REGION Network 146: Step[2901] :
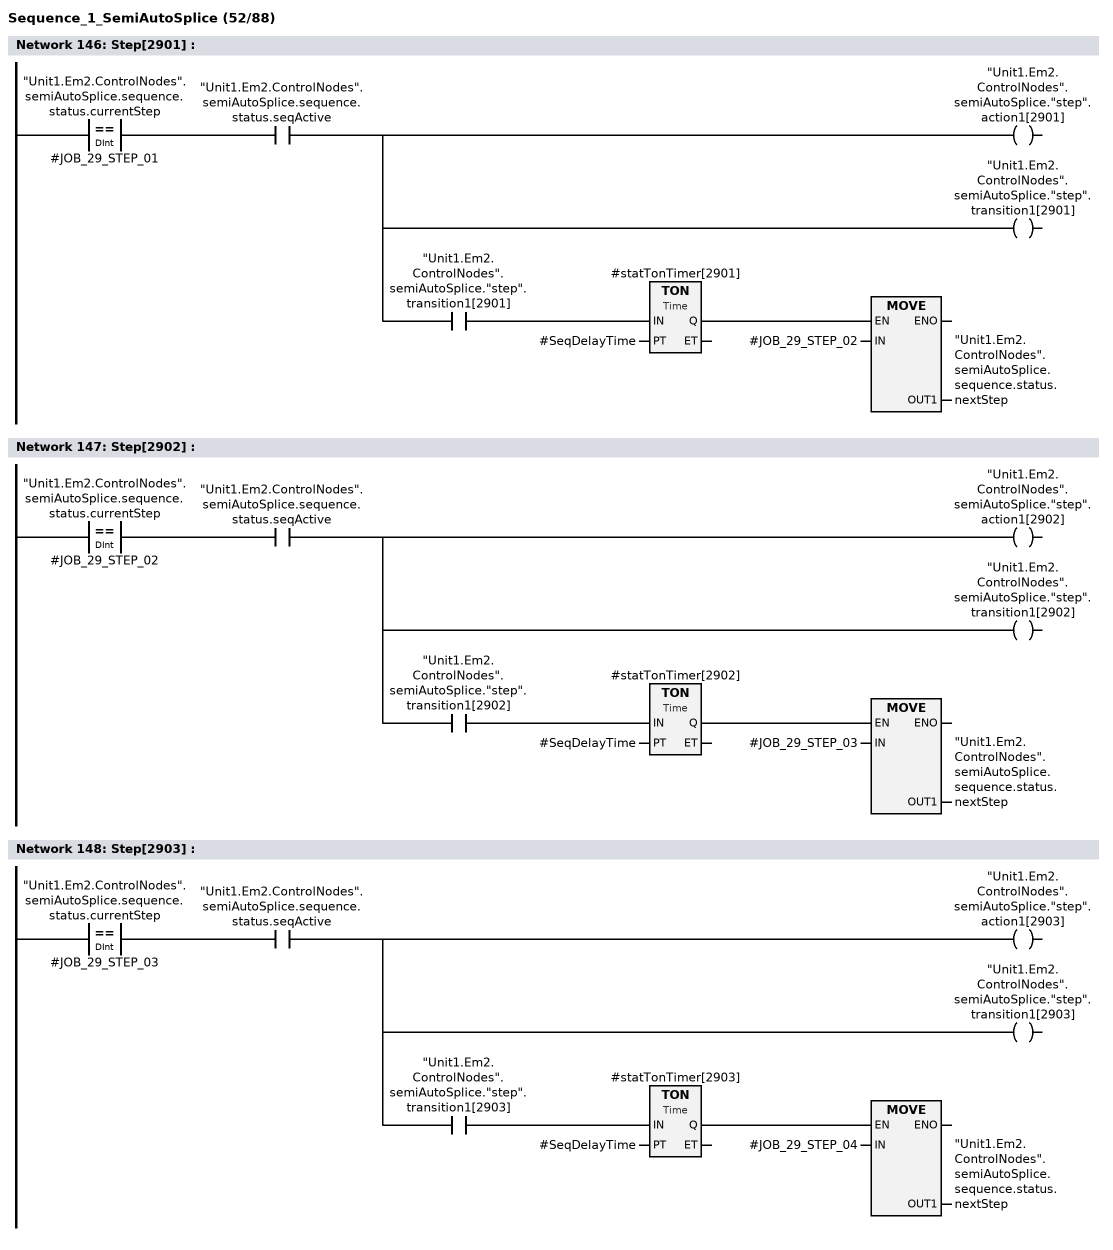
   RUNG wire#powerrail
      { S7_Templates := "SrcType := DInt" } EQ_Contact(in1 := "Unit1.Em2.ControlNodes".semiAutoSplice.sequence.status.currentStep, in2 := #JOB_29_STEP_01)
      Contact( "Unit1.Em2.ControlNodes".semiAutoSplice.sequence.status.seqActive )
      wire#w1
      Coil( "Unit1.Em2.ControlNodes".semiAutoSplice."step".action1[2901] )
   END_RUNG
   RUNG wire#w1
      Coil( "Unit1.Em2.ControlNodes".semiAutoSplice."step".transition1[2901] )
   END_RUNG
   RUNG wire#w1
      Contact( "Unit1.Em2.ControlNodes".semiAutoSplice."step".transition1[2901] )
      { S7_Templates := "time_type := Time" } #statTonTimer[2901].TON(pt := #SeqDelayTime, et =>)
      Move(in := #JOB_29_STEP_02, out1 => "Unit1.Em2.ControlNodes".semiAutoSplice.sequence.status.nextStep)
   END_RUNG
   // the same network as SCL:
   "Unit1.Em2.ControlNodes".semiAutoSplice."step".action1[2901] := ("Unit1.Em2.ControlNodes".semiAutoSplice.sequence.status.currentStep = #JOB_29_STEP_01) AND "Unit1.Em2.ControlNodes".semiAutoSplice.sequence.status.seqActive;
   "Unit1.Em2.ControlNodes".semiAutoSplice."step".transition1[2901] := ("Unit1.Em2.ControlNodes".semiAutoSplice.sequence.status.currentStep = #JOB_29_STEP_01) AND "Unit1.Em2.ControlNodes".semiAutoSplice.sequence.status.seqActive;
   #statTonTimer[2901].TON(IN := ("Unit1.Em2.ControlNodes".semiAutoSplice.sequence.status.currentStep = #JOB_29_STEP_01) AND "Unit1.Em2.ControlNodes".semiAutoSplice.sequence.status.seqActive AND "Unit1.Em2.ControlNodes".semiAutoSplice."step".transition1[2901],
                           PT := #SeqDelayTime);
   IF #statTonTimer[2901].Q THEN
       "Unit1.Em2.ControlNodes".semiAutoSplice.sequence.status.nextStep := #JOB_29_STEP_02;
   END_IF;
END_REGION

REGION Network 147: Step[2902] :
   RUNG wire#powerrail
      { S7_Templates := "SrcType := DInt" } EQ_Contact(in1 := "Unit1.Em2.ControlNodes".semiAutoSplice.sequence.status.currentStep, in2 := #JOB_29_STEP_02)
      Contact( "Unit1.Em2.ControlNodes".semiAutoSplice.sequence.status.seqActive )
      wire#w1
      Coil( "Unit1.Em2.ControlNodes".semiAutoSplice."step".action1[2902] )
   END_RUNG
   RUNG wire#w1
      Coil( "Unit1.Em2.ControlNodes".semiAutoSplice."step".transition1[2902] )
   END_RUNG
   RUNG wire#w1
      Contact( "Unit1.Em2.ControlNodes".semiAutoSplice."step".transition1[2902] )
      { S7_Templates := "time_type := Time" } #statTonTimer[2902].TON(pt := #SeqDelayTime, et =>)
      Move(in := #JOB_29_STEP_03, out1 => "Unit1.Em2.ControlNodes".semiAutoSplice.sequence.status.nextStep)
   END_RUNG
   // the same network as SCL:
   "Unit1.Em2.ControlNodes".semiAutoSplice."step".action1[2902] := ("Unit1.Em2.ControlNodes".semiAutoSplice.sequence.status.currentStep = #JOB_29_STEP_02) AND "Unit1.Em2.ControlNodes".semiAutoSplice.sequence.status.seqActive;
   "Unit1.Em2.ControlNodes".semiAutoSplice."step".transition1[2902] := ("Unit1.Em2.ControlNodes".semiAutoSplice.sequence.status.currentStep = #JOB_29_STEP_02) AND "Unit1.Em2.ControlNodes".semiAutoSplice.sequence.status.seqActive;
   #statTonTimer[2902].TON(IN := ("Unit1.Em2.ControlNodes".semiAutoSplice.sequence.status.currentStep = #JOB_29_STEP_02) AND "Unit1.Em2.ControlNodes".semiAutoSplice.sequence.status.seqActive AND "Unit1.Em2.ControlNodes".semiAutoSplice."step".transition1[2902],
                           PT := #SeqDelayTime);
   IF #statTonTimer[2902].Q THEN
       "Unit1.Em2.ControlNodes".semiAutoSplice.sequence.status.nextStep := #JOB_29_STEP_03;
   END_IF;
END_REGION

REGION Network 148: Step[2903] :
   RUNG wire#powerrail
      { S7_Templates := "SrcType := DInt" } EQ_Contact(in1 := "Unit1.Em2.ControlNodes".semiAutoSplice.sequence.status.currentStep, in2 := #JOB_29_STEP_03)
      Contact( "Unit1.Em2.ControlNodes".semiAutoSplice.sequence.status.seqActive )
      wire#w1
      Coil( "Unit1.Em2.ControlNodes".semiAutoSplice."step".action1[2903] )
   END_RUNG
   RUNG wire#w1
      Coil( "Unit1.Em2.ControlNodes".semiAutoSplice."step".transition1[2903] )
   END_RUNG
   RUNG wire#w1
      Contact( "Unit1.Em2.ControlNodes".semiAutoSplice."step".transition1[2903] )
      { S7_Templates := "time_type := Time" } #statTonTimer[2903].TON(pt := #SeqDelayTime, et =>)
      Move(in := #JOB_29_STEP_04, out1 => "Unit1.Em2.ControlNodes".semiAutoSplice.sequence.status.nextStep)
   END_RUNG
   // the same network as SCL:
   "Unit1.Em2.ControlNodes".semiAutoSplice."step".action1[2903] := ("Unit1.Em2.ControlNodes".semiAutoSplice.sequence.status.currentStep = #JOB_29_STEP_03) AND "Unit1.Em2.ControlNodes".semiAutoSplice.sequence.status.seqActive;
   "Unit1.Em2.ControlNodes".semiAutoSplice."step".transition1[2903] := ("Unit1.Em2.ControlNodes".semiAutoSplice.sequence.status.currentStep = #JOB_29_STEP_03) AND "Unit1.Em2.ControlNodes".semiAutoSplice.sequence.status.seqActive;
   #statTonTimer[2903].TON(IN := ("Unit1.Em2.ControlNodes".semiAutoSplice.sequence.status.currentStep = #JOB_29_STEP_03) AND "Unit1.Em2.ControlNodes".semiAutoSplice.sequence.status.seqActive AND "Unit1.Em2.ControlNodes".semiAutoSplice."step".transition1[2903],
                           PT := #SeqDelayTime);
   IF #statTonTimer[2903].Q THEN
       "Unit1.Em2.ControlNodes".semiAutoSplice.sequence.status.nextStep := #JOB_29_STEP_04;
   END_IF;
END_REGION

REGION Network 149: Step[2904] :
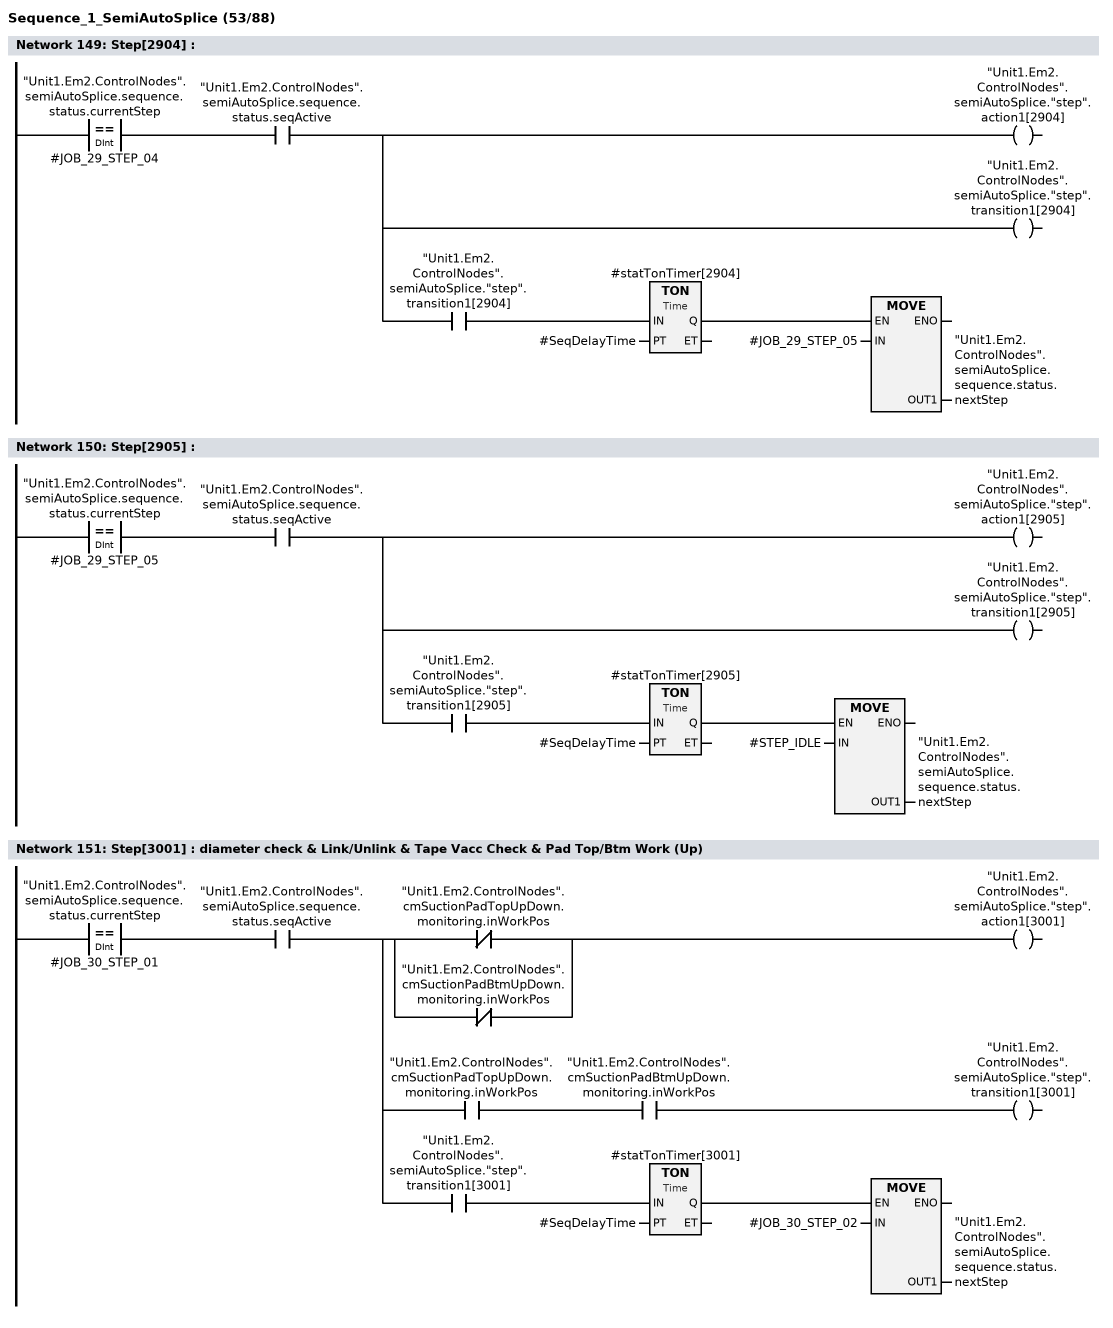
   RUNG wire#powerrail
      { S7_Templates := "SrcType := DInt" } EQ_Contact(in1 := "Unit1.Em2.ControlNodes".semiAutoSplice.sequence.status.currentStep, in2 := #JOB_29_STEP_04)
      Contact( "Unit1.Em2.ControlNodes".semiAutoSplice.sequence.status.seqActive )
      wire#w1
      Coil( "Unit1.Em2.ControlNodes".semiAutoSplice."step".action1[2904] )
   END_RUNG
   RUNG wire#w1
      Coil( "Unit1.Em2.ControlNodes".semiAutoSplice."step".transition1[2904] )
   END_RUNG
   RUNG wire#w1
      Contact( "Unit1.Em2.ControlNodes".semiAutoSplice."step".transition1[2904] )
      { S7_Templates := "time_type := Time" } #statTonTimer[2904].TON(pt := #SeqDelayTime, et =>)
      Move(in := #JOB_29_STEP_05, out1 => "Unit1.Em2.ControlNodes".semiAutoSplice.sequence.status.nextStep)
   END_RUNG
   // the same network as SCL:
   "Unit1.Em2.ControlNodes".semiAutoSplice."step".action1[2904] := ("Unit1.Em2.ControlNodes".semiAutoSplice.sequence.status.currentStep = #JOB_29_STEP_04) AND "Unit1.Em2.ControlNodes".semiAutoSplice.sequence.status.seqActive;
   "Unit1.Em2.ControlNodes".semiAutoSplice."step".transition1[2904] := ("Unit1.Em2.ControlNodes".semiAutoSplice.sequence.status.currentStep = #JOB_29_STEP_04) AND "Unit1.Em2.ControlNodes".semiAutoSplice.sequence.status.seqActive;
   #statTonTimer[2904].TON(IN := ("Unit1.Em2.ControlNodes".semiAutoSplice.sequence.status.currentStep = #JOB_29_STEP_04) AND "Unit1.Em2.ControlNodes".semiAutoSplice.sequence.status.seqActive AND "Unit1.Em2.ControlNodes".semiAutoSplice."step".transition1[2904],
                           PT := #SeqDelayTime);
   IF #statTonTimer[2904].Q THEN
       "Unit1.Em2.ControlNodes".semiAutoSplice.sequence.status.nextStep := #JOB_29_STEP_05;
   END_IF;
END_REGION

REGION Network 150: Step[2905] :
   RUNG wire#powerrail
      { S7_Templates := "SrcType := DInt" } EQ_Contact(in1 := "Unit1.Em2.ControlNodes".semiAutoSplice.sequence.status.currentStep, in2 := #JOB_29_STEP_05)
      Contact( "Unit1.Em2.ControlNodes".semiAutoSplice.sequence.status.seqActive )
      wire#w1
      Coil( "Unit1.Em2.ControlNodes".semiAutoSplice."step".action1[2905] )
   END_RUNG
   RUNG wire#w1
      Coil( "Unit1.Em2.ControlNodes".semiAutoSplice."step".transition1[2905] )
   END_RUNG
   RUNG wire#w1
      Contact( "Unit1.Em2.ControlNodes".semiAutoSplice."step".transition1[2905] )
      { S7_Templates := "time_type := Time" } #statTonTimer[2905].TON(pt := #SeqDelayTime, et =>)
      Move(in := #STEP_IDLE, out1 => "Unit1.Em2.ControlNodes".semiAutoSplice.sequence.status.nextStep)
   END_RUNG
   // the same network as SCL:
   "Unit1.Em2.ControlNodes".semiAutoSplice."step".action1[2905] := ("Unit1.Em2.ControlNodes".semiAutoSplice.sequence.status.currentStep = #JOB_29_STEP_05) AND "Unit1.Em2.ControlNodes".semiAutoSplice.sequence.status.seqActive;
   "Unit1.Em2.ControlNodes".semiAutoSplice."step".transition1[2905] := ("Unit1.Em2.ControlNodes".semiAutoSplice.sequence.status.currentStep = #JOB_29_STEP_05) AND "Unit1.Em2.ControlNodes".semiAutoSplice.sequence.status.seqActive;
   #statTonTimer[2905].TON(IN := ("Unit1.Em2.ControlNodes".semiAutoSplice.sequence.status.currentStep = #JOB_29_STEP_05) AND "Unit1.Em2.ControlNodes".semiAutoSplice.sequence.status.seqActive AND "Unit1.Em2.ControlNodes".semiAutoSplice."step".transition1[2905],
                           PT := #SeqDelayTime);
   IF #statTonTimer[2905].Q THEN
       "Unit1.Em2.ControlNodes".semiAutoSplice.sequence.status.nextStep := #STEP_IDLE;
   END_IF;
END_REGION

REGION Network 151: Step[3001] : diameter check & Link/Unlink & Tape Vacc Check & Pad Top/Btm Work (Up)
   RUNG wire#powerrail
      { S7_Templates := "SrcType := DInt" } EQ_Contact(in1 := "Unit1.Em2.ControlNodes".semiAutoSplice.sequence.status.currentStep, in2 := #JOB_30_STEP_01)
      Contact( "Unit1.Em2.ControlNodes".semiAutoSplice.sequence.status.seqActive )
      wire#w1
      I_Contact( "Unit1.Em2.ControlNodes".cmSuctionPadTopUpDown.monitoring.inWorkPos )
      wire#w2
      Coil( "Unit1.Em2.ControlNodes".semiAutoSplice."step".action1[3001] )
   END_RUNG
   RUNG wire#w1
      I_Contact( "Unit1.Em2.ControlNodes".cmSuctionPadBtmUpDown.monitoring.inWorkPos )
   END_RUNG wire#w2
   RUNG wire#w1
      Contact( "Unit1.Em2.ControlNodes".cmSuctionPadTopUpDown.monitoring.inWorkPos )
      Contact( "Unit1.Em2.ControlNodes".cmSuctionPadBtmUpDown.monitoring.inWorkPos )
      Coil( "Unit1.Em2.ControlNodes".semiAutoSplice."step".transition1[3001] )
   END_RUNG
   RUNG wire#w1
      Contact( "Unit1.Em2.ControlNodes".semiAutoSplice."step".transition1[3001] )
      { S7_Templates := "time_type := Time" } #statTonTimer[3001].TON(pt := #SeqDelayTime, et =>)
      Move(in := #JOB_30_STEP_02, out1 => "Unit1.Em2.ControlNodes".semiAutoSplice.sequence.status.nextStep)
   END_RUNG
   // the same network as SCL:
   #_w1 := ("Unit1.Em2.ControlNodes".semiAutoSplice.sequence.status.currentStep = #JOB_30_STEP_01) AND "Unit1.Em2.ControlNodes".semiAutoSplice.sequence.status.seqActive;
   "Unit1.Em2.ControlNodes".semiAutoSplice."step".action1[3001] := #_w1 AND (NOT "Unit1.Em2.ControlNodes".cmSuctionPadTopUpDown.monitoring.inWorkPos OR NOT "Unit1.Em2.ControlNodes".cmSuctionPadBtmUpDown.monitoring.inWorkPos);
   "Unit1.Em2.ControlNodes".semiAutoSplice."step".transition1[3001] := #_w1 AND "Unit1.Em2.ControlNodes".cmSuctionPadTopUpDown.monitoring.inWorkPos AND "Unit1.Em2.ControlNodes".cmSuctionPadBtmUpDown.monitoring.inWorkPos;
   #statTonTimer[3001].TON(IN := #_w1 AND "Unit1.Em2.ControlNodes".semiAutoSplice."step".transition1[3001],
                           PT := #SeqDelayTime);
   IF #statTonTimer[3001].Q THEN
       "Unit1.Em2.ControlNodes".semiAutoSplice.sequence.status.nextStep := #JOB_30_STEP_02;
   END_IF;
END_REGION

REGION Network 152: Step[3002] :
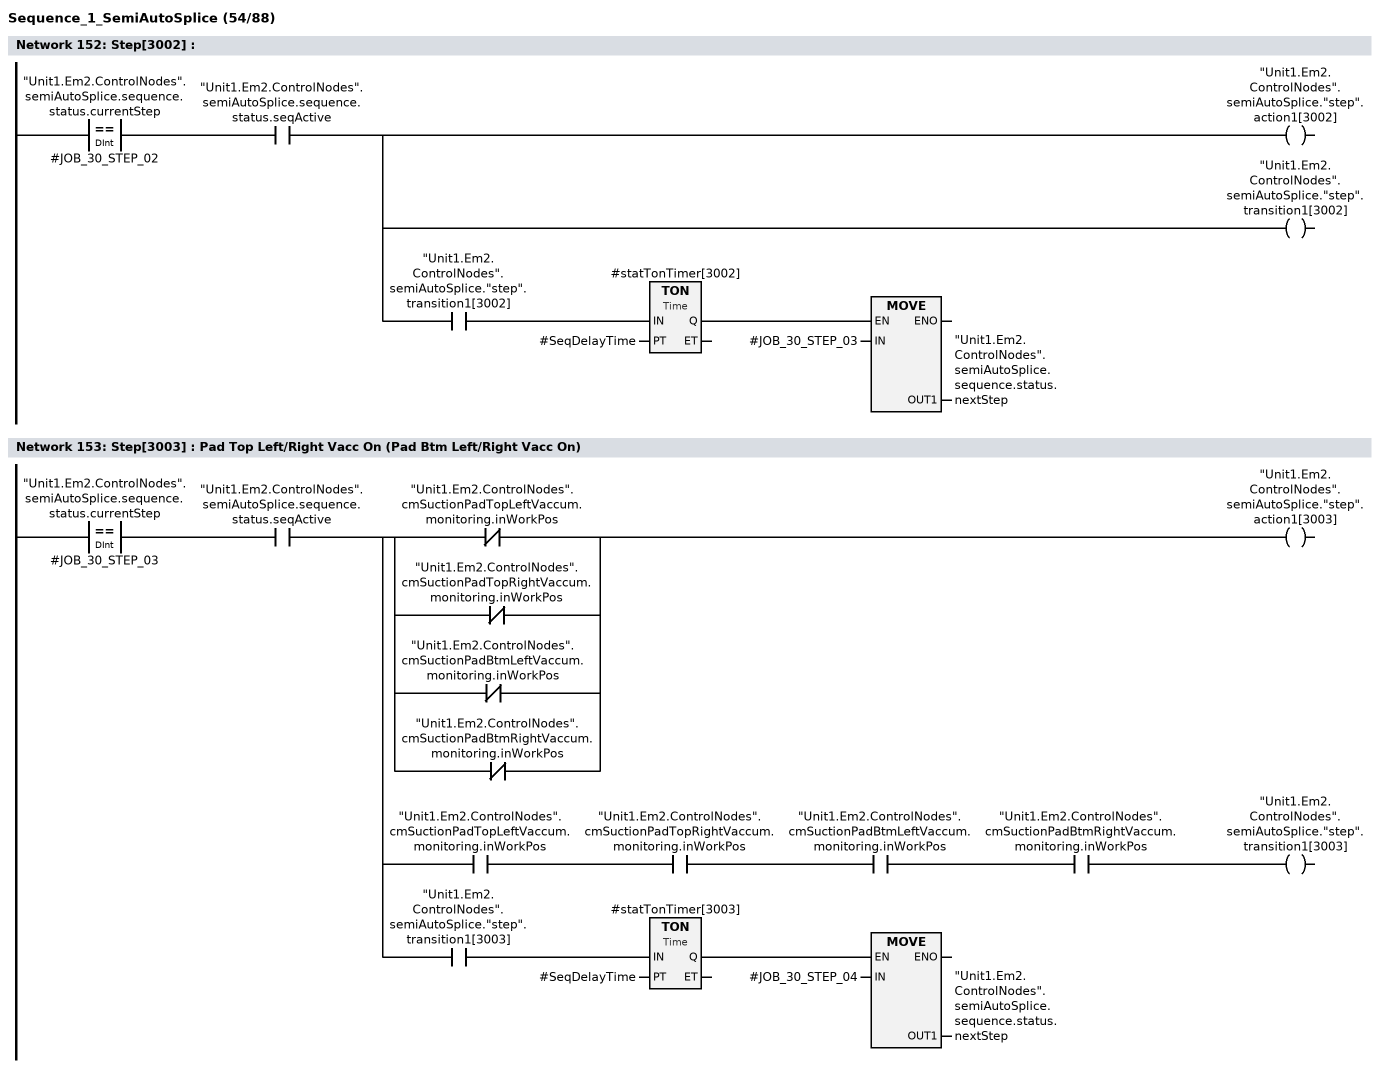
   RUNG wire#powerrail
      { S7_Templates := "SrcType := DInt" } EQ_Contact(in1 := "Unit1.Em2.ControlNodes".semiAutoSplice.sequence.status.currentStep, in2 := #JOB_30_STEP_02)
      Contact( "Unit1.Em2.ControlNodes".semiAutoSplice.sequence.status.seqActive )
      wire#w1
      Coil( "Unit1.Em2.ControlNodes".semiAutoSplice."step".action1[3002] )
   END_RUNG
   RUNG wire#w1
      Coil( "Unit1.Em2.ControlNodes".semiAutoSplice."step".transition1[3002] )
   END_RUNG
   RUNG wire#w1
      Contact( "Unit1.Em2.ControlNodes".semiAutoSplice."step".transition1[3002] )
      { S7_Templates := "time_type := Time" } #statTonTimer[3002].TON(pt := #SeqDelayTime, et =>)
      Move(in := #JOB_30_STEP_03, out1 => "Unit1.Em2.ControlNodes".semiAutoSplice.sequence.status.nextStep)
   END_RUNG
   // the same network as SCL:
   "Unit1.Em2.ControlNodes".semiAutoSplice."step".action1[3002] := ("Unit1.Em2.ControlNodes".semiAutoSplice.sequence.status.currentStep = #JOB_30_STEP_02) AND "Unit1.Em2.ControlNodes".semiAutoSplice.sequence.status.seqActive;
   "Unit1.Em2.ControlNodes".semiAutoSplice."step".transition1[3002] := ("Unit1.Em2.ControlNodes".semiAutoSplice.sequence.status.currentStep = #JOB_30_STEP_02) AND "Unit1.Em2.ControlNodes".semiAutoSplice.sequence.status.seqActive;
   #statTonTimer[3002].TON(IN := ("Unit1.Em2.ControlNodes".semiAutoSplice.sequence.status.currentStep = #JOB_30_STEP_02) AND "Unit1.Em2.ControlNodes".semiAutoSplice.sequence.status.seqActive AND "Unit1.Em2.ControlNodes".semiAutoSplice."step".transition1[3002],
                           PT := #SeqDelayTime);
   IF #statTonTimer[3002].Q THEN
       "Unit1.Em2.ControlNodes".semiAutoSplice.sequence.status.nextStep := #JOB_30_STEP_03;
   END_IF;
END_REGION

REGION Network 153: Step[3003] : Pad Top Left/Right Vacc On (Pad Btm Left/Right Vacc On)
   RUNG wire#powerrail
      { S7_Templates := "SrcType := DInt" } EQ_Contact(in1 := "Unit1.Em2.ControlNodes".semiAutoSplice.sequence.status.currentStep, in2 := #JOB_30_STEP_03)
      Contact( "Unit1.Em2.ControlNodes".semiAutoSplice.sequence.status.seqActive )
      wire#w1
      I_Contact( "Unit1.Em2.ControlNodes".cmSuctionPadTopLeftVaccum.monitoring.inWorkPos )
      wire#w2
      Coil( "Unit1.Em2.ControlNodes".semiAutoSplice."step".action1[3003] )
   END_RUNG
   RUNG wire#w1
      I_Contact( "Unit1.Em2.ControlNodes".cmSuctionPadTopRightVaccum.monitoring.inWorkPos )
   END_RUNG wire#w2
   RUNG wire#w1
      I_Contact( "Unit1.Em2.ControlNodes".cmSuctionPadBtmLeftVaccum.monitoring.inWorkPos )
   END_RUNG wire#w2
   RUNG wire#w1
      I_Contact( "Unit1.Em2.ControlNodes".cmSuctionPadBtmRightVaccum.monitoring.inWorkPos )
   END_RUNG wire#w2
   RUNG wire#w1
      Contact( "Unit1.Em2.ControlNodes".cmSuctionPadTopLeftVaccum.monitoring.inWorkPos )
      Contact( "Unit1.Em2.ControlNodes".cmSuctionPadTopRightVaccum.monitoring.inWorkPos )
      Contact( "Unit1.Em2.ControlNodes".cmSuctionPadBtmLeftVaccum.monitoring.inWorkPos )
      Contact( "Unit1.Em2.ControlNodes".cmSuctionPadBtmRightVaccum.monitoring.inWorkPos )
      Coil( "Unit1.Em2.ControlNodes".semiAutoSplice."step".transition1[3003] )
   END_RUNG
   RUNG wire#w1
      Contact( "Unit1.Em2.ControlNodes".semiAutoSplice."step".transition1[3003] )
      { S7_Templates := "time_type := Time" } #statTonTimer[3003].TON(pt := #SeqDelayTime, et =>)
      Move(in := #JOB_30_STEP_04, out1 => "Unit1.Em2.ControlNodes".semiAutoSplice.sequence.status.nextStep)
   END_RUNG
   // the same network as SCL:
   #_w1 := ("Unit1.Em2.ControlNodes".semiAutoSplice.sequence.status.currentStep = #JOB_30_STEP_03) AND "Unit1.Em2.ControlNodes".semiAutoSplice.sequence.status.seqActive;
   "Unit1.Em2.ControlNodes".semiAutoSplice."step".action1[3003] := #_w1 AND (NOT "Unit1.Em2.ControlNodes".cmSuctionPadTopLeftVaccum.monitoring.inWorkPos OR NOT "Unit1.Em2.ControlNodes".cmSuctionPadTopRightVaccum.monitoring.inWorkPos OR NOT "Unit1.Em2.ControlNodes".cmSuctionPadBtmLeftVaccum.monitoring.inWorkPos OR NOT "Unit1.Em2.ControlNodes".cmSuctionPadBtmRightVaccum.monitoring.inWorkPos);
   "Unit1.Em2.ControlNodes".semiAutoSplice."step".transition1[3003] := #_w1 AND "Unit1.Em2.ControlNodes".cmSuctionPadTopLeftVaccum.monitoring.inWorkPos AND "Unit1.Em2.ControlNodes".cmSuctionPadTopRightVaccum.monitoring.inWorkPos AND "Unit1.Em2.ControlNodes".cmSuctionPadBtmLeftVaccum.monitoring.inWorkPos AND "Unit1.Em2.ControlNodes".cmSuctionPadBtmRightVaccum.monitoring.inWorkPos;
   #statTonTimer[3003].TON(IN := #_w1 AND "Unit1.Em2.ControlNodes".semiAutoSplice."step".transition1[3003],
                           PT := #SeqDelayTime);
   IF #statTonTimer[3003].Q THEN
       "Unit1.Em2.ControlNodes".semiAutoSplice.sequence.status.nextStep := #JOB_30_STEP_04;
   END_IF;
END_REGION

REGION Network 154: Step[3004] :
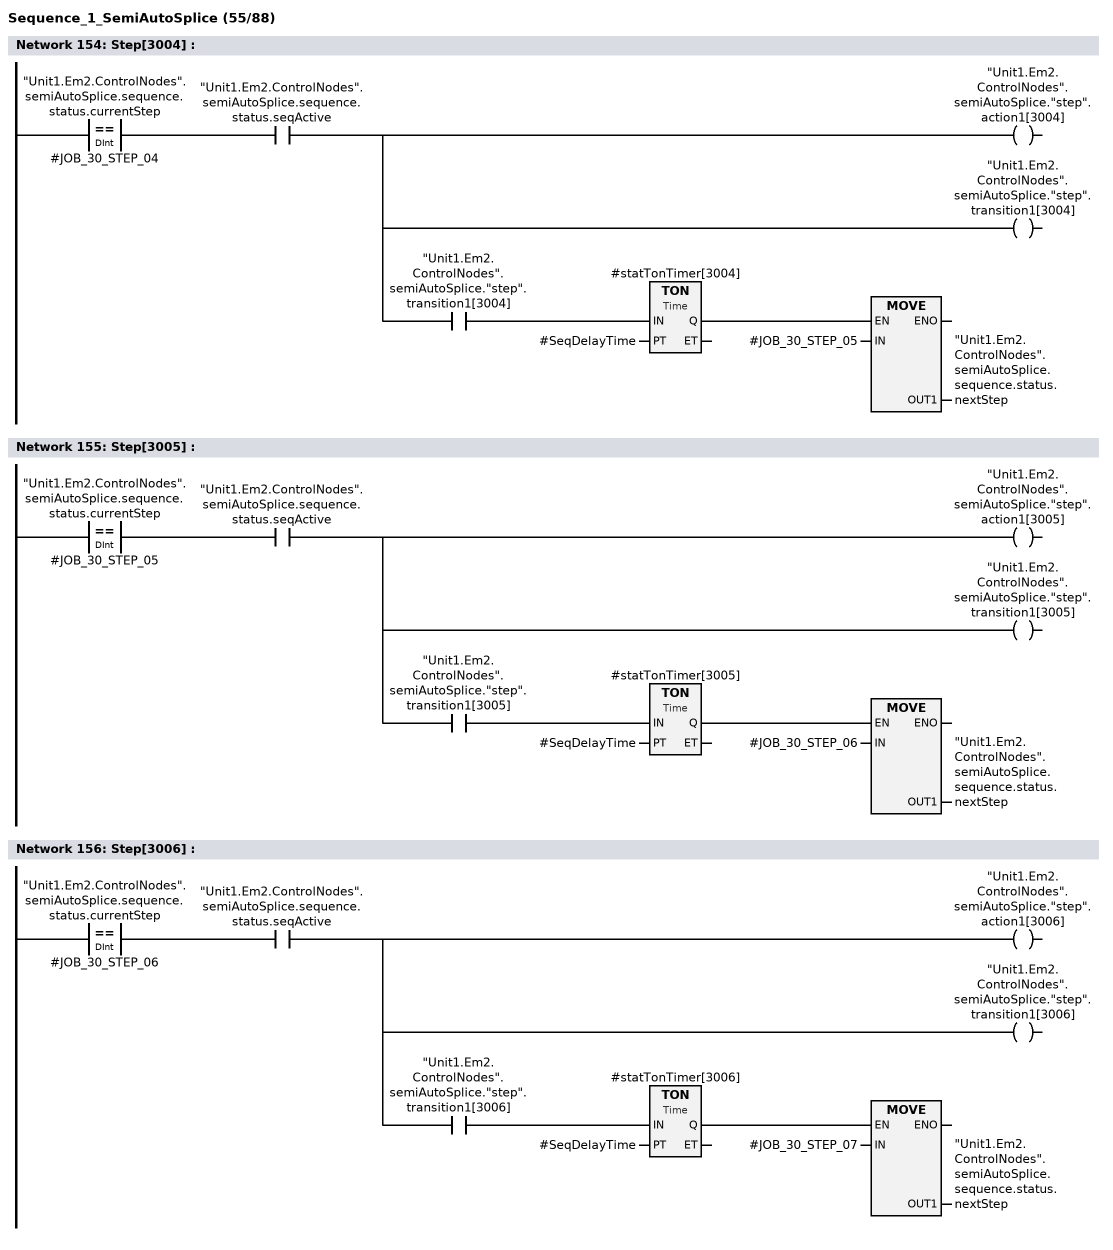
   RUNG wire#powerrail
      { S7_Templates := "SrcType := DInt" } EQ_Contact(in1 := "Unit1.Em2.ControlNodes".semiAutoSplice.sequence.status.currentStep, in2 := #JOB_30_STEP_04)
      Contact( "Unit1.Em2.ControlNodes".semiAutoSplice.sequence.status.seqActive )
      wire#w1
      Coil( "Unit1.Em2.ControlNodes".semiAutoSplice."step".action1[3004] )
   END_RUNG
   RUNG wire#w1
      Coil( "Unit1.Em2.ControlNodes".semiAutoSplice."step".transition1[3004] )
   END_RUNG
   RUNG wire#w1
      Contact( "Unit1.Em2.ControlNodes".semiAutoSplice."step".transition1[3004] )
      { S7_Templates := "time_type := Time" } #statTonTimer[3004].TON(pt := #SeqDelayTime, et =>)
      Move(in := #JOB_30_STEP_05, out1 => "Unit1.Em2.ControlNodes".semiAutoSplice.sequence.status.nextStep)
   END_RUNG
   // the same network as SCL:
   "Unit1.Em2.ControlNodes".semiAutoSplice."step".action1[3004] := ("Unit1.Em2.ControlNodes".semiAutoSplice.sequence.status.currentStep = #JOB_30_STEP_04) AND "Unit1.Em2.ControlNodes".semiAutoSplice.sequence.status.seqActive;
   "Unit1.Em2.ControlNodes".semiAutoSplice."step".transition1[3004] := ("Unit1.Em2.ControlNodes".semiAutoSplice.sequence.status.currentStep = #JOB_30_STEP_04) AND "Unit1.Em2.ControlNodes".semiAutoSplice.sequence.status.seqActive;
   #statTonTimer[3004].TON(IN := ("Unit1.Em2.ControlNodes".semiAutoSplice.sequence.status.currentStep = #JOB_30_STEP_04) AND "Unit1.Em2.ControlNodes".semiAutoSplice.sequence.status.seqActive AND "Unit1.Em2.ControlNodes".semiAutoSplice."step".transition1[3004],
                           PT := #SeqDelayTime);
   IF #statTonTimer[3004].Q THEN
       "Unit1.Em2.ControlNodes".semiAutoSplice.sequence.status.nextStep := #JOB_30_STEP_05;
   END_IF;
END_REGION

REGION Network 155: Step[3005] :
   RUNG wire#powerrail
      { S7_Templates := "SrcType := DInt" } EQ_Contact(in1 := "Unit1.Em2.ControlNodes".semiAutoSplice.sequence.status.currentStep, in2 := #JOB_30_STEP_05)
      Contact( "Unit1.Em2.ControlNodes".semiAutoSplice.sequence.status.seqActive )
      wire#w1
      Coil( "Unit1.Em2.ControlNodes".semiAutoSplice."step".action1[3005] )
   END_RUNG
   RUNG wire#w1
      Coil( "Unit1.Em2.ControlNodes".semiAutoSplice."step".transition1[3005] )
   END_RUNG
   RUNG wire#w1
      Contact( "Unit1.Em2.ControlNodes".semiAutoSplice."step".transition1[3005] )
      { S7_Templates := "time_type := Time" } #statTonTimer[3005].TON(pt := #SeqDelayTime, et =>)
      Move(in := #JOB_30_STEP_06, out1 => "Unit1.Em2.ControlNodes".semiAutoSplice.sequence.status.nextStep)
   END_RUNG
   // the same network as SCL:
   "Unit1.Em2.ControlNodes".semiAutoSplice."step".action1[3005] := ("Unit1.Em2.ControlNodes".semiAutoSplice.sequence.status.currentStep = #JOB_30_STEP_05) AND "Unit1.Em2.ControlNodes".semiAutoSplice.sequence.status.seqActive;
   "Unit1.Em2.ControlNodes".semiAutoSplice."step".transition1[3005] := ("Unit1.Em2.ControlNodes".semiAutoSplice.sequence.status.currentStep = #JOB_30_STEP_05) AND "Unit1.Em2.ControlNodes".semiAutoSplice.sequence.status.seqActive;
   #statTonTimer[3005].TON(IN := ("Unit1.Em2.ControlNodes".semiAutoSplice.sequence.status.currentStep = #JOB_30_STEP_05) AND "Unit1.Em2.ControlNodes".semiAutoSplice.sequence.status.seqActive AND "Unit1.Em2.ControlNodes".semiAutoSplice."step".transition1[3005],
                           PT := #SeqDelayTime);
   IF #statTonTimer[3005].Q THEN
       "Unit1.Em2.ControlNodes".semiAutoSplice.sequence.status.nextStep := #JOB_30_STEP_06;
   END_IF;
END_REGION

REGION Network 156: Step[3006] :
   RUNG wire#powerrail
      { S7_Templates := "SrcType := DInt" } EQ_Contact(in1 := "Unit1.Em2.ControlNodes".semiAutoSplice.sequence.status.currentStep, in2 := #JOB_30_STEP_06)
      Contact( "Unit1.Em2.ControlNodes".semiAutoSplice.sequence.status.seqActive )
      wire#w1
      Coil( "Unit1.Em2.ControlNodes".semiAutoSplice."step".action1[3006] )
   END_RUNG
   RUNG wire#w1
      Coil( "Unit1.Em2.ControlNodes".semiAutoSplice."step".transition1[3006] )
   END_RUNG
   RUNG wire#w1
      Contact( "Unit1.Em2.ControlNodes".semiAutoSplice."step".transition1[3006] )
      { S7_Templates := "time_type := Time" } #statTonTimer[3006].TON(pt := #SeqDelayTime, et =>)
      Move(in := #JOB_30_STEP_07, out1 => "Unit1.Em2.ControlNodes".semiAutoSplice.sequence.status.nextStep)
   END_RUNG
   // the same network as SCL:
   "Unit1.Em2.ControlNodes".semiAutoSplice."step".action1[3006] := ("Unit1.Em2.ControlNodes".semiAutoSplice.sequence.status.currentStep = #JOB_30_STEP_06) AND "Unit1.Em2.ControlNodes".semiAutoSplice.sequence.status.seqActive;
   "Unit1.Em2.ControlNodes".semiAutoSplice."step".transition1[3006] := ("Unit1.Em2.ControlNodes".semiAutoSplice.sequence.status.currentStep = #JOB_30_STEP_06) AND "Unit1.Em2.ControlNodes".semiAutoSplice.sequence.status.seqActive;
   #statTonTimer[3006].TON(IN := ("Unit1.Em2.ControlNodes".semiAutoSplice.sequence.status.currentStep = #JOB_30_STEP_06) AND "Unit1.Em2.ControlNodes".semiAutoSplice.sequence.status.seqActive AND "Unit1.Em2.ControlNodes".semiAutoSplice."step".transition1[3006],
                           PT := #SeqDelayTime);
   IF #statTonTimer[3006].Q THEN
       "Unit1.Em2.ControlNodes".semiAutoSplice.sequence.status.nextStep := #JOB_30_STEP_07;
   END_IF;
END_REGION

REGION Network 157: Step[3007] :
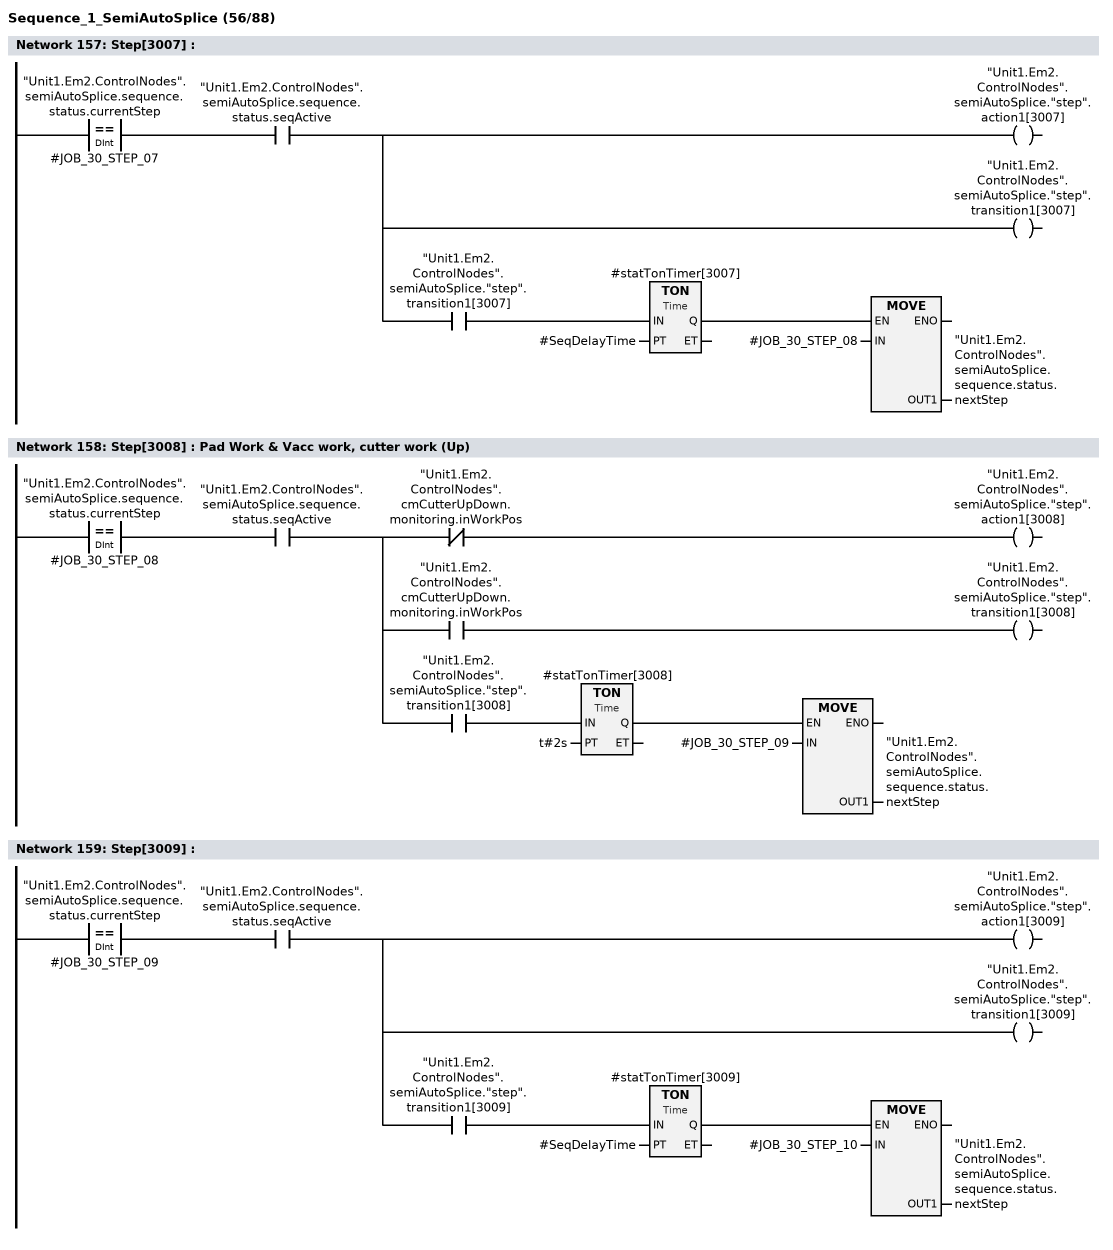
   RUNG wire#powerrail
      { S7_Templates := "SrcType := DInt" } EQ_Contact(in1 := "Unit1.Em2.ControlNodes".semiAutoSplice.sequence.status.currentStep, in2 := #JOB_30_STEP_07)
      Contact( "Unit1.Em2.ControlNodes".semiAutoSplice.sequence.status.seqActive )
      wire#w1
      Coil( "Unit1.Em2.ControlNodes".semiAutoSplice."step".action1[3007] )
   END_RUNG
   RUNG wire#w1
      Coil( "Unit1.Em2.ControlNodes".semiAutoSplice."step".transition1[3007] )
   END_RUNG
   RUNG wire#w1
      Contact( "Unit1.Em2.ControlNodes".semiAutoSplice."step".transition1[3007] )
      { S7_Templates := "time_type := Time" } #statTonTimer[3007].TON(pt := #SeqDelayTime, et =>)
      Move(in := #JOB_30_STEP_08, out1 => "Unit1.Em2.ControlNodes".semiAutoSplice.sequence.status.nextStep)
   END_RUNG
   // the same network as SCL:
   "Unit1.Em2.ControlNodes".semiAutoSplice."step".action1[3007] := ("Unit1.Em2.ControlNodes".semiAutoSplice.sequence.status.currentStep = #JOB_30_STEP_07) AND "Unit1.Em2.ControlNodes".semiAutoSplice.sequence.status.seqActive;
   "Unit1.Em2.ControlNodes".semiAutoSplice."step".transition1[3007] := ("Unit1.Em2.ControlNodes".semiAutoSplice.sequence.status.currentStep = #JOB_30_STEP_07) AND "Unit1.Em2.ControlNodes".semiAutoSplice.sequence.status.seqActive;
   #statTonTimer[3007].TON(IN := ("Unit1.Em2.ControlNodes".semiAutoSplice.sequence.status.currentStep = #JOB_30_STEP_07) AND "Unit1.Em2.ControlNodes".semiAutoSplice.sequence.status.seqActive AND "Unit1.Em2.ControlNodes".semiAutoSplice."step".transition1[3007],
                           PT := #SeqDelayTime);
   IF #statTonTimer[3007].Q THEN
       "Unit1.Em2.ControlNodes".semiAutoSplice.sequence.status.nextStep := #JOB_30_STEP_08;
   END_IF;
END_REGION

REGION Network 158: Step[3008] : Pad Work & Vacc work, cutter work (Up)
   RUNG wire#powerrail
      { S7_Templates := "SrcType := DInt" } EQ_Contact(in1 := "Unit1.Em2.ControlNodes".semiAutoSplice.sequence.status.currentStep, in2 := #JOB_30_STEP_08)
      Contact( "Unit1.Em2.ControlNodes".semiAutoSplice.sequence.status.seqActive )
      wire#w1
      I_Contact( "Unit1.Em2.ControlNodes".cmCutterUpDown.monitoring.inWorkPos )
      Coil( "Unit1.Em2.ControlNodes".semiAutoSplice."step".action1[3008] )
   END_RUNG
   RUNG wire#w1
      Contact( "Unit1.Em2.ControlNodes".cmCutterUpDown.monitoring.inWorkPos )
      Coil( "Unit1.Em2.ControlNodes".semiAutoSplice."step".transition1[3008] )
   END_RUNG
   RUNG wire#w1
      Contact( "Unit1.Em2.ControlNodes".semiAutoSplice."step".transition1[3008] )
      { S7_Templates := "time_type := Time" } #statTonTimer[3008].TON(pt := t#2s, et =>)
      Move(in := #JOB_30_STEP_09, out1 => "Unit1.Em2.ControlNodes".semiAutoSplice.sequence.status.nextStep)
   END_RUNG
   // the same network as SCL:
   #_w1 := ("Unit1.Em2.ControlNodes".semiAutoSplice.sequence.status.currentStep = #JOB_30_STEP_08) AND "Unit1.Em2.ControlNodes".semiAutoSplice.sequence.status.seqActive;
   "Unit1.Em2.ControlNodes".semiAutoSplice."step".action1[3008] := #_w1 AND NOT "Unit1.Em2.ControlNodes".cmCutterUpDown.monitoring.inWorkPos;
   "Unit1.Em2.ControlNodes".semiAutoSplice."step".transition1[3008] := #_w1 AND "Unit1.Em2.ControlNodes".cmCutterUpDown.monitoring.inWorkPos;
   #statTonTimer[3008].TON(IN := #_w1 AND "Unit1.Em2.ControlNodes".semiAutoSplice."step".transition1[3008],
                           PT := t#2s);
   IF #statTonTimer[3008].Q THEN
       "Unit1.Em2.ControlNodes".semiAutoSplice.sequence.status.nextStep := #JOB_30_STEP_09;
   END_IF;
END_REGION

REGION Network 159: Step[3009] :
   RUNG wire#powerrail
      { S7_Templates := "SrcType := DInt" } EQ_Contact(in1 := "Unit1.Em2.ControlNodes".semiAutoSplice.sequence.status.currentStep, in2 := #JOB_30_STEP_09)
      Contact( "Unit1.Em2.ControlNodes".semiAutoSplice.sequence.status.seqActive )
      wire#w1
      Coil( "Unit1.Em2.ControlNodes".semiAutoSplice."step".action1[3009] )
   END_RUNG
   RUNG wire#w1
      Coil( "Unit1.Em2.ControlNodes".semiAutoSplice."step".transition1[3009] )
   END_RUNG
   RUNG wire#w1
      Contact( "Unit1.Em2.ControlNodes".semiAutoSplice."step".transition1[3009] )
      { S7_Templates := "time_type := Time" } #statTonTimer[3009].TON(pt := #SeqDelayTime, et =>)
      Move(in := #JOB_30_STEP_10, out1 => "Unit1.Em2.ControlNodes".semiAutoSplice.sequence.status.nextStep)
   END_RUNG
   // the same network as SCL:
   "Unit1.Em2.ControlNodes".semiAutoSplice."step".action1[3009] := ("Unit1.Em2.ControlNodes".semiAutoSplice.sequence.status.currentStep = #JOB_30_STEP_09) AND "Unit1.Em2.ControlNodes".semiAutoSplice.sequence.status.seqActive;
   "Unit1.Em2.ControlNodes".semiAutoSplice."step".transition1[3009] := ("Unit1.Em2.ControlNodes".semiAutoSplice.sequence.status.currentStep = #JOB_30_STEP_09) AND "Unit1.Em2.ControlNodes".semiAutoSplice.sequence.status.seqActive;
   #statTonTimer[3009].TON(IN := ("Unit1.Em2.ControlNodes".semiAutoSplice.sequence.status.currentStep = #JOB_30_STEP_09) AND "Unit1.Em2.ControlNodes".semiAutoSplice.sequence.status.seqActive AND "Unit1.Em2.ControlNodes".semiAutoSplice."step".transition1[3009],
                           PT := #SeqDelayTime);
   IF #statTonTimer[3009].Q THEN
       "Unit1.Em2.ControlNodes".semiAutoSplice.sequence.status.nextStep := #JOB_30_STEP_10;
   END_IF;
END_REGION

REGION Network 160: Step[3010] : Pad Work & Vacc work, cutter Home (Down)
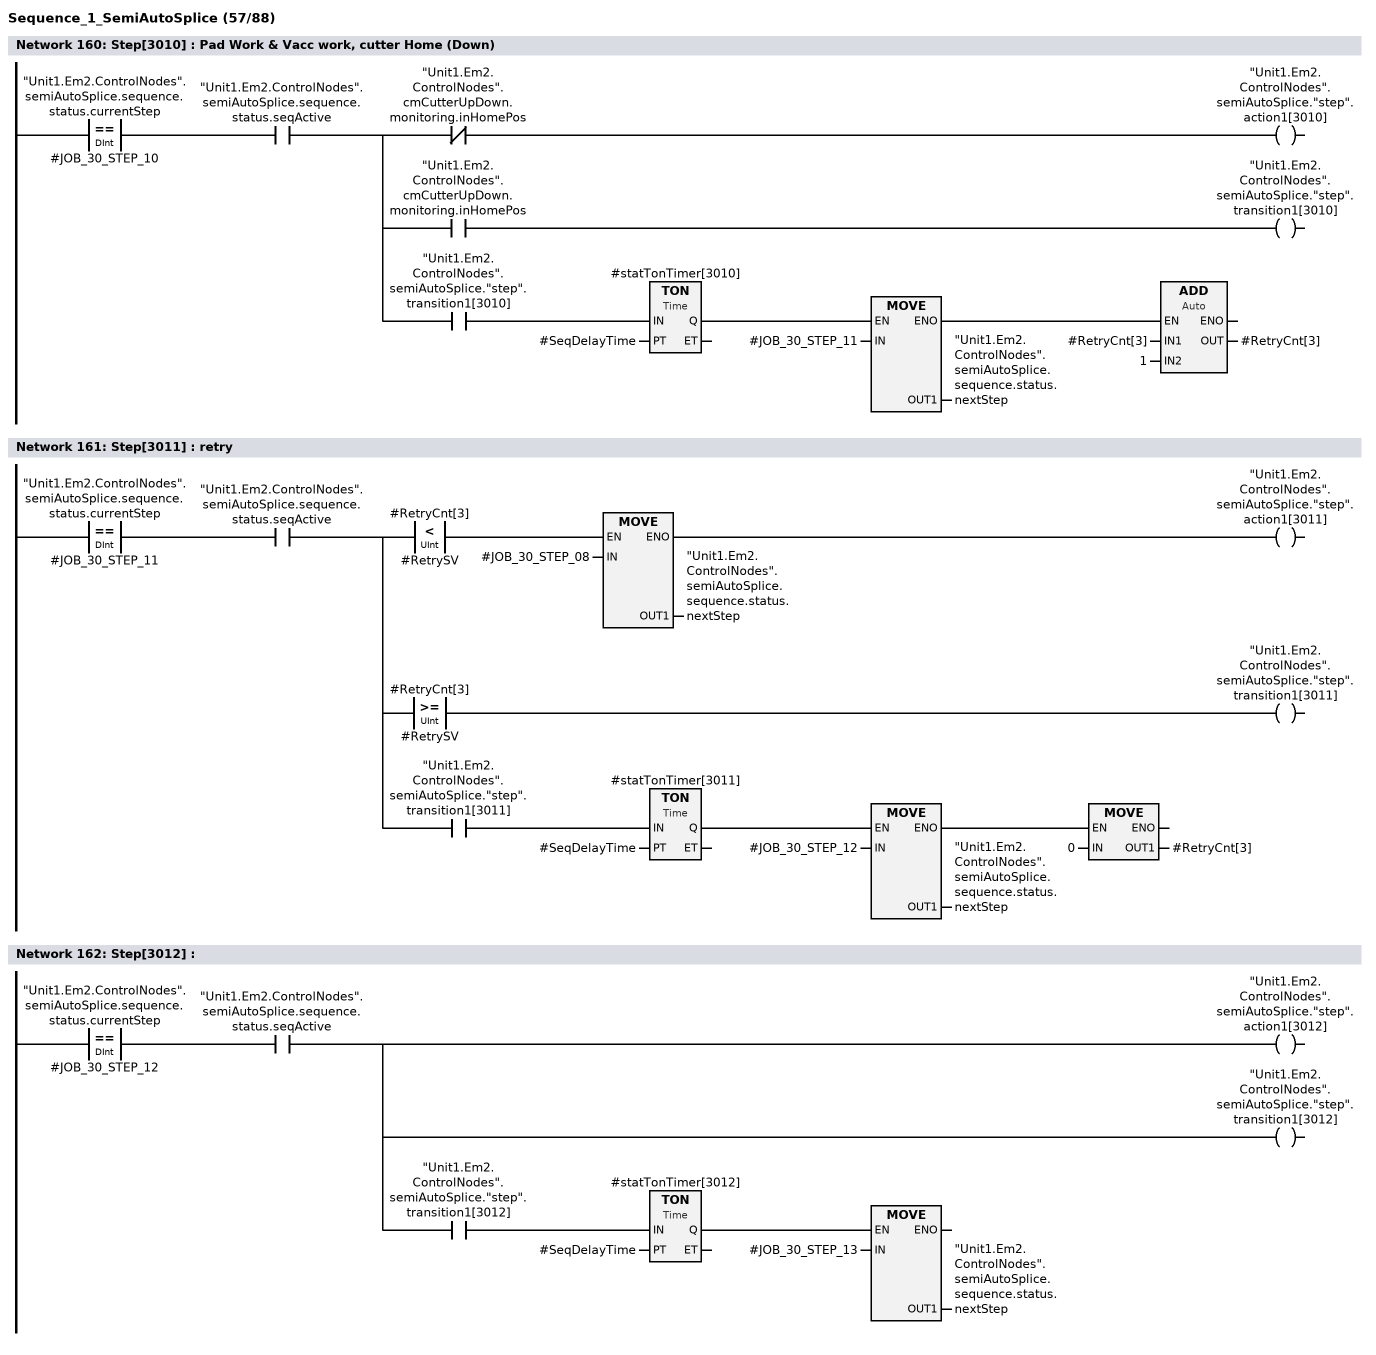
   RUNG wire#powerrail
      { S7_Templates := "SrcType := DInt" } EQ_Contact(in1 := "Unit1.Em2.ControlNodes".semiAutoSplice.sequence.status.currentStep, in2 := #JOB_30_STEP_10)
      Contact( "Unit1.Em2.ControlNodes".semiAutoSplice.sequence.status.seqActive )
      wire#w1
      I_Contact( "Unit1.Em2.ControlNodes".cmCutterUpDown.monitoring.inHomePos )
      Coil( "Unit1.Em2.ControlNodes".semiAutoSplice."step".action1[3010] )
   END_RUNG
   RUNG wire#w1
      Contact( "Unit1.Em2.ControlNodes".cmCutterUpDown.monitoring.inHomePos )
      Coil( "Unit1.Em2.ControlNodes".semiAutoSplice."step".transition1[3010] )
   END_RUNG
   RUNG wire#w1
      Contact( "Unit1.Em2.ControlNodes".semiAutoSplice."step".transition1[3010] )
      { S7_Templates := "time_type := Time" } #statTonTimer[3010].TON(pt := #SeqDelayTime, et =>)
      Move(in := #JOB_30_STEP_11, out1 => "Unit1.Em2.ControlNodes".semiAutoSplice.sequence.status.nextStep)
      Add(in1 := #RetryCnt[3], in2 := 1, out => #RetryCnt[3])
   END_RUNG
   // the same network as SCL:
   #_w1 := ("Unit1.Em2.ControlNodes".semiAutoSplice.sequence.status.currentStep = #JOB_30_STEP_10) AND "Unit1.Em2.ControlNodes".semiAutoSplice.sequence.status.seqActive;
   "Unit1.Em2.ControlNodes".semiAutoSplice."step".action1[3010] := #_w1 AND NOT "Unit1.Em2.ControlNodes".cmCutterUpDown.monitoring.inHomePos;
   "Unit1.Em2.ControlNodes".semiAutoSplice."step".transition1[3010] := #_w1 AND "Unit1.Em2.ControlNodes".cmCutterUpDown.monitoring.inHomePos;
   #statTonTimer[3010].TON(IN := #_w1 AND "Unit1.Em2.ControlNodes".semiAutoSplice."step".transition1[3010],
                           PT := #SeqDelayTime);
   IF #statTonTimer[3010].Q THEN
       "Unit1.Em2.ControlNodes".semiAutoSplice.sequence.status.nextStep := #JOB_30_STEP_11;
       #RetryCnt[3] := #RetryCnt[3] + 1;
   END_IF;
END_REGION

REGION Network 161: Step[3011] : retry
   RUNG wire#powerrail
      { S7_Templates := "SrcType := DInt" } EQ_Contact(in1 := "Unit1.Em2.ControlNodes".semiAutoSplice.sequence.status.currentStep, in2 := #JOB_30_STEP_11)
      Contact( "Unit1.Em2.ControlNodes".semiAutoSplice.sequence.status.seqActive )
      wire#w1
      { S7_Templates := "SrcType := UInt" } LT_Contact(in1 := #RetryCnt[3], in2 := #RetrySV)
      Move(in := #JOB_30_STEP_08, out1 => "Unit1.Em2.ControlNodes".semiAutoSplice.sequence.status.nextStep)
      Coil( "Unit1.Em2.ControlNodes".semiAutoSplice."step".action1[3011] )
   END_RUNG
   RUNG wire#w1
      { S7_Templates := "SrcType := UInt" } GE_Contact(in1 := #RetryCnt[3], in2 := #RetrySV)
      Coil( "Unit1.Em2.ControlNodes".semiAutoSplice."step".transition1[3011] )
   END_RUNG
   RUNG wire#w1
      Contact( "Unit1.Em2.ControlNodes".semiAutoSplice."step".transition1[3011] )
      { S7_Templates := "time_type := Time" } #statTonTimer[3011].TON(pt := #SeqDelayTime, et =>)
      Move(in := #JOB_30_STEP_12, out1 => "Unit1.Em2.ControlNodes".semiAutoSplice.sequence.status.nextStep)
      Move(in := 0, out1 => #RetryCnt[3])
   END_RUNG
   // the same network as SCL:
   #_w1 := ("Unit1.Em2.ControlNodes".semiAutoSplice.sequence.status.currentStep = #JOB_30_STEP_11) AND "Unit1.Em2.ControlNodes".semiAutoSplice.sequence.status.seqActive;
   #_w2 := #_w1 AND (#RetryCnt[3] < #RetrySV);
   IF #_w2 THEN "Unit1.Em2.ControlNodes".semiAutoSplice.sequence.status.nextStep := #JOB_30_STEP_08; END_IF;
   "Unit1.Em2.ControlNodes".semiAutoSplice."step".action1[3011] := #_w2;
   "Unit1.Em2.ControlNodes".semiAutoSplice."step".transition1[3011] := #_w1 AND (#RetryCnt[3] >= #RetrySV);
   #statTonTimer[3011].TON(IN := #_w1 AND "Unit1.Em2.ControlNodes".semiAutoSplice."step".transition1[3011],
                           PT := #SeqDelayTime);
   IF #statTonTimer[3011].Q THEN
       "Unit1.Em2.ControlNodes".semiAutoSplice.sequence.status.nextStep := #JOB_30_STEP_12;
       #RetryCnt[3] := 0;
   END_IF;
END_REGION

REGION Network 162: Step[3012] :
   RUNG wire#powerrail
      { S7_Templates := "SrcType := DInt" } EQ_Contact(in1 := "Unit1.Em2.ControlNodes".semiAutoSplice.sequence.status.currentStep, in2 := #JOB_30_STEP_12)
      Contact( "Unit1.Em2.ControlNodes".semiAutoSplice.sequence.status.seqActive )
      wire#w1
      Coil( "Unit1.Em2.ControlNodes".semiAutoSplice."step".action1[3012] )
   END_RUNG
   RUNG wire#w1
      Coil( "Unit1.Em2.ControlNodes".semiAutoSplice."step".transition1[3012] )
   END_RUNG
   RUNG wire#w1
      Contact( "Unit1.Em2.ControlNodes".semiAutoSplice."step".transition1[3012] )
      { S7_Templates := "time_type := Time" } #statTonTimer[3012].TON(pt := #SeqDelayTime, et =>)
      Move(in := #JOB_30_STEP_13, out1 => "Unit1.Em2.ControlNodes".semiAutoSplice.sequence.status.nextStep)
   END_RUNG
   // the same network as SCL:
   "Unit1.Em2.ControlNodes".semiAutoSplice."step".action1[3012] := ("Unit1.Em2.ControlNodes".semiAutoSplice.sequence.status.currentStep = #JOB_30_STEP_12) AND "Unit1.Em2.ControlNodes".semiAutoSplice.sequence.status.seqActive;
   "Unit1.Em2.ControlNodes".semiAutoSplice."step".transition1[3012] := ("Unit1.Em2.ControlNodes".semiAutoSplice.sequence.status.currentStep = #JOB_30_STEP_12) AND "Unit1.Em2.ControlNodes".semiAutoSplice.sequence.status.seqActive;
   #statTonTimer[3012].TON(IN := ("Unit1.Em2.ControlNodes".semiAutoSplice.sequence.status.currentStep = #JOB_30_STEP_12) AND "Unit1.Em2.ControlNodes".semiAutoSplice.sequence.status.seqActive AND "Unit1.Em2.ControlNodes".semiAutoSplice."step".transition1[3012],
                           PT := #SeqDelayTime);
   IF #statTonTimer[3012].Q THEN
       "Unit1.Em2.ControlNodes".semiAutoSplice.sequence.status.nextStep := #JOB_30_STEP_13;
   END_IF;
END_REGION

REGION Network 163: Step[3013] :
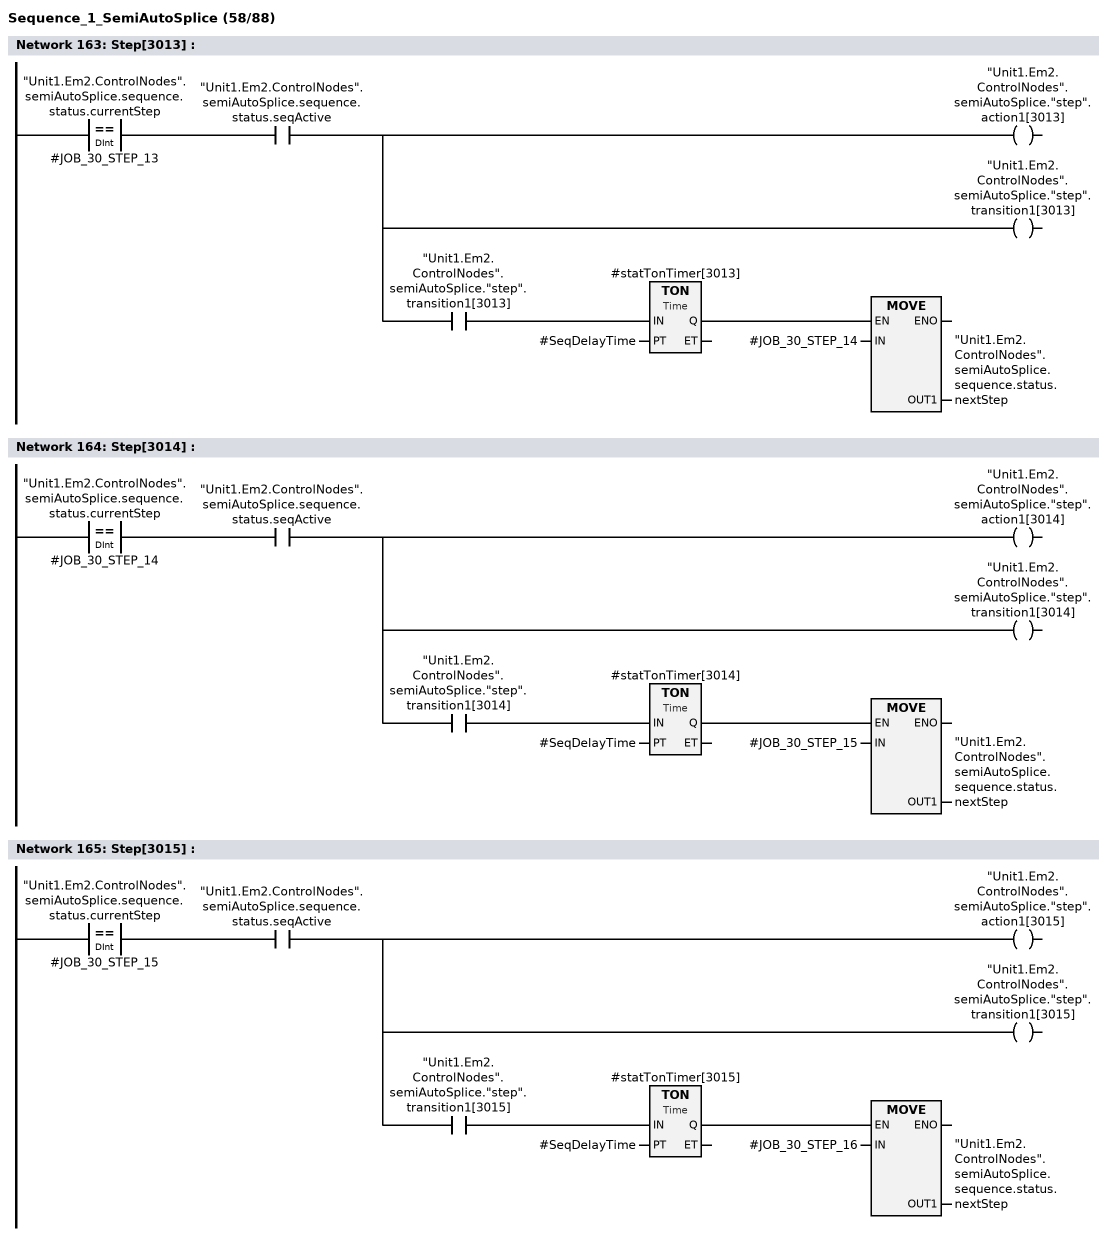
   RUNG wire#powerrail
      { S7_Templates := "SrcType := DInt" } EQ_Contact(in1 := "Unit1.Em2.ControlNodes".semiAutoSplice.sequence.status.currentStep, in2 := #JOB_30_STEP_13)
      Contact( "Unit1.Em2.ControlNodes".semiAutoSplice.sequence.status.seqActive )
      wire#w1
      Coil( "Unit1.Em2.ControlNodes".semiAutoSplice."step".action1[3013] )
   END_RUNG
   RUNG wire#w1
      Coil( "Unit1.Em2.ControlNodes".semiAutoSplice."step".transition1[3013] )
   END_RUNG
   RUNG wire#w1
      Contact( "Unit1.Em2.ControlNodes".semiAutoSplice."step".transition1[3013] )
      { S7_Templates := "time_type := Time" } #statTonTimer[3013].TON(pt := #SeqDelayTime, et =>)
      Move(in := #JOB_30_STEP_14, out1 => "Unit1.Em2.ControlNodes".semiAutoSplice.sequence.status.nextStep)
   END_RUNG
   // the same network as SCL:
   "Unit1.Em2.ControlNodes".semiAutoSplice."step".action1[3013] := ("Unit1.Em2.ControlNodes".semiAutoSplice.sequence.status.currentStep = #JOB_30_STEP_13) AND "Unit1.Em2.ControlNodes".semiAutoSplice.sequence.status.seqActive;
   "Unit1.Em2.ControlNodes".semiAutoSplice."step".transition1[3013] := ("Unit1.Em2.ControlNodes".semiAutoSplice.sequence.status.currentStep = #JOB_30_STEP_13) AND "Unit1.Em2.ControlNodes".semiAutoSplice.sequence.status.seqActive;
   #statTonTimer[3013].TON(IN := ("Unit1.Em2.ControlNodes".semiAutoSplice.sequence.status.currentStep = #JOB_30_STEP_13) AND "Unit1.Em2.ControlNodes".semiAutoSplice.sequence.status.seqActive AND "Unit1.Em2.ControlNodes".semiAutoSplice."step".transition1[3013],
                           PT := #SeqDelayTime);
   IF #statTonTimer[3013].Q THEN
       "Unit1.Em2.ControlNodes".semiAutoSplice.sequence.status.nextStep := #JOB_30_STEP_14;
   END_IF;
END_REGION

REGION Network 164: Step[3014] :
   RUNG wire#powerrail
      { S7_Templates := "SrcType := DInt" } EQ_Contact(in1 := "Unit1.Em2.ControlNodes".semiAutoSplice.sequence.status.currentStep, in2 := #JOB_30_STEP_14)
      Contact( "Unit1.Em2.ControlNodes".semiAutoSplice.sequence.status.seqActive )
      wire#w1
      Coil( "Unit1.Em2.ControlNodes".semiAutoSplice."step".action1[3014] )
   END_RUNG
   RUNG wire#w1
      Coil( "Unit1.Em2.ControlNodes".semiAutoSplice."step".transition1[3014] )
   END_RUNG
   RUNG wire#w1
      Contact( "Unit1.Em2.ControlNodes".semiAutoSplice."step".transition1[3014] )
      { S7_Templates := "time_type := Time" } #statTonTimer[3014].TON(pt := #SeqDelayTime, et =>)
      Move(in := #JOB_30_STEP_15, out1 => "Unit1.Em2.ControlNodes".semiAutoSplice.sequence.status.nextStep)
   END_RUNG
   // the same network as SCL:
   "Unit1.Em2.ControlNodes".semiAutoSplice."step".action1[3014] := ("Unit1.Em2.ControlNodes".semiAutoSplice.sequence.status.currentStep = #JOB_30_STEP_14) AND "Unit1.Em2.ControlNodes".semiAutoSplice.sequence.status.seqActive;
   "Unit1.Em2.ControlNodes".semiAutoSplice."step".transition1[3014] := ("Unit1.Em2.ControlNodes".semiAutoSplice.sequence.status.currentStep = #JOB_30_STEP_14) AND "Unit1.Em2.ControlNodes".semiAutoSplice.sequence.status.seqActive;
   #statTonTimer[3014].TON(IN := ("Unit1.Em2.ControlNodes".semiAutoSplice.sequence.status.currentStep = #JOB_30_STEP_14) AND "Unit1.Em2.ControlNodes".semiAutoSplice.sequence.status.seqActive AND "Unit1.Em2.ControlNodes".semiAutoSplice."step".transition1[3014],
                           PT := #SeqDelayTime);
   IF #statTonTimer[3014].Q THEN
       "Unit1.Em2.ControlNodes".semiAutoSplice.sequence.status.nextStep := #JOB_30_STEP_15;
   END_IF;
END_REGION

REGION Network 165: Step[3015] :
   RUNG wire#powerrail
      { S7_Templates := "SrcType := DInt" } EQ_Contact(in1 := "Unit1.Em2.ControlNodes".semiAutoSplice.sequence.status.currentStep, in2 := #JOB_30_STEP_15)
      Contact( "Unit1.Em2.ControlNodes".semiAutoSplice.sequence.status.seqActive )
      wire#w1
      Coil( "Unit1.Em2.ControlNodes".semiAutoSplice."step".action1[3015] )
   END_RUNG
   RUNG wire#w1
      Coil( "Unit1.Em2.ControlNodes".semiAutoSplice."step".transition1[3015] )
   END_RUNG
   RUNG wire#w1
      Contact( "Unit1.Em2.ControlNodes".semiAutoSplice."step".transition1[3015] )
      { S7_Templates := "time_type := Time" } #statTonTimer[3015].TON(pt := #SeqDelayTime, et =>)
      Move(in := #JOB_30_STEP_16, out1 => "Unit1.Em2.ControlNodes".semiAutoSplice.sequence.status.nextStep)
   END_RUNG
   // the same network as SCL:
   "Unit1.Em2.ControlNodes".semiAutoSplice."step".action1[3015] := ("Unit1.Em2.ControlNodes".semiAutoSplice.sequence.status.currentStep = #JOB_30_STEP_15) AND "Unit1.Em2.ControlNodes".semiAutoSplice.sequence.status.seqActive;
   "Unit1.Em2.ControlNodes".semiAutoSplice."step".transition1[3015] := ("Unit1.Em2.ControlNodes".semiAutoSplice.sequence.status.currentStep = #JOB_30_STEP_15) AND "Unit1.Em2.ControlNodes".semiAutoSplice.sequence.status.seqActive;
   #statTonTimer[3015].TON(IN := ("Unit1.Em2.ControlNodes".semiAutoSplice.sequence.status.currentStep = #JOB_30_STEP_15) AND "Unit1.Em2.ControlNodes".semiAutoSplice.sequence.status.seqActive AND "Unit1.Em2.ControlNodes".semiAutoSplice."step".transition1[3015],
                           PT := #SeqDelayTime);
   IF #statTonTimer[3015].Q THEN
       "Unit1.Em2.ControlNodes".semiAutoSplice.sequence.status.nextStep := #JOB_30_STEP_16;
   END_IF;
END_REGION

REGION Network 166: Step[3016] :
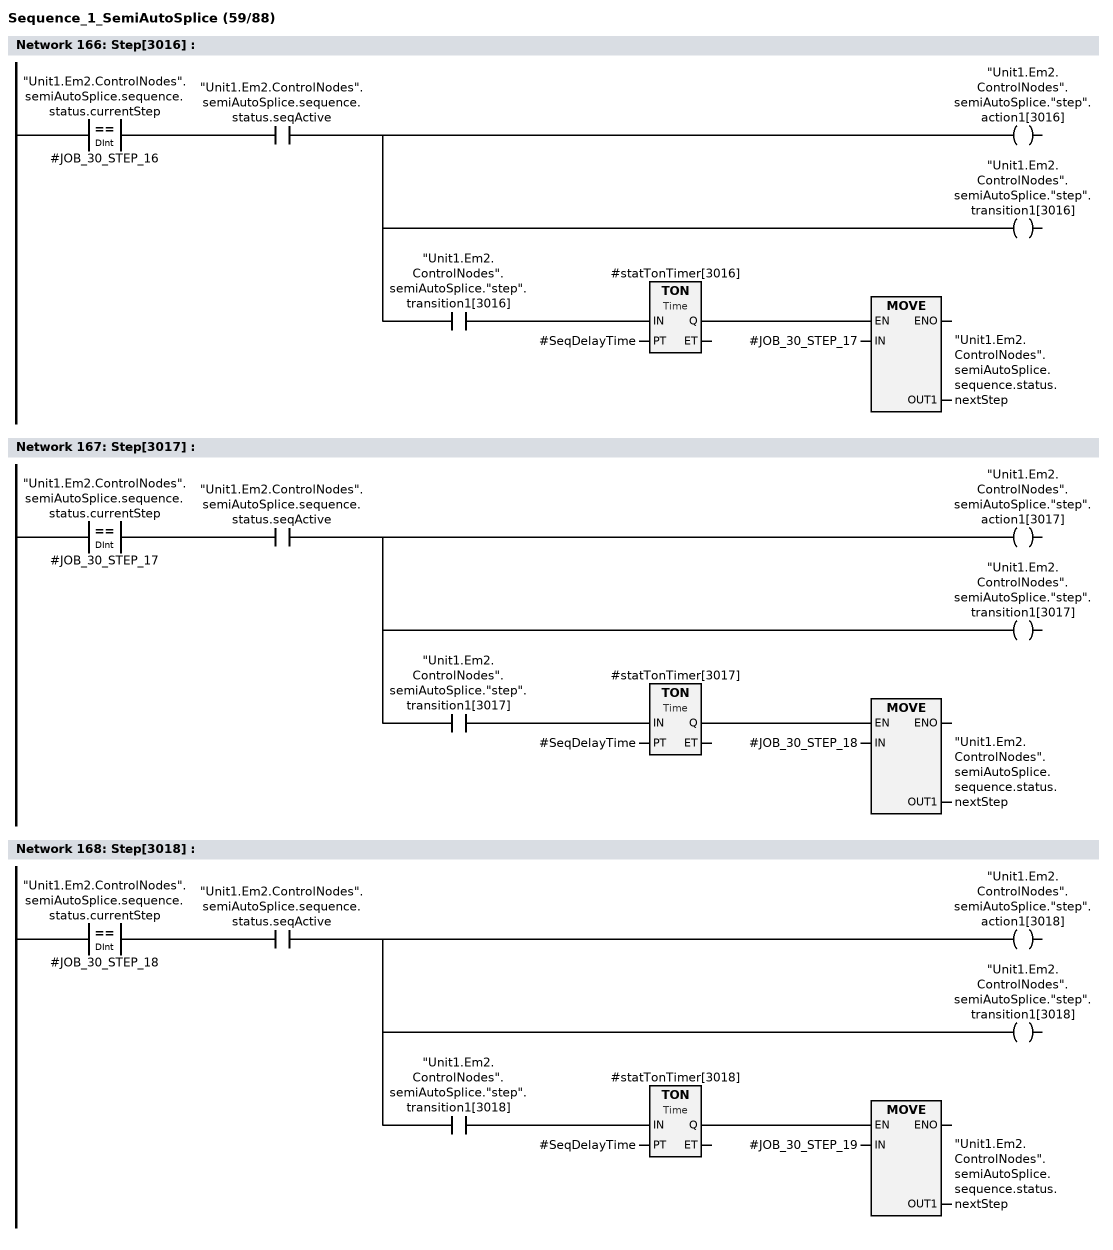
   RUNG wire#powerrail
      { S7_Templates := "SrcType := DInt" } EQ_Contact(in1 := "Unit1.Em2.ControlNodes".semiAutoSplice.sequence.status.currentStep, in2 := #JOB_30_STEP_16)
      Contact( "Unit1.Em2.ControlNodes".semiAutoSplice.sequence.status.seqActive )
      wire#w1
      Coil( "Unit1.Em2.ControlNodes".semiAutoSplice."step".action1[3016] )
   END_RUNG
   RUNG wire#w1
      Coil( "Unit1.Em2.ControlNodes".semiAutoSplice."step".transition1[3016] )
   END_RUNG
   RUNG wire#w1
      Contact( "Unit1.Em2.ControlNodes".semiAutoSplice."step".transition1[3016] )
      { S7_Templates := "time_type := Time" } #statTonTimer[3016].TON(pt := #SeqDelayTime, et =>)
      Move(in := #JOB_30_STEP_17, out1 => "Unit1.Em2.ControlNodes".semiAutoSplice.sequence.status.nextStep)
   END_RUNG
   // the same network as SCL:
   "Unit1.Em2.ControlNodes".semiAutoSplice."step".action1[3016] := ("Unit1.Em2.ControlNodes".semiAutoSplice.sequence.status.currentStep = #JOB_30_STEP_16) AND "Unit1.Em2.ControlNodes".semiAutoSplice.sequence.status.seqActive;
   "Unit1.Em2.ControlNodes".semiAutoSplice."step".transition1[3016] := ("Unit1.Em2.ControlNodes".semiAutoSplice.sequence.status.currentStep = #JOB_30_STEP_16) AND "Unit1.Em2.ControlNodes".semiAutoSplice.sequence.status.seqActive;
   #statTonTimer[3016].TON(IN := ("Unit1.Em2.ControlNodes".semiAutoSplice.sequence.status.currentStep = #JOB_30_STEP_16) AND "Unit1.Em2.ControlNodes".semiAutoSplice.sequence.status.seqActive AND "Unit1.Em2.ControlNodes".semiAutoSplice."step".transition1[3016],
                           PT := #SeqDelayTime);
   IF #statTonTimer[3016].Q THEN
       "Unit1.Em2.ControlNodes".semiAutoSplice.sequence.status.nextStep := #JOB_30_STEP_17;
   END_IF;
END_REGION

REGION Network 167: Step[3017] :
   RUNG wire#powerrail
      { S7_Templates := "SrcType := DInt" } EQ_Contact(in1 := "Unit1.Em2.ControlNodes".semiAutoSplice.sequence.status.currentStep, in2 := #JOB_30_STEP_17)
      Contact( "Unit1.Em2.ControlNodes".semiAutoSplice.sequence.status.seqActive )
      wire#w1
      Coil( "Unit1.Em2.ControlNodes".semiAutoSplice."step".action1[3017] )
   END_RUNG
   RUNG wire#w1
      Coil( "Unit1.Em2.ControlNodes".semiAutoSplice."step".transition1[3017] )
   END_RUNG
   RUNG wire#w1
      Contact( "Unit1.Em2.ControlNodes".semiAutoSplice."step".transition1[3017] )
      { S7_Templates := "time_type := Time" } #statTonTimer[3017].TON(pt := #SeqDelayTime, et =>)
      Move(in := #JOB_30_STEP_18, out1 => "Unit1.Em2.ControlNodes".semiAutoSplice.sequence.status.nextStep)
   END_RUNG
   // the same network as SCL:
   "Unit1.Em2.ControlNodes".semiAutoSplice."step".action1[3017] := ("Unit1.Em2.ControlNodes".semiAutoSplice.sequence.status.currentStep = #JOB_30_STEP_17) AND "Unit1.Em2.ControlNodes".semiAutoSplice.sequence.status.seqActive;
   "Unit1.Em2.ControlNodes".semiAutoSplice."step".transition1[3017] := ("Unit1.Em2.ControlNodes".semiAutoSplice.sequence.status.currentStep = #JOB_30_STEP_17) AND "Unit1.Em2.ControlNodes".semiAutoSplice.sequence.status.seqActive;
   #statTonTimer[3017].TON(IN := ("Unit1.Em2.ControlNodes".semiAutoSplice.sequence.status.currentStep = #JOB_30_STEP_17) AND "Unit1.Em2.ControlNodes".semiAutoSplice.sequence.status.seqActive AND "Unit1.Em2.ControlNodes".semiAutoSplice."step".transition1[3017],
                           PT := #SeqDelayTime);
   IF #statTonTimer[3017].Q THEN
       "Unit1.Em2.ControlNodes".semiAutoSplice.sequence.status.nextStep := #JOB_30_STEP_18;
   END_IF;
END_REGION

REGION Network 168: Step[3018] :
   RUNG wire#powerrail
      { S7_Templates := "SrcType := DInt" } EQ_Contact(in1 := "Unit1.Em2.ControlNodes".semiAutoSplice.sequence.status.currentStep, in2 := #JOB_30_STEP_18)
      Contact( "Unit1.Em2.ControlNodes".semiAutoSplice.sequence.status.seqActive )
      wire#w1
      Coil( "Unit1.Em2.ControlNodes".semiAutoSplice."step".action1[3018] )
   END_RUNG
   RUNG wire#w1
      Coil( "Unit1.Em2.ControlNodes".semiAutoSplice."step".transition1[3018] )
   END_RUNG
   RUNG wire#w1
      Contact( "Unit1.Em2.ControlNodes".semiAutoSplice."step".transition1[3018] )
      { S7_Templates := "time_type := Time" } #statTonTimer[3018].TON(pt := #SeqDelayTime, et =>)
      Move(in := #JOB_30_STEP_19, out1 => "Unit1.Em2.ControlNodes".semiAutoSplice.sequence.status.nextStep)
   END_RUNG
   // the same network as SCL:
   "Unit1.Em2.ControlNodes".semiAutoSplice."step".action1[3018] := ("Unit1.Em2.ControlNodes".semiAutoSplice.sequence.status.currentStep = #JOB_30_STEP_18) AND "Unit1.Em2.ControlNodes".semiAutoSplice.sequence.status.seqActive;
   "Unit1.Em2.ControlNodes".semiAutoSplice."step".transition1[3018] := ("Unit1.Em2.ControlNodes".semiAutoSplice.sequence.status.currentStep = #JOB_30_STEP_18) AND "Unit1.Em2.ControlNodes".semiAutoSplice.sequence.status.seqActive;
   #statTonTimer[3018].TON(IN := ("Unit1.Em2.ControlNodes".semiAutoSplice.sequence.status.currentStep = #JOB_30_STEP_18) AND "Unit1.Em2.ControlNodes".semiAutoSplice.sequence.status.seqActive AND "Unit1.Em2.ControlNodes".semiAutoSplice."step".transition1[3018],
                           PT := #SeqDelayTime);
   IF #statTonTimer[3018].Q THEN
       "Unit1.Em2.ControlNodes".semiAutoSplice.sequence.status.nextStep := #JOB_30_STEP_19;
   END_IF;
END_REGION

REGION Network 169: Step[3019] :
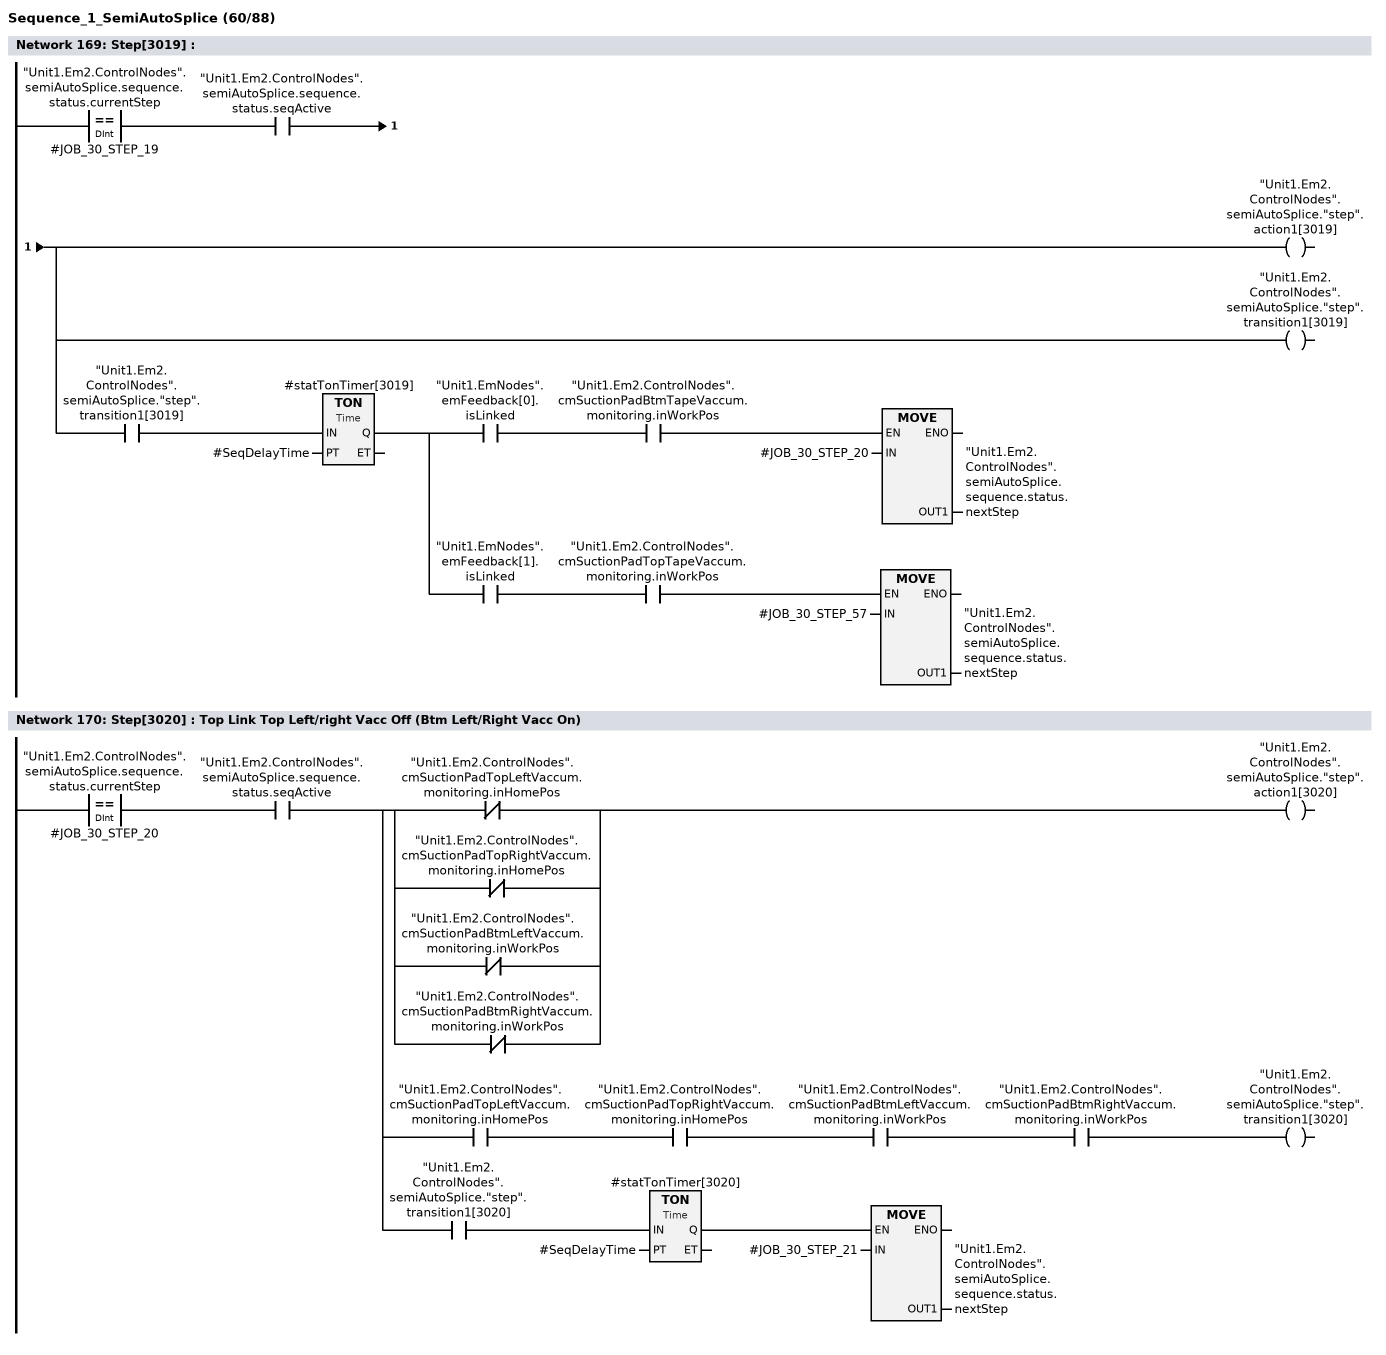
   RUNG wire#powerrail
      { S7_Templates := "SrcType := DInt" } EQ_Contact(in1 := "Unit1.Em2.ControlNodes".semiAutoSplice.sequence.status.currentStep, in2 := #JOB_30_STEP_19)
      Contact( "Unit1.Em2.ControlNodes".semiAutoSplice.sequence.status.seqActive )
      wire#w1
      Coil( "Unit1.Em2.ControlNodes".semiAutoSplice."step".action1[3019] )
   END_RUNG
   RUNG wire#w1
      Coil( "Unit1.Em2.ControlNodes".semiAutoSplice."step".transition1[3019] )
   END_RUNG
   RUNG wire#w1
      Contact( "Unit1.Em2.ControlNodes".semiAutoSplice."step".transition1[3019] )
      { S7_Templates := "time_type := Time" } #statTonTimer[3019].TON(pt := #SeqDelayTime, et =>)
      wire#w2
      Contact( "Unit1.EmNodes".emFeedback[0].isLinked )
      Contact( "Unit1.Em2.ControlNodes".cmSuctionPadBtmTapeVaccum.monitoring.inWorkPos )
      Move(in := #JOB_30_STEP_20, out1 => "Unit1.Em2.ControlNodes".semiAutoSplice.sequence.status.nextStep)
   END_RUNG
   RUNG wire#w2
      Contact( "Unit1.EmNodes".emFeedback[1].isLinked )
      Contact( "Unit1.Em2.ControlNodes".cmSuctionPadTopTapeVaccum.monitoring.inWorkPos )
      Move(in := #JOB_30_STEP_57, out1 => "Unit1.Em2.ControlNodes".semiAutoSplice.sequence.status.nextStep)
   END_RUNG
   // the same network as SCL:
   "Unit1.Em2.ControlNodes".semiAutoSplice."step".action1[3019] := ("Unit1.Em2.ControlNodes".semiAutoSplice.sequence.status.currentStep = #JOB_30_STEP_19) AND "Unit1.Em2.ControlNodes".semiAutoSplice.sequence.status.seqActive;
   "Unit1.Em2.ControlNodes".semiAutoSplice."step".transition1[3019] := ("Unit1.Em2.ControlNodes".semiAutoSplice.sequence.status.currentStep = #JOB_30_STEP_19) AND "Unit1.Em2.ControlNodes".semiAutoSplice.sequence.status.seqActive;
   #statTonTimer[3019].TON(IN := ("Unit1.Em2.ControlNodes".semiAutoSplice.sequence.status.currentStep = #JOB_30_STEP_19) AND "Unit1.Em2.ControlNodes".semiAutoSplice.sequence.status.seqActive AND "Unit1.Em2.ControlNodes".semiAutoSplice."step".transition1[3019],
                           PT := #SeqDelayTime);
   IF #statTonTimer[3019].Q AND "Unit1.EmNodes".emFeedback[0].isLinked AND "Unit1.Em2.ControlNodes".cmSuctionPadBtmTapeVaccum.monitoring.inWorkPos THEN
       "Unit1.Em2.ControlNodes".semiAutoSplice.sequence.status.nextStep := #JOB_30_STEP_20;
   END_IF;
   IF #statTonTimer[3019].Q AND "Unit1.EmNodes".emFeedback[1].isLinked AND "Unit1.Em2.ControlNodes".cmSuctionPadTopTapeVaccum.monitoring.inWorkPos THEN
       "Unit1.Em2.ControlNodes".semiAutoSplice.sequence.status.nextStep := #JOB_30_STEP_57;
   END_IF;
END_REGION

REGION Network 170: Step[3020] : Top Link Top Left/right Vacc Off (Btm Left/Right Vacc On)
   RUNG wire#powerrail
      { S7_Templates := "SrcType := DInt" } EQ_Contact(in1 := "Unit1.Em2.ControlNodes".semiAutoSplice.sequence.status.currentStep, in2 := #JOB_30_STEP_20)
      Contact( "Unit1.Em2.ControlNodes".semiAutoSplice.sequence.status.seqActive )
      wire#w1
      I_Contact( "Unit1.Em2.ControlNodes".cmSuctionPadTopLeftVaccum.monitoring.inHomePos )
      wire#w2
      Coil( "Unit1.Em2.ControlNodes".semiAutoSplice."step".action1[3020] )
   END_RUNG
   RUNG wire#w1
      I_Contact( "Unit1.Em2.ControlNodes".cmSuctionPadTopRightVaccum.monitoring.inHomePos )
   END_RUNG wire#w2
   RUNG wire#w1
      I_Contact( "Unit1.Em2.ControlNodes".cmSuctionPadBtmLeftVaccum.monitoring.inWorkPos )
   END_RUNG wire#w2
   RUNG wire#w1
      I_Contact( "Unit1.Em2.ControlNodes".cmSuctionPadBtmRightVaccum.monitoring.inWorkPos )
   END_RUNG wire#w2
   RUNG wire#w1
      Contact( "Unit1.Em2.ControlNodes".cmSuctionPadTopLeftVaccum.monitoring.inHomePos )
      Contact( "Unit1.Em2.ControlNodes".cmSuctionPadTopRightVaccum.monitoring.inHomePos )
      Contact( "Unit1.Em2.ControlNodes".cmSuctionPadBtmLeftVaccum.monitoring.inWorkPos )
      Contact( "Unit1.Em2.ControlNodes".cmSuctionPadBtmRightVaccum.monitoring.inWorkPos )
      Coil( "Unit1.Em2.ControlNodes".semiAutoSplice."step".transition1[3020] )
   END_RUNG
   RUNG wire#w1
      Contact( "Unit1.Em2.ControlNodes".semiAutoSplice."step".transition1[3020] )
      { S7_Templates := "time_type := Time" } #statTonTimer[3020].TON(pt := #SeqDelayTime, et =>)
      Move(in := #JOB_30_STEP_21, out1 => "Unit1.Em2.ControlNodes".semiAutoSplice.sequence.status.nextStep)
   END_RUNG
   // the same network as SCL:
   #_w1 := ("Unit1.Em2.ControlNodes".semiAutoSplice.sequence.status.currentStep = #JOB_30_STEP_20) AND "Unit1.Em2.ControlNodes".semiAutoSplice.sequence.status.seqActive;
   "Unit1.Em2.ControlNodes".semiAutoSplice."step".action1[3020] := #_w1 AND (NOT "Unit1.Em2.ControlNodes".cmSuctionPadTopLeftVaccum.monitoring.inHomePos OR NOT "Unit1.Em2.ControlNodes".cmSuctionPadTopRightVaccum.monitoring.inHomePos OR NOT "Unit1.Em2.ControlNodes".cmSuctionPadBtmLeftVaccum.monitoring.inWorkPos OR NOT "Unit1.Em2.ControlNodes".cmSuctionPadBtmRightVaccum.monitoring.inWorkPos);
   "Unit1.Em2.ControlNodes".semiAutoSplice."step".transition1[3020] := #_w1 AND "Unit1.Em2.ControlNodes".cmSuctionPadTopLeftVaccum.monitoring.inHomePos AND "Unit1.Em2.ControlNodes".cmSuctionPadTopRightVaccum.monitoring.inHomePos AND "Unit1.Em2.ControlNodes".cmSuctionPadBtmLeftVaccum.monitoring.inWorkPos AND "Unit1.Em2.ControlNodes".cmSuctionPadBtmRightVaccum.monitoring.inWorkPos;
   #statTonTimer[3020].TON(IN := #_w1 AND "Unit1.Em2.ControlNodes".semiAutoSplice."step".transition1[3020],
                           PT := #SeqDelayTime);
   IF #statTonTimer[3020].Q THEN
       "Unit1.Em2.ControlNodes".semiAutoSplice.sequence.status.nextStep := #JOB_30_STEP_21;
   END_IF;
END_REGION

REGION Network 171: Step[3021] : Pad Top Home (Down)
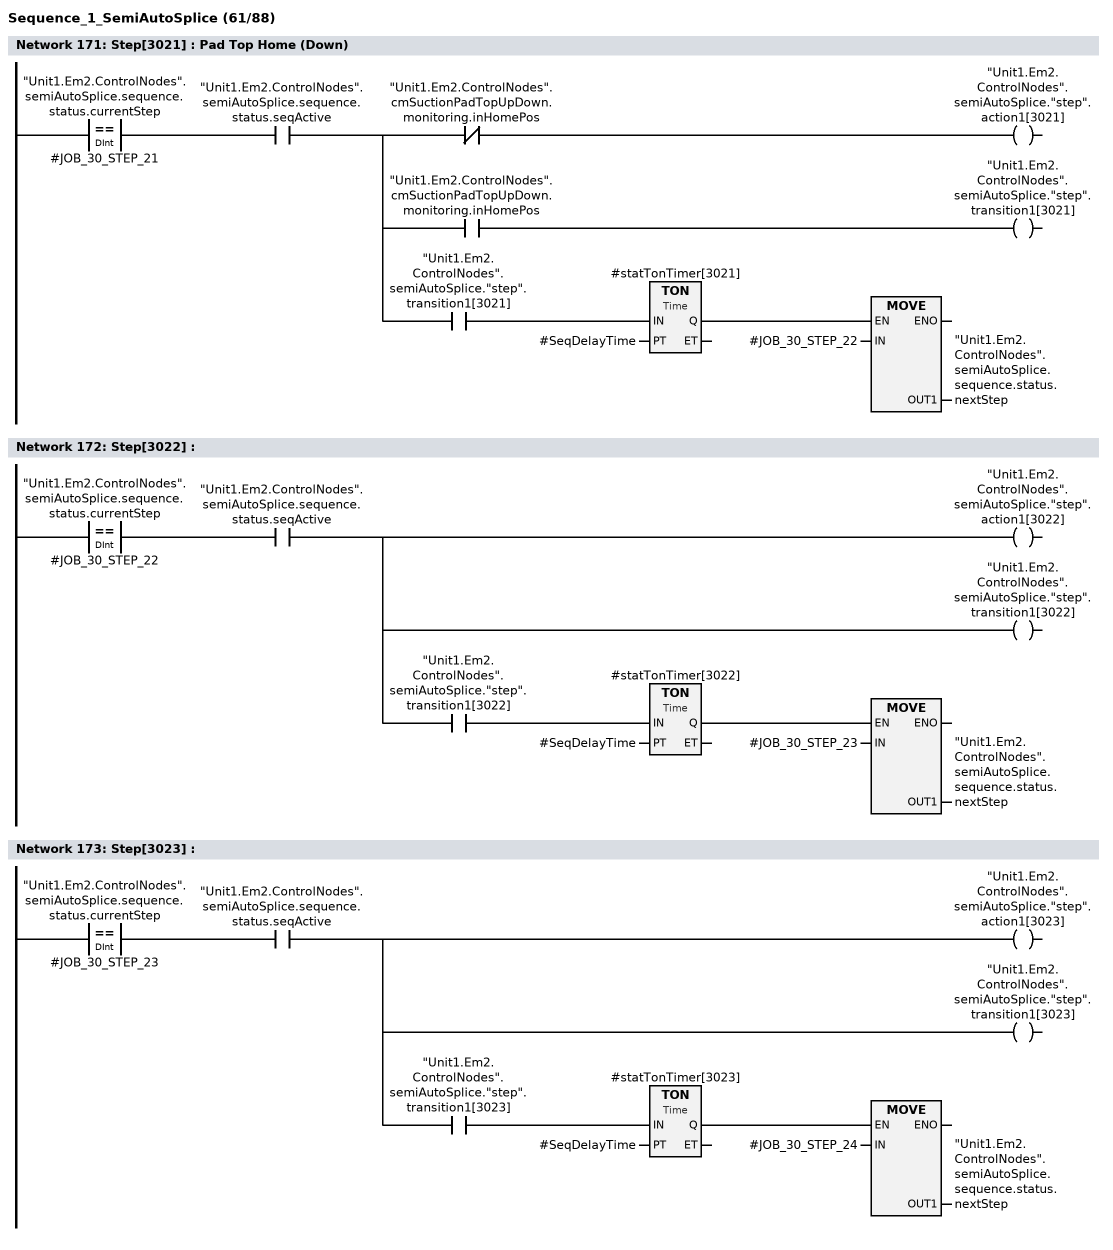
   RUNG wire#powerrail
      { S7_Templates := "SrcType := DInt" } EQ_Contact(in1 := "Unit1.Em2.ControlNodes".semiAutoSplice.sequence.status.currentStep, in2 := #JOB_30_STEP_21)
      Contact( "Unit1.Em2.ControlNodes".semiAutoSplice.sequence.status.seqActive )
      wire#w1
      I_Contact( "Unit1.Em2.ControlNodes".cmSuctionPadTopUpDown.monitoring.inHomePos )
      Coil( "Unit1.Em2.ControlNodes".semiAutoSplice."step".action1[3021] )
   END_RUNG
   RUNG wire#w1
      Contact( "Unit1.Em2.ControlNodes".cmSuctionPadTopUpDown.monitoring.inHomePos )
      Coil( "Unit1.Em2.ControlNodes".semiAutoSplice."step".transition1[3021] )
   END_RUNG
   RUNG wire#w1
      Contact( "Unit1.Em2.ControlNodes".semiAutoSplice."step".transition1[3021] )
      { S7_Templates := "time_type := Time" } #statTonTimer[3021].TON(pt := #SeqDelayTime, et =>)
      Move(in := #JOB_30_STEP_22, out1 => "Unit1.Em2.ControlNodes".semiAutoSplice.sequence.status.nextStep)
   END_RUNG
   // the same network as SCL:
   #_w1 := ("Unit1.Em2.ControlNodes".semiAutoSplice.sequence.status.currentStep = #JOB_30_STEP_21) AND "Unit1.Em2.ControlNodes".semiAutoSplice.sequence.status.seqActive;
   "Unit1.Em2.ControlNodes".semiAutoSplice."step".action1[3021] := #_w1 AND NOT "Unit1.Em2.ControlNodes".cmSuctionPadTopUpDown.monitoring.inHomePos;
   "Unit1.Em2.ControlNodes".semiAutoSplice."step".transition1[3021] := #_w1 AND "Unit1.Em2.ControlNodes".cmSuctionPadTopUpDown.monitoring.inHomePos;
   #statTonTimer[3021].TON(IN := #_w1 AND "Unit1.Em2.ControlNodes".semiAutoSplice."step".transition1[3021],
                           PT := #SeqDelayTime);
   IF #statTonTimer[3021].Q THEN
       "Unit1.Em2.ControlNodes".semiAutoSplice.sequence.status.nextStep := #JOB_30_STEP_22;
   END_IF;
END_REGION

REGION Network 172: Step[3022] :
   RUNG wire#powerrail
      { S7_Templates := "SrcType := DInt" } EQ_Contact(in1 := "Unit1.Em2.ControlNodes".semiAutoSplice.sequence.status.currentStep, in2 := #JOB_30_STEP_22)
      Contact( "Unit1.Em2.ControlNodes".semiAutoSplice.sequence.status.seqActive )
      wire#w1
      Coil( "Unit1.Em2.ControlNodes".semiAutoSplice."step".action1[3022] )
   END_RUNG
   RUNG wire#w1
      Coil( "Unit1.Em2.ControlNodes".semiAutoSplice."step".transition1[3022] )
   END_RUNG
   RUNG wire#w1
      Contact( "Unit1.Em2.ControlNodes".semiAutoSplice."step".transition1[3022] )
      { S7_Templates := "time_type := Time" } #statTonTimer[3022].TON(pt := #SeqDelayTime, et =>)
      Move(in := #JOB_30_STEP_23, out1 => "Unit1.Em2.ControlNodes".semiAutoSplice.sequence.status.nextStep)
   END_RUNG
   // the same network as SCL:
   "Unit1.Em2.ControlNodes".semiAutoSplice."step".action1[3022] := ("Unit1.Em2.ControlNodes".semiAutoSplice.sequence.status.currentStep = #JOB_30_STEP_22) AND "Unit1.Em2.ControlNodes".semiAutoSplice.sequence.status.seqActive;
   "Unit1.Em2.ControlNodes".semiAutoSplice."step".transition1[3022] := ("Unit1.Em2.ControlNodes".semiAutoSplice.sequence.status.currentStep = #JOB_30_STEP_22) AND "Unit1.Em2.ControlNodes".semiAutoSplice.sequence.status.seqActive;
   #statTonTimer[3022].TON(IN := ("Unit1.Em2.ControlNodes".semiAutoSplice.sequence.status.currentStep = #JOB_30_STEP_22) AND "Unit1.Em2.ControlNodes".semiAutoSplice.sequence.status.seqActive AND "Unit1.Em2.ControlNodes".semiAutoSplice."step".transition1[3022],
                           PT := #SeqDelayTime);
   IF #statTonTimer[3022].Q THEN
       "Unit1.Em2.ControlNodes".semiAutoSplice.sequence.status.nextStep := #JOB_30_STEP_23;
   END_IF;
END_REGION

REGION Network 173: Step[3023] :
   RUNG wire#powerrail
      { S7_Templates := "SrcType := DInt" } EQ_Contact(in1 := "Unit1.Em2.ControlNodes".semiAutoSplice.sequence.status.currentStep, in2 := #JOB_30_STEP_23)
      Contact( "Unit1.Em2.ControlNodes".semiAutoSplice.sequence.status.seqActive )
      wire#w1
      Coil( "Unit1.Em2.ControlNodes".semiAutoSplice."step".action1[3023] )
   END_RUNG
   RUNG wire#w1
      Coil( "Unit1.Em2.ControlNodes".semiAutoSplice."step".transition1[3023] )
   END_RUNG
   RUNG wire#w1
      Contact( "Unit1.Em2.ControlNodes".semiAutoSplice."step".transition1[3023] )
      { S7_Templates := "time_type := Time" } #statTonTimer[3023].TON(pt := #SeqDelayTime, et =>)
      Move(in := #JOB_30_STEP_24, out1 => "Unit1.Em2.ControlNodes".semiAutoSplice.sequence.status.nextStep)
   END_RUNG
   // the same network as SCL:
   "Unit1.Em2.ControlNodes".semiAutoSplice."step".action1[3023] := ("Unit1.Em2.ControlNodes".semiAutoSplice.sequence.status.currentStep = #JOB_30_STEP_23) AND "Unit1.Em2.ControlNodes".semiAutoSplice.sequence.status.seqActive;
   "Unit1.Em2.ControlNodes".semiAutoSplice."step".transition1[3023] := ("Unit1.Em2.ControlNodes".semiAutoSplice.sequence.status.currentStep = #JOB_30_STEP_23) AND "Unit1.Em2.ControlNodes".semiAutoSplice.sequence.status.seqActive;
   #statTonTimer[3023].TON(IN := ("Unit1.Em2.ControlNodes".semiAutoSplice.sequence.status.currentStep = #JOB_30_STEP_23) AND "Unit1.Em2.ControlNodes".semiAutoSplice.sequence.status.seqActive AND "Unit1.Em2.ControlNodes".semiAutoSplice."step".transition1[3023],
                           PT := #SeqDelayTime);
   IF #statTonTimer[3023].Q THEN
       "Unit1.Em2.ControlNodes".semiAutoSplice.sequence.status.nextStep := #JOB_30_STEP_24;
   END_IF;
END_REGION

REGION Network 174: Step[3024] : rewinder Top
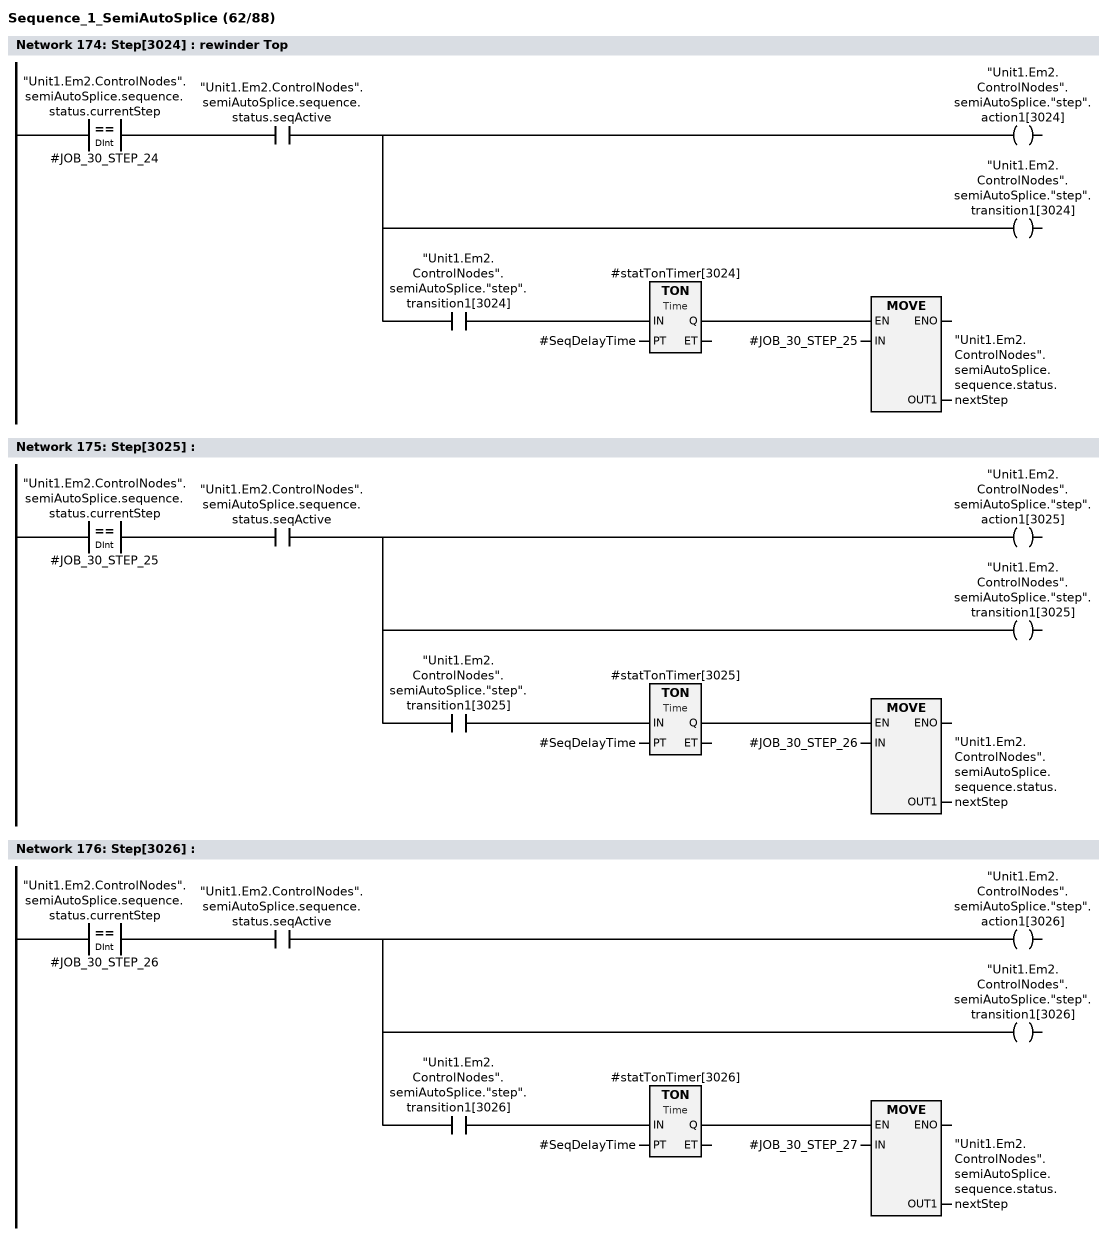
   RUNG wire#powerrail
      { S7_Templates := "SrcType := DInt" } EQ_Contact(in1 := "Unit1.Em2.ControlNodes".semiAutoSplice.sequence.status.currentStep, in2 := #JOB_30_STEP_24)
      Contact( "Unit1.Em2.ControlNodes".semiAutoSplice.sequence.status.seqActive )
      wire#w1
      Coil( "Unit1.Em2.ControlNodes".semiAutoSplice."step".action1[3024] )
   END_RUNG
   RUNG wire#w1
      Coil( "Unit1.Em2.ControlNodes".semiAutoSplice."step".transition1[3024] )
   END_RUNG
   RUNG wire#w1
      Contact( "Unit1.Em2.ControlNodes".semiAutoSplice."step".transition1[3024] )
      { S7_Templates := "time_type := Time" } #statTonTimer[3024].TON(pt := #SeqDelayTime, et =>)
      Move(in := #JOB_30_STEP_25, out1 => "Unit1.Em2.ControlNodes".semiAutoSplice.sequence.status.nextStep)
   END_RUNG
   // the same network as SCL:
   "Unit1.Em2.ControlNodes".semiAutoSplice."step".action1[3024] := ("Unit1.Em2.ControlNodes".semiAutoSplice.sequence.status.currentStep = #JOB_30_STEP_24) AND "Unit1.Em2.ControlNodes".semiAutoSplice.sequence.status.seqActive;
   "Unit1.Em2.ControlNodes".semiAutoSplice."step".transition1[3024] := ("Unit1.Em2.ControlNodes".semiAutoSplice.sequence.status.currentStep = #JOB_30_STEP_24) AND "Unit1.Em2.ControlNodes".semiAutoSplice.sequence.status.seqActive;
   #statTonTimer[3024].TON(IN := ("Unit1.Em2.ControlNodes".semiAutoSplice.sequence.status.currentStep = #JOB_30_STEP_24) AND "Unit1.Em2.ControlNodes".semiAutoSplice.sequence.status.seqActive AND "Unit1.Em2.ControlNodes".semiAutoSplice."step".transition1[3024],
                           PT := #SeqDelayTime);
   IF #statTonTimer[3024].Q THEN
       "Unit1.Em2.ControlNodes".semiAutoSplice.sequence.status.nextStep := #JOB_30_STEP_25;
   END_IF;
END_REGION

REGION Network 175: Step[3025] :
   RUNG wire#powerrail
      { S7_Templates := "SrcType := DInt" } EQ_Contact(in1 := "Unit1.Em2.ControlNodes".semiAutoSplice.sequence.status.currentStep, in2 := #JOB_30_STEP_25)
      Contact( "Unit1.Em2.ControlNodes".semiAutoSplice.sequence.status.seqActive )
      wire#w1
      Coil( "Unit1.Em2.ControlNodes".semiAutoSplice."step".action1[3025] )
   END_RUNG
   RUNG wire#w1
      Coil( "Unit1.Em2.ControlNodes".semiAutoSplice."step".transition1[3025] )
   END_RUNG
   RUNG wire#w1
      Contact( "Unit1.Em2.ControlNodes".semiAutoSplice."step".transition1[3025] )
      { S7_Templates := "time_type := Time" } #statTonTimer[3025].TON(pt := #SeqDelayTime, et =>)
      Move(in := #JOB_30_STEP_26, out1 => "Unit1.Em2.ControlNodes".semiAutoSplice.sequence.status.nextStep)
   END_RUNG
   // the same network as SCL:
   "Unit1.Em2.ControlNodes".semiAutoSplice."step".action1[3025] := ("Unit1.Em2.ControlNodes".semiAutoSplice.sequence.status.currentStep = #JOB_30_STEP_25) AND "Unit1.Em2.ControlNodes".semiAutoSplice.sequence.status.seqActive;
   "Unit1.Em2.ControlNodes".semiAutoSplice."step".transition1[3025] := ("Unit1.Em2.ControlNodes".semiAutoSplice.sequence.status.currentStep = #JOB_30_STEP_25) AND "Unit1.Em2.ControlNodes".semiAutoSplice.sequence.status.seqActive;
   #statTonTimer[3025].TON(IN := ("Unit1.Em2.ControlNodes".semiAutoSplice.sequence.status.currentStep = #JOB_30_STEP_25) AND "Unit1.Em2.ControlNodes".semiAutoSplice.sequence.status.seqActive AND "Unit1.Em2.ControlNodes".semiAutoSplice."step".transition1[3025],
                           PT := #SeqDelayTime);
   IF #statTonTimer[3025].Q THEN
       "Unit1.Em2.ControlNodes".semiAutoSplice.sequence.status.nextStep := #JOB_30_STEP_26;
   END_IF;
END_REGION

REGION Network 176: Step[3026] :
   RUNG wire#powerrail
      { S7_Templates := "SrcType := DInt" } EQ_Contact(in1 := "Unit1.Em2.ControlNodes".semiAutoSplice.sequence.status.currentStep, in2 := #JOB_30_STEP_26)
      Contact( "Unit1.Em2.ControlNodes".semiAutoSplice.sequence.status.seqActive )
      wire#w1
      Coil( "Unit1.Em2.ControlNodes".semiAutoSplice."step".action1[3026] )
   END_RUNG
   RUNG wire#w1
      Coil( "Unit1.Em2.ControlNodes".semiAutoSplice."step".transition1[3026] )
   END_RUNG
   RUNG wire#w1
      Contact( "Unit1.Em2.ControlNodes".semiAutoSplice."step".transition1[3026] )
      { S7_Templates := "time_type := Time" } #statTonTimer[3026].TON(pt := #SeqDelayTime, et =>)
      Move(in := #JOB_30_STEP_27, out1 => "Unit1.Em2.ControlNodes".semiAutoSplice.sequence.status.nextStep)
   END_RUNG
   // the same network as SCL:
   "Unit1.Em2.ControlNodes".semiAutoSplice."step".action1[3026] := ("Unit1.Em2.ControlNodes".semiAutoSplice.sequence.status.currentStep = #JOB_30_STEP_26) AND "Unit1.Em2.ControlNodes".semiAutoSplice.sequence.status.seqActive;
   "Unit1.Em2.ControlNodes".semiAutoSplice."step".transition1[3026] := ("Unit1.Em2.ControlNodes".semiAutoSplice.sequence.status.currentStep = #JOB_30_STEP_26) AND "Unit1.Em2.ControlNodes".semiAutoSplice.sequence.status.seqActive;
   #statTonTimer[3026].TON(IN := ("Unit1.Em2.ControlNodes".semiAutoSplice.sequence.status.currentStep = #JOB_30_STEP_26) AND "Unit1.Em2.ControlNodes".semiAutoSplice.sequence.status.seqActive AND "Unit1.Em2.ControlNodes".semiAutoSplice."step".transition1[3026],
                           PT := #SeqDelayTime);
   IF #statTonTimer[3026].Q THEN
       "Unit1.Em2.ControlNodes".semiAutoSplice.sequence.status.nextStep := #JOB_30_STEP_27;
   END_IF;
END_REGION

REGION Network 177: Step[3027] : Pad Top Work (Up)
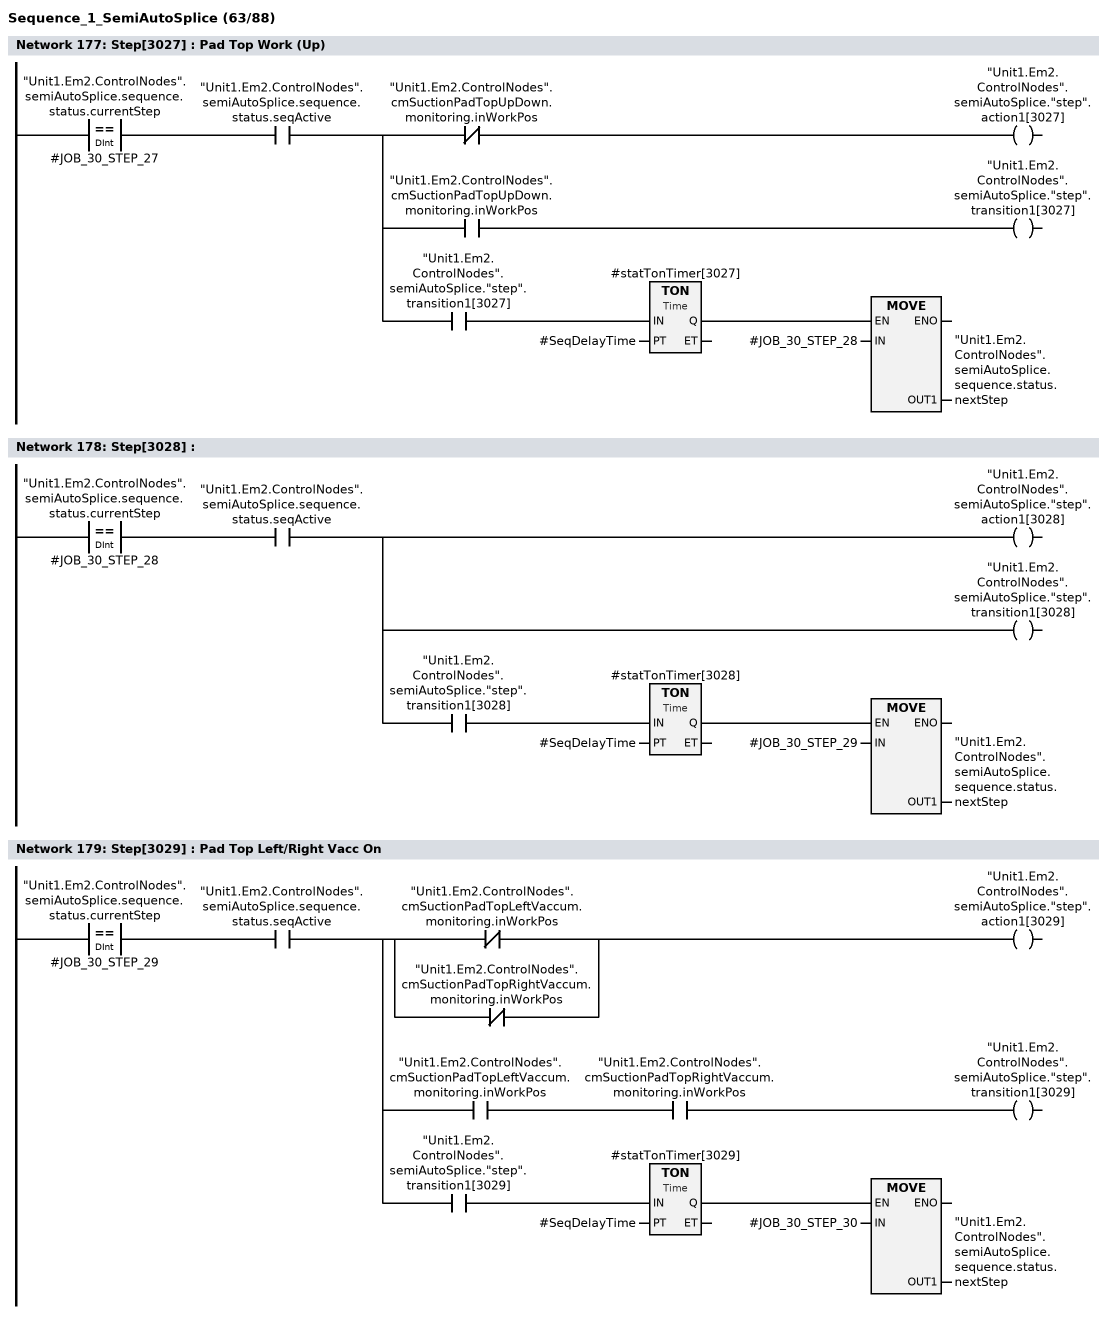
   RUNG wire#powerrail
      { S7_Templates := "SrcType := DInt" } EQ_Contact(in1 := "Unit1.Em2.ControlNodes".semiAutoSplice.sequence.status.currentStep, in2 := #JOB_30_STEP_27)
      Contact( "Unit1.Em2.ControlNodes".semiAutoSplice.sequence.status.seqActive )
      wire#w1
      I_Contact( "Unit1.Em2.ControlNodes".cmSuctionPadTopUpDown.monitoring.inWorkPos )
      Coil( "Unit1.Em2.ControlNodes".semiAutoSplice."step".action1[3027] )
   END_RUNG
   RUNG wire#w1
      Contact( "Unit1.Em2.ControlNodes".cmSuctionPadTopUpDown.monitoring.inWorkPos )
      Coil( "Unit1.Em2.ControlNodes".semiAutoSplice."step".transition1[3027] )
   END_RUNG
   RUNG wire#w1
      Contact( "Unit1.Em2.ControlNodes".semiAutoSplice."step".transition1[3027] )
      { S7_Templates := "time_type := Time" } #statTonTimer[3027].TON(pt := #SeqDelayTime, et =>)
      Move(in := #JOB_30_STEP_28, out1 => "Unit1.Em2.ControlNodes".semiAutoSplice.sequence.status.nextStep)
   END_RUNG
   // the same network as SCL:
   #_w1 := ("Unit1.Em2.ControlNodes".semiAutoSplice.sequence.status.currentStep = #JOB_30_STEP_27) AND "Unit1.Em2.ControlNodes".semiAutoSplice.sequence.status.seqActive;
   "Unit1.Em2.ControlNodes".semiAutoSplice."step".action1[3027] := #_w1 AND NOT "Unit1.Em2.ControlNodes".cmSuctionPadTopUpDown.monitoring.inWorkPos;
   "Unit1.Em2.ControlNodes".semiAutoSplice."step".transition1[3027] := #_w1 AND "Unit1.Em2.ControlNodes".cmSuctionPadTopUpDown.monitoring.inWorkPos;
   #statTonTimer[3027].TON(IN := #_w1 AND "Unit1.Em2.ControlNodes".semiAutoSplice."step".transition1[3027],
                           PT := #SeqDelayTime);
   IF #statTonTimer[3027].Q THEN
       "Unit1.Em2.ControlNodes".semiAutoSplice.sequence.status.nextStep := #JOB_30_STEP_28;
   END_IF;
END_REGION

REGION Network 178: Step[3028] :
   RUNG wire#powerrail
      { S7_Templates := "SrcType := DInt" } EQ_Contact(in1 := "Unit1.Em2.ControlNodes".semiAutoSplice.sequence.status.currentStep, in2 := #JOB_30_STEP_28)
      Contact( "Unit1.Em2.ControlNodes".semiAutoSplice.sequence.status.seqActive )
      wire#w1
      Coil( "Unit1.Em2.ControlNodes".semiAutoSplice."step".action1[3028] )
   END_RUNG
   RUNG wire#w1
      Coil( "Unit1.Em2.ControlNodes".semiAutoSplice."step".transition1[3028] )
   END_RUNG
   RUNG wire#w1
      Contact( "Unit1.Em2.ControlNodes".semiAutoSplice."step".transition1[3028] )
      { S7_Templates := "time_type := Time" } #statTonTimer[3028].TON(pt := #SeqDelayTime, et =>)
      Move(in := #JOB_30_STEP_29, out1 => "Unit1.Em2.ControlNodes".semiAutoSplice.sequence.status.nextStep)
   END_RUNG
   // the same network as SCL:
   "Unit1.Em2.ControlNodes".semiAutoSplice."step".action1[3028] := ("Unit1.Em2.ControlNodes".semiAutoSplice.sequence.status.currentStep = #JOB_30_STEP_28) AND "Unit1.Em2.ControlNodes".semiAutoSplice.sequence.status.seqActive;
   "Unit1.Em2.ControlNodes".semiAutoSplice."step".transition1[3028] := ("Unit1.Em2.ControlNodes".semiAutoSplice.sequence.status.currentStep = #JOB_30_STEP_28) AND "Unit1.Em2.ControlNodes".semiAutoSplice.sequence.status.seqActive;
   #statTonTimer[3028].TON(IN := ("Unit1.Em2.ControlNodes".semiAutoSplice.sequence.status.currentStep = #JOB_30_STEP_28) AND "Unit1.Em2.ControlNodes".semiAutoSplice.sequence.status.seqActive AND "Unit1.Em2.ControlNodes".semiAutoSplice."step".transition1[3028],
                           PT := #SeqDelayTime);
   IF #statTonTimer[3028].Q THEN
       "Unit1.Em2.ControlNodes".semiAutoSplice.sequence.status.nextStep := #JOB_30_STEP_29;
   END_IF;
END_REGION

REGION Network 179: Step[3029] : Pad Top Left/Right Vacc On
   RUNG wire#powerrail
      { S7_Templates := "SrcType := DInt" } EQ_Contact(in1 := "Unit1.Em2.ControlNodes".semiAutoSplice.sequence.status.currentStep, in2 := #JOB_30_STEP_29)
      Contact( "Unit1.Em2.ControlNodes".semiAutoSplice.sequence.status.seqActive )
      wire#w1
      I_Contact( "Unit1.Em2.ControlNodes".cmSuctionPadTopLeftVaccum.monitoring.inWorkPos )
      wire#w2
      Coil( "Unit1.Em2.ControlNodes".semiAutoSplice."step".action1[3029] )
   END_RUNG
   RUNG wire#w1
      I_Contact( "Unit1.Em2.ControlNodes".cmSuctionPadTopRightVaccum.monitoring.inWorkPos )
   END_RUNG wire#w2
   RUNG wire#w1
      Contact( "Unit1.Em2.ControlNodes".cmSuctionPadTopLeftVaccum.monitoring.inWorkPos )
      Contact( "Unit1.Em2.ControlNodes".cmSuctionPadTopRightVaccum.monitoring.inWorkPos )
      Coil( "Unit1.Em2.ControlNodes".semiAutoSplice."step".transition1[3029] )
   END_RUNG
   RUNG wire#w1
      Contact( "Unit1.Em2.ControlNodes".semiAutoSplice."step".transition1[3029] )
      { S7_Templates := "time_type := Time" } #statTonTimer[3029].TON(pt := #SeqDelayTime, et =>)
      Move(in := #JOB_30_STEP_30, out1 => "Unit1.Em2.ControlNodes".semiAutoSplice.sequence.status.nextStep)
   END_RUNG
   // the same network as SCL:
   #_w1 := ("Unit1.Em2.ControlNodes".semiAutoSplice.sequence.status.currentStep = #JOB_30_STEP_29) AND "Unit1.Em2.ControlNodes".semiAutoSplice.sequence.status.seqActive;
   "Unit1.Em2.ControlNodes".semiAutoSplice."step".action1[3029] := #_w1 AND (NOT "Unit1.Em2.ControlNodes".cmSuctionPadTopLeftVaccum.monitoring.inWorkPos OR NOT "Unit1.Em2.ControlNodes".cmSuctionPadTopRightVaccum.monitoring.inWorkPos);
   "Unit1.Em2.ControlNodes".semiAutoSplice."step".transition1[3029] := #_w1 AND "Unit1.Em2.ControlNodes".cmSuctionPadTopLeftVaccum.monitoring.inWorkPos AND "Unit1.Em2.ControlNodes".cmSuctionPadTopRightVaccum.monitoring.inWorkPos;
   #statTonTimer[3029].TON(IN := #_w1 AND "Unit1.Em2.ControlNodes".semiAutoSplice."step".transition1[3029],
                           PT := #SeqDelayTime);
   IF #statTonTimer[3029].Q THEN
       "Unit1.Em2.ControlNodes".semiAutoSplice.sequence.status.nextStep := #JOB_30_STEP_30;
   END_IF;
END_REGION

REGION Network 180: Step[3030] :
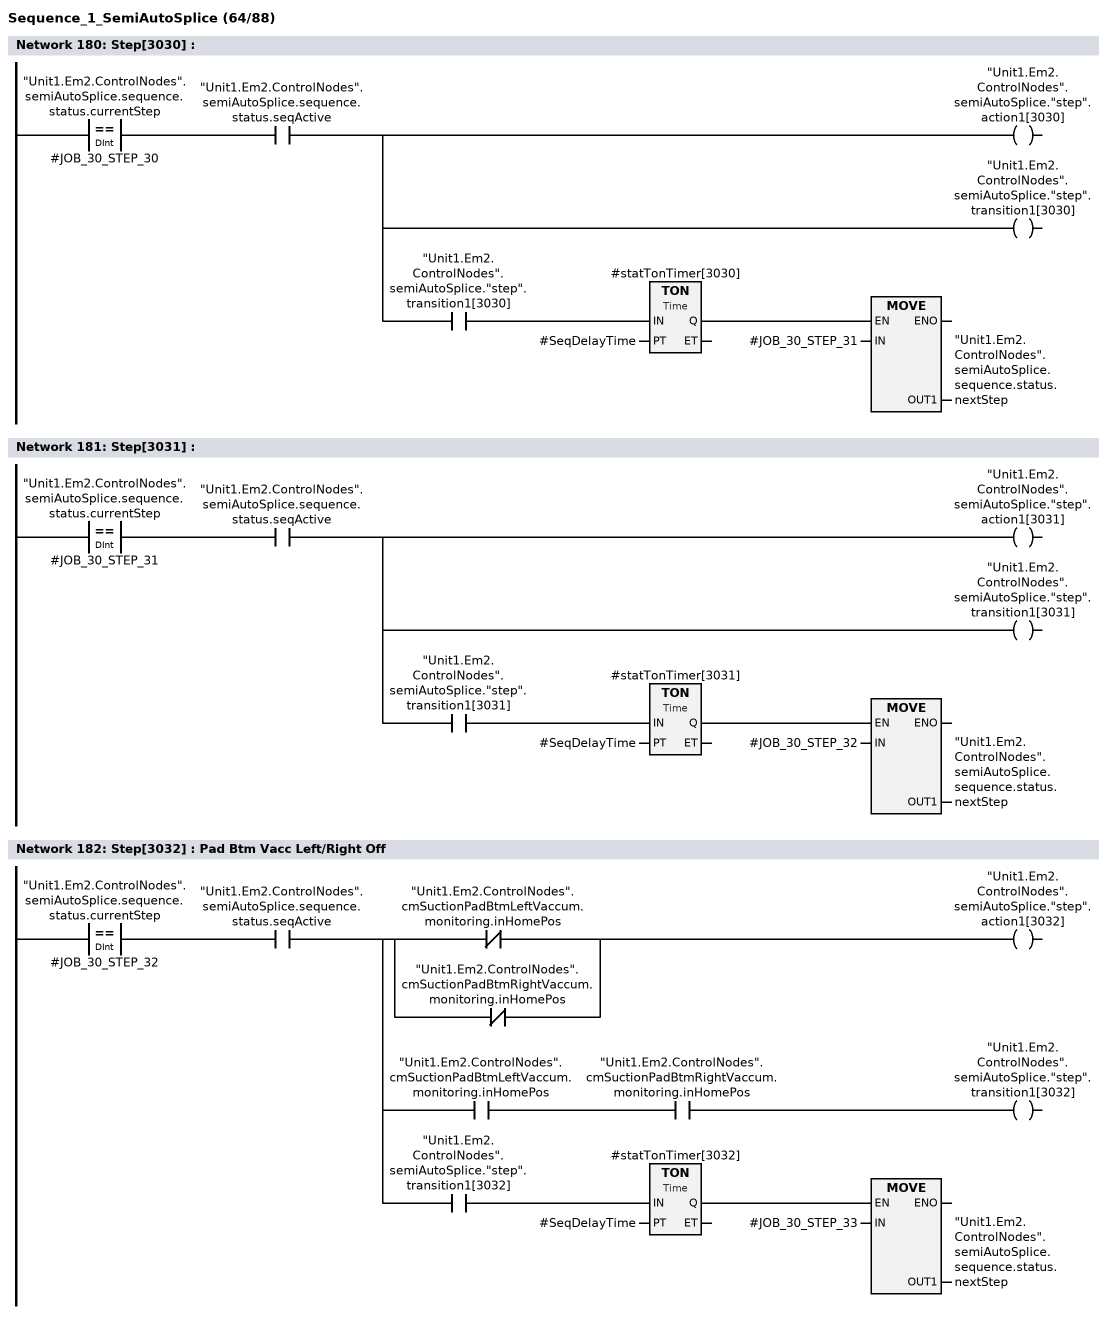
   RUNG wire#powerrail
      { S7_Templates := "SrcType := DInt" } EQ_Contact(in1 := "Unit1.Em2.ControlNodes".semiAutoSplice.sequence.status.currentStep, in2 := #JOB_30_STEP_30)
      Contact( "Unit1.Em2.ControlNodes".semiAutoSplice.sequence.status.seqActive )
      wire#w1
      Coil( "Unit1.Em2.ControlNodes".semiAutoSplice."step".action1[3030] )
   END_RUNG
   RUNG wire#w1
      Coil( "Unit1.Em2.ControlNodes".semiAutoSplice."step".transition1[3030] )
   END_RUNG
   RUNG wire#w1
      Contact( "Unit1.Em2.ControlNodes".semiAutoSplice."step".transition1[3030] )
      { S7_Templates := "time_type := Time" } #statTonTimer[3030].TON(pt := #SeqDelayTime, et =>)
      Move(in := #JOB_30_STEP_31, out1 => "Unit1.Em2.ControlNodes".semiAutoSplice.sequence.status.nextStep)
   END_RUNG
   // the same network as SCL:
   "Unit1.Em2.ControlNodes".semiAutoSplice."step".action1[3030] := ("Unit1.Em2.ControlNodes".semiAutoSplice.sequence.status.currentStep = #JOB_30_STEP_30) AND "Unit1.Em2.ControlNodes".semiAutoSplice.sequence.status.seqActive;
   "Unit1.Em2.ControlNodes".semiAutoSplice."step".transition1[3030] := ("Unit1.Em2.ControlNodes".semiAutoSplice.sequence.status.currentStep = #JOB_30_STEP_30) AND "Unit1.Em2.ControlNodes".semiAutoSplice.sequence.status.seqActive;
   #statTonTimer[3030].TON(IN := ("Unit1.Em2.ControlNodes".semiAutoSplice.sequence.status.currentStep = #JOB_30_STEP_30) AND "Unit1.Em2.ControlNodes".semiAutoSplice.sequence.status.seqActive AND "Unit1.Em2.ControlNodes".semiAutoSplice."step".transition1[3030],
                           PT := #SeqDelayTime);
   IF #statTonTimer[3030].Q THEN
       "Unit1.Em2.ControlNodes".semiAutoSplice.sequence.status.nextStep := #JOB_30_STEP_31;
   END_IF;
END_REGION

REGION Network 181: Step[3031] :
   RUNG wire#powerrail
      { S7_Templates := "SrcType := DInt" } EQ_Contact(in1 := "Unit1.Em2.ControlNodes".semiAutoSplice.sequence.status.currentStep, in2 := #JOB_30_STEP_31)
      Contact( "Unit1.Em2.ControlNodes".semiAutoSplice.sequence.status.seqActive )
      wire#w1
      Coil( "Unit1.Em2.ControlNodes".semiAutoSplice."step".action1[3031] )
   END_RUNG
   RUNG wire#w1
      Coil( "Unit1.Em2.ControlNodes".semiAutoSplice."step".transition1[3031] )
   END_RUNG
   RUNG wire#w1
      Contact( "Unit1.Em2.ControlNodes".semiAutoSplice."step".transition1[3031] )
      { S7_Templates := "time_type := Time" } #statTonTimer[3031].TON(pt := #SeqDelayTime, et =>)
      Move(in := #JOB_30_STEP_32, out1 => "Unit1.Em2.ControlNodes".semiAutoSplice.sequence.status.nextStep)
   END_RUNG
   // the same network as SCL:
   "Unit1.Em2.ControlNodes".semiAutoSplice."step".action1[3031] := ("Unit1.Em2.ControlNodes".semiAutoSplice.sequence.status.currentStep = #JOB_30_STEP_31) AND "Unit1.Em2.ControlNodes".semiAutoSplice.sequence.status.seqActive;
   "Unit1.Em2.ControlNodes".semiAutoSplice."step".transition1[3031] := ("Unit1.Em2.ControlNodes".semiAutoSplice.sequence.status.currentStep = #JOB_30_STEP_31) AND "Unit1.Em2.ControlNodes".semiAutoSplice.sequence.status.seqActive;
   #statTonTimer[3031].TON(IN := ("Unit1.Em2.ControlNodes".semiAutoSplice.sequence.status.currentStep = #JOB_30_STEP_31) AND "Unit1.Em2.ControlNodes".semiAutoSplice.sequence.status.seqActive AND "Unit1.Em2.ControlNodes".semiAutoSplice."step".transition1[3031],
                           PT := #SeqDelayTime);
   IF #statTonTimer[3031].Q THEN
       "Unit1.Em2.ControlNodes".semiAutoSplice.sequence.status.nextStep := #JOB_30_STEP_32;
   END_IF;
END_REGION

REGION Network 182: Step[3032] : Pad Btm Vacc Left/Right Off
   RUNG wire#powerrail
      { S7_Templates := "SrcType := DInt" } EQ_Contact(in1 := "Unit1.Em2.ControlNodes".semiAutoSplice.sequence.status.currentStep, in2 := #JOB_30_STEP_32)
      Contact( "Unit1.Em2.ControlNodes".semiAutoSplice.sequence.status.seqActive )
      wire#w1
      I_Contact( "Unit1.Em2.ControlNodes".cmSuctionPadBtmLeftVaccum.monitoring.inHomePos )
      wire#w2
      Coil( "Unit1.Em2.ControlNodes".semiAutoSplice."step".action1[3032] )
   END_RUNG
   RUNG wire#w1
      I_Contact( "Unit1.Em2.ControlNodes".cmSuctionPadBtmRightVaccum.monitoring.inHomePos )
   END_RUNG wire#w2
   RUNG wire#w1
      Contact( "Unit1.Em2.ControlNodes".cmSuctionPadBtmLeftVaccum.monitoring.inHomePos )
      Contact( "Unit1.Em2.ControlNodes".cmSuctionPadBtmRightVaccum.monitoring.inHomePos )
      Coil( "Unit1.Em2.ControlNodes".semiAutoSplice."step".transition1[3032] )
   END_RUNG
   RUNG wire#w1
      Contact( "Unit1.Em2.ControlNodes".semiAutoSplice."step".transition1[3032] )
      { S7_Templates := "time_type := Time" } #statTonTimer[3032].TON(pt := #SeqDelayTime, et =>)
      Move(in := #JOB_30_STEP_33, out1 => "Unit1.Em2.ControlNodes".semiAutoSplice.sequence.status.nextStep)
   END_RUNG
   // the same network as SCL:
   #_w1 := ("Unit1.Em2.ControlNodes".semiAutoSplice.sequence.status.currentStep = #JOB_30_STEP_32) AND "Unit1.Em2.ControlNodes".semiAutoSplice.sequence.status.seqActive;
   "Unit1.Em2.ControlNodes".semiAutoSplice."step".action1[3032] := #_w1 AND (NOT "Unit1.Em2.ControlNodes".cmSuctionPadBtmLeftVaccum.monitoring.inHomePos OR NOT "Unit1.Em2.ControlNodes".cmSuctionPadBtmRightVaccum.monitoring.inHomePos);
   "Unit1.Em2.ControlNodes".semiAutoSplice."step".transition1[3032] := #_w1 AND "Unit1.Em2.ControlNodes".cmSuctionPadBtmLeftVaccum.monitoring.inHomePos AND "Unit1.Em2.ControlNodes".cmSuctionPadBtmRightVaccum.monitoring.inHomePos;
   #statTonTimer[3032].TON(IN := #_w1 AND "Unit1.Em2.ControlNodes".semiAutoSplice."step".transition1[3032],
                           PT := #SeqDelayTime);
   IF #statTonTimer[3032].Q THEN
       "Unit1.Em2.ControlNodes".semiAutoSplice.sequence.status.nextStep := #JOB_30_STEP_33;
   END_IF;
END_REGION

REGION Network 183: Step[3033] :
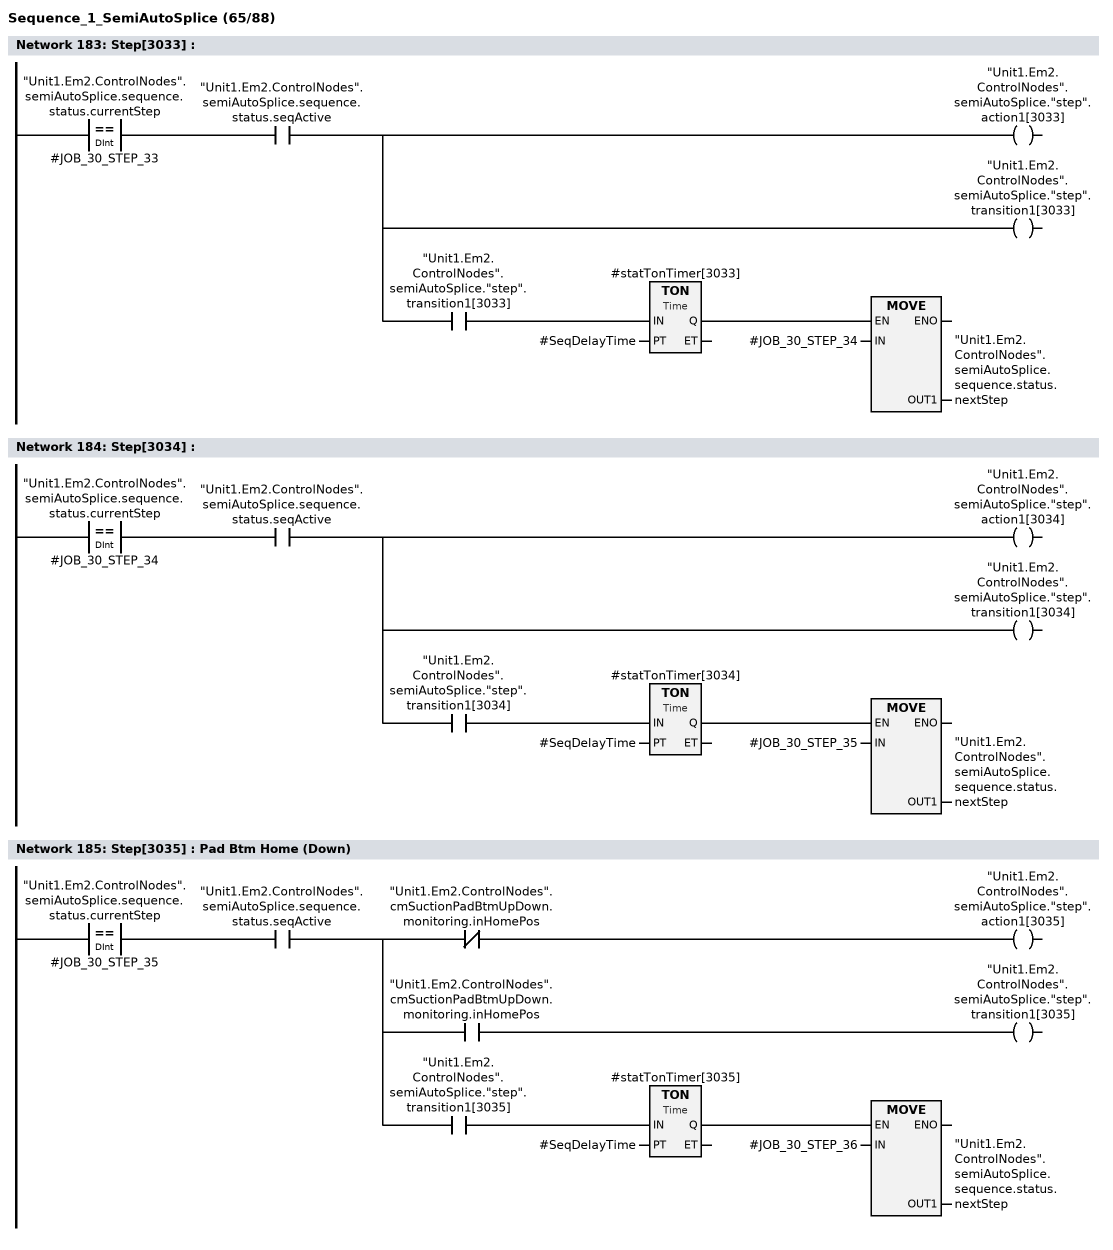
   RUNG wire#powerrail
      { S7_Templates := "SrcType := DInt" } EQ_Contact(in1 := "Unit1.Em2.ControlNodes".semiAutoSplice.sequence.status.currentStep, in2 := #JOB_30_STEP_33)
      Contact( "Unit1.Em2.ControlNodes".semiAutoSplice.sequence.status.seqActive )
      wire#w1
      Coil( "Unit1.Em2.ControlNodes".semiAutoSplice."step".action1[3033] )
   END_RUNG
   RUNG wire#w1
      Coil( "Unit1.Em2.ControlNodes".semiAutoSplice."step".transition1[3033] )
   END_RUNG
   RUNG wire#w1
      Contact( "Unit1.Em2.ControlNodes".semiAutoSplice."step".transition1[3033] )
      { S7_Templates := "time_type := Time" } #statTonTimer[3033].TON(pt := #SeqDelayTime, et =>)
      Move(in := #JOB_30_STEP_34, out1 => "Unit1.Em2.ControlNodes".semiAutoSplice.sequence.status.nextStep)
   END_RUNG
   // the same network as SCL:
   "Unit1.Em2.ControlNodes".semiAutoSplice."step".action1[3033] := ("Unit1.Em2.ControlNodes".semiAutoSplice.sequence.status.currentStep = #JOB_30_STEP_33) AND "Unit1.Em2.ControlNodes".semiAutoSplice.sequence.status.seqActive;
   "Unit1.Em2.ControlNodes".semiAutoSplice."step".transition1[3033] := ("Unit1.Em2.ControlNodes".semiAutoSplice.sequence.status.currentStep = #JOB_30_STEP_33) AND "Unit1.Em2.ControlNodes".semiAutoSplice.sequence.status.seqActive;
   #statTonTimer[3033].TON(IN := ("Unit1.Em2.ControlNodes".semiAutoSplice.sequence.status.currentStep = #JOB_30_STEP_33) AND "Unit1.Em2.ControlNodes".semiAutoSplice.sequence.status.seqActive AND "Unit1.Em2.ControlNodes".semiAutoSplice."step".transition1[3033],
                           PT := #SeqDelayTime);
   IF #statTonTimer[3033].Q THEN
       "Unit1.Em2.ControlNodes".semiAutoSplice.sequence.status.nextStep := #JOB_30_STEP_34;
   END_IF;
END_REGION

REGION Network 184: Step[3034] :
   RUNG wire#powerrail
      { S7_Templates := "SrcType := DInt" } EQ_Contact(in1 := "Unit1.Em2.ControlNodes".semiAutoSplice.sequence.status.currentStep, in2 := #JOB_30_STEP_34)
      Contact( "Unit1.Em2.ControlNodes".semiAutoSplice.sequence.status.seqActive )
      wire#w1
      Coil( "Unit1.Em2.ControlNodes".semiAutoSplice."step".action1[3034] )
   END_RUNG
   RUNG wire#w1
      Coil( "Unit1.Em2.ControlNodes".semiAutoSplice."step".transition1[3034] )
   END_RUNG
   RUNG wire#w1
      Contact( "Unit1.Em2.ControlNodes".semiAutoSplice."step".transition1[3034] )
      { S7_Templates := "time_type := Time" } #statTonTimer[3034].TON(pt := #SeqDelayTime, et =>)
      Move(in := #JOB_30_STEP_35, out1 => "Unit1.Em2.ControlNodes".semiAutoSplice.sequence.status.nextStep)
   END_RUNG
   // the same network as SCL:
   "Unit1.Em2.ControlNodes".semiAutoSplice."step".action1[3034] := ("Unit1.Em2.ControlNodes".semiAutoSplice.sequence.status.currentStep = #JOB_30_STEP_34) AND "Unit1.Em2.ControlNodes".semiAutoSplice.sequence.status.seqActive;
   "Unit1.Em2.ControlNodes".semiAutoSplice."step".transition1[3034] := ("Unit1.Em2.ControlNodes".semiAutoSplice.sequence.status.currentStep = #JOB_30_STEP_34) AND "Unit1.Em2.ControlNodes".semiAutoSplice.sequence.status.seqActive;
   #statTonTimer[3034].TON(IN := ("Unit1.Em2.ControlNodes".semiAutoSplice.sequence.status.currentStep = #JOB_30_STEP_34) AND "Unit1.Em2.ControlNodes".semiAutoSplice.sequence.status.seqActive AND "Unit1.Em2.ControlNodes".semiAutoSplice."step".transition1[3034],
                           PT := #SeqDelayTime);
   IF #statTonTimer[3034].Q THEN
       "Unit1.Em2.ControlNodes".semiAutoSplice.sequence.status.nextStep := #JOB_30_STEP_35;
   END_IF;
END_REGION

REGION Network 185: Step[3035] : Pad Btm Home (Down)
   RUNG wire#powerrail
      { S7_Templates := "SrcType := DInt" } EQ_Contact(in1 := "Unit1.Em2.ControlNodes".semiAutoSplice.sequence.status.currentStep, in2 := #JOB_30_STEP_35)
      Contact( "Unit1.Em2.ControlNodes".semiAutoSplice.sequence.status.seqActive )
      wire#w1
      I_Contact( "Unit1.Em2.ControlNodes".cmSuctionPadBtmUpDown.monitoring.inHomePos )
      Coil( "Unit1.Em2.ControlNodes".semiAutoSplice."step".action1[3035] )
   END_RUNG
   RUNG wire#w1
      Contact( "Unit1.Em2.ControlNodes".cmSuctionPadBtmUpDown.monitoring.inHomePos )
      Coil( "Unit1.Em2.ControlNodes".semiAutoSplice."step".transition1[3035] )
   END_RUNG
   RUNG wire#w1
      Contact( "Unit1.Em2.ControlNodes".semiAutoSplice."step".transition1[3035] )
      { S7_Templates := "time_type := Time" } #statTonTimer[3035].TON(pt := #SeqDelayTime, et =>)
      Move(in := #JOB_30_STEP_36, out1 => "Unit1.Em2.ControlNodes".semiAutoSplice.sequence.status.nextStep)
   END_RUNG
   // the same network as SCL:
   #_w1 := ("Unit1.Em2.ControlNodes".semiAutoSplice.sequence.status.currentStep = #JOB_30_STEP_35) AND "Unit1.Em2.ControlNodes".semiAutoSplice.sequence.status.seqActive;
   "Unit1.Em2.ControlNodes".semiAutoSplice."step".action1[3035] := #_w1 AND NOT "Unit1.Em2.ControlNodes".cmSuctionPadBtmUpDown.monitoring.inHomePos;
   "Unit1.Em2.ControlNodes".semiAutoSplice."step".transition1[3035] := #_w1 AND "Unit1.Em2.ControlNodes".cmSuctionPadBtmUpDown.monitoring.inHomePos;
   #statTonTimer[3035].TON(IN := #_w1 AND "Unit1.Em2.ControlNodes".semiAutoSplice."step".transition1[3035],
                           PT := #SeqDelayTime);
   IF #statTonTimer[3035].Q THEN
       "Unit1.Em2.ControlNodes".semiAutoSplice.sequence.status.nextStep := #JOB_30_STEP_36;
   END_IF;
END_REGION

REGION Network 186: Step[3036] :
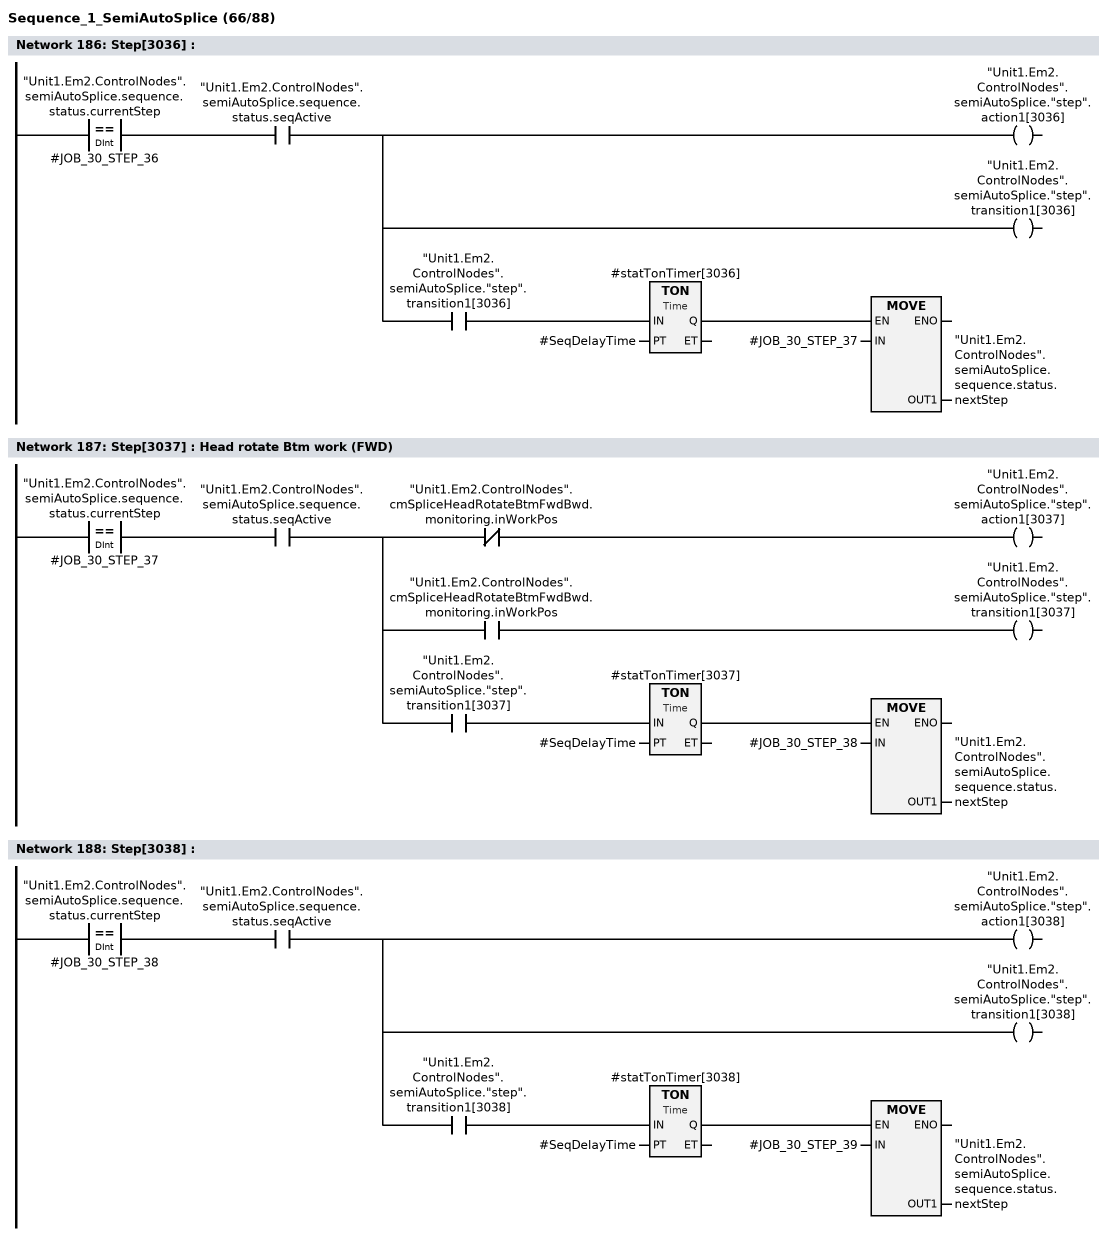
   RUNG wire#powerrail
      { S7_Templates := "SrcType := DInt" } EQ_Contact(in1 := "Unit1.Em2.ControlNodes".semiAutoSplice.sequence.status.currentStep, in2 := #JOB_30_STEP_36)
      Contact( "Unit1.Em2.ControlNodes".semiAutoSplice.sequence.status.seqActive )
      wire#w1
      Coil( "Unit1.Em2.ControlNodes".semiAutoSplice."step".action1[3036] )
   END_RUNG
   RUNG wire#w1
      Coil( "Unit1.Em2.ControlNodes".semiAutoSplice."step".transition1[3036] )
   END_RUNG
   RUNG wire#w1
      Contact( "Unit1.Em2.ControlNodes".semiAutoSplice."step".transition1[3036] )
      { S7_Templates := "time_type := Time" } #statTonTimer[3036].TON(pt := #SeqDelayTime, et =>)
      Move(in := #JOB_30_STEP_37, out1 => "Unit1.Em2.ControlNodes".semiAutoSplice.sequence.status.nextStep)
   END_RUNG
   // the same network as SCL:
   "Unit1.Em2.ControlNodes".semiAutoSplice."step".action1[3036] := ("Unit1.Em2.ControlNodes".semiAutoSplice.sequence.status.currentStep = #JOB_30_STEP_36) AND "Unit1.Em2.ControlNodes".semiAutoSplice.sequence.status.seqActive;
   "Unit1.Em2.ControlNodes".semiAutoSplice."step".transition1[3036] := ("Unit1.Em2.ControlNodes".semiAutoSplice.sequence.status.currentStep = #JOB_30_STEP_36) AND "Unit1.Em2.ControlNodes".semiAutoSplice.sequence.status.seqActive;
   #statTonTimer[3036].TON(IN := ("Unit1.Em2.ControlNodes".semiAutoSplice.sequence.status.currentStep = #JOB_30_STEP_36) AND "Unit1.Em2.ControlNodes".semiAutoSplice.sequence.status.seqActive AND "Unit1.Em2.ControlNodes".semiAutoSplice."step".transition1[3036],
                           PT := #SeqDelayTime);
   IF #statTonTimer[3036].Q THEN
       "Unit1.Em2.ControlNodes".semiAutoSplice.sequence.status.nextStep := #JOB_30_STEP_37;
   END_IF;
END_REGION

REGION Network 187: Step[3037] : Head rotate Btm work (FWD)
   RUNG wire#powerrail
      { S7_Templates := "SrcType := DInt" } EQ_Contact(in1 := "Unit1.Em2.ControlNodes".semiAutoSplice.sequence.status.currentStep, in2 := #JOB_30_STEP_37)
      Contact( "Unit1.Em2.ControlNodes".semiAutoSplice.sequence.status.seqActive )
      wire#w1
      I_Contact( "Unit1.Em2.ControlNodes".cmSpliceHeadRotateBtmFwdBwd.monitoring.inWorkPos )
      Coil( "Unit1.Em2.ControlNodes".semiAutoSplice."step".action1[3037] )
   END_RUNG
   RUNG wire#w1
      Contact( "Unit1.Em2.ControlNodes".cmSpliceHeadRotateBtmFwdBwd.monitoring.inWorkPos )
      Coil( "Unit1.Em2.ControlNodes".semiAutoSplice."step".transition1[3037] )
   END_RUNG
   RUNG wire#w1
      Contact( "Unit1.Em2.ControlNodes".semiAutoSplice."step".transition1[3037] )
      { S7_Templates := "time_type := Time" } #statTonTimer[3037].TON(pt := #SeqDelayTime, et =>)
      Move(in := #JOB_30_STEP_38, out1 => "Unit1.Em2.ControlNodes".semiAutoSplice.sequence.status.nextStep)
   END_RUNG
   // the same network as SCL:
   #_w1 := ("Unit1.Em2.ControlNodes".semiAutoSplice.sequence.status.currentStep = #JOB_30_STEP_37) AND "Unit1.Em2.ControlNodes".semiAutoSplice.sequence.status.seqActive;
   "Unit1.Em2.ControlNodes".semiAutoSplice."step".action1[3037] := #_w1 AND NOT "Unit1.Em2.ControlNodes".cmSpliceHeadRotateBtmFwdBwd.monitoring.inWorkPos;
   "Unit1.Em2.ControlNodes".semiAutoSplice."step".transition1[3037] := #_w1 AND "Unit1.Em2.ControlNodes".cmSpliceHeadRotateBtmFwdBwd.monitoring.inWorkPos;
   #statTonTimer[3037].TON(IN := #_w1 AND "Unit1.Em2.ControlNodes".semiAutoSplice."step".transition1[3037],
                           PT := #SeqDelayTime);
   IF #statTonTimer[3037].Q THEN
       "Unit1.Em2.ControlNodes".semiAutoSplice.sequence.status.nextStep := #JOB_30_STEP_38;
   END_IF;
END_REGION

REGION Network 188: Step[3038] :
   RUNG wire#powerrail
      { S7_Templates := "SrcType := DInt" } EQ_Contact(in1 := "Unit1.Em2.ControlNodes".semiAutoSplice.sequence.status.currentStep, in2 := #JOB_30_STEP_38)
      Contact( "Unit1.Em2.ControlNodes".semiAutoSplice.sequence.status.seqActive )
      wire#w1
      Coil( "Unit1.Em2.ControlNodes".semiAutoSplice."step".action1[3038] )
   END_RUNG
   RUNG wire#w1
      Coil( "Unit1.Em2.ControlNodes".semiAutoSplice."step".transition1[3038] )
   END_RUNG
   RUNG wire#w1
      Contact( "Unit1.Em2.ControlNodes".semiAutoSplice."step".transition1[3038] )
      { S7_Templates := "time_type := Time" } #statTonTimer[3038].TON(pt := #SeqDelayTime, et =>)
      Move(in := #JOB_30_STEP_39, out1 => "Unit1.Em2.ControlNodes".semiAutoSplice.sequence.status.nextStep)
   END_RUNG
   // the same network as SCL:
   "Unit1.Em2.ControlNodes".semiAutoSplice."step".action1[3038] := ("Unit1.Em2.ControlNodes".semiAutoSplice.sequence.status.currentStep = #JOB_30_STEP_38) AND "Unit1.Em2.ControlNodes".semiAutoSplice.sequence.status.seqActive;
   "Unit1.Em2.ControlNodes".semiAutoSplice."step".transition1[3038] := ("Unit1.Em2.ControlNodes".semiAutoSplice.sequence.status.currentStep = #JOB_30_STEP_38) AND "Unit1.Em2.ControlNodes".semiAutoSplice.sequence.status.seqActive;
   #statTonTimer[3038].TON(IN := ("Unit1.Em2.ControlNodes".semiAutoSplice.sequence.status.currentStep = #JOB_30_STEP_38) AND "Unit1.Em2.ControlNodes".semiAutoSplice.sequence.status.seqActive AND "Unit1.Em2.ControlNodes".semiAutoSplice."step".transition1[3038],
                           PT := #SeqDelayTime);
   IF #statTonTimer[3038].Q THEN
       "Unit1.Em2.ControlNodes".semiAutoSplice.sequence.status.nextStep := #JOB_30_STEP_39;
   END_IF;
END_REGION

REGION Network 189: Step[3039] : Tape Btm work (Up)
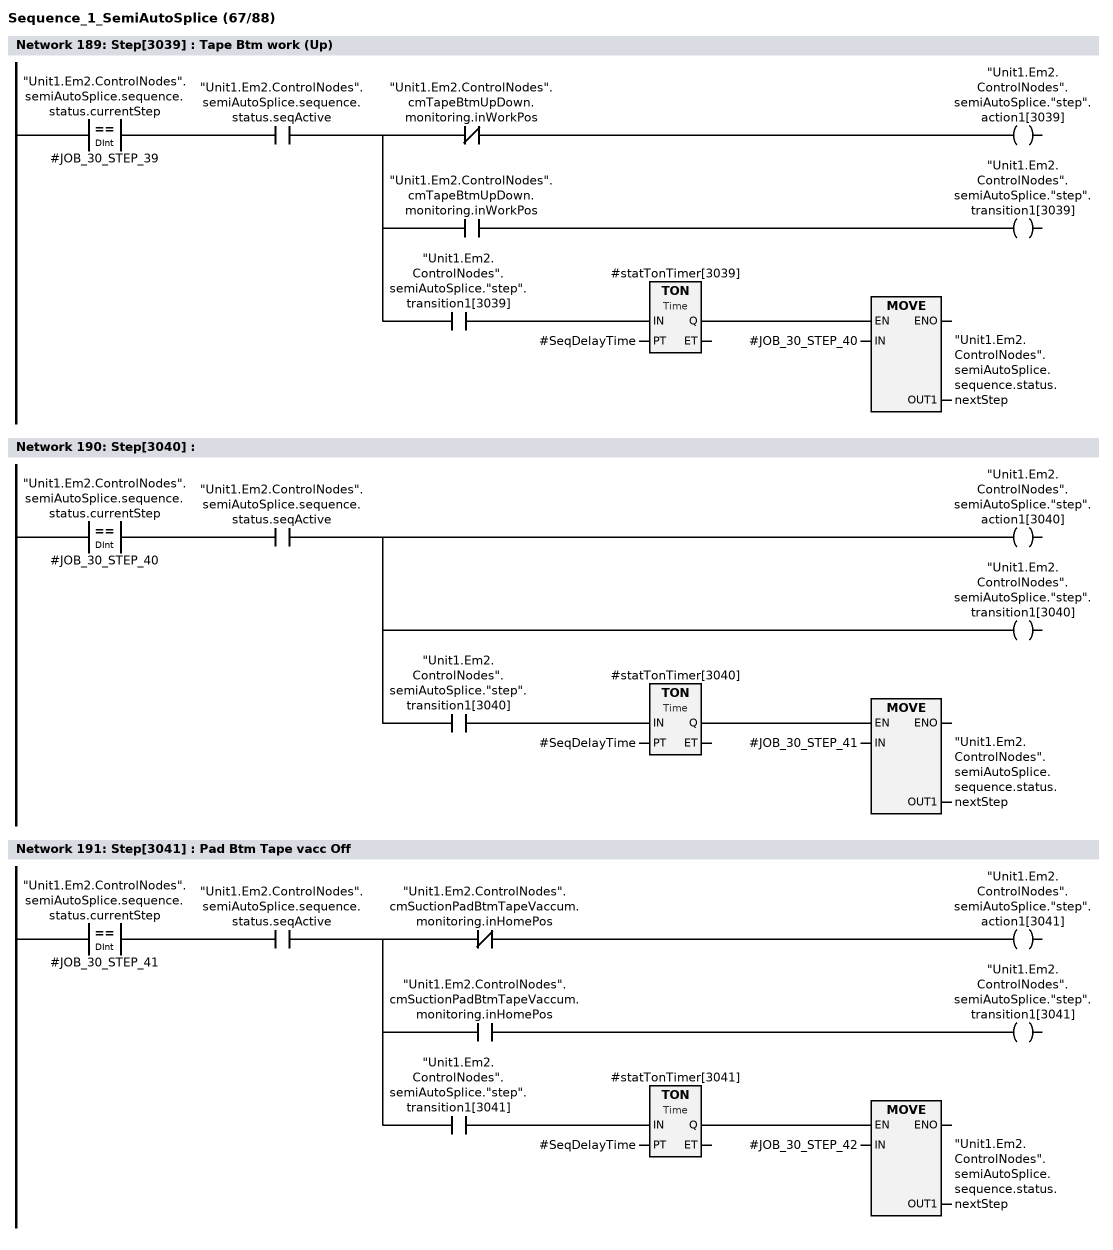
   RUNG wire#powerrail
      { S7_Templates := "SrcType := DInt" } EQ_Contact(in1 := "Unit1.Em2.ControlNodes".semiAutoSplice.sequence.status.currentStep, in2 := #JOB_30_STEP_39)
      Contact( "Unit1.Em2.ControlNodes".semiAutoSplice.sequence.status.seqActive )
      wire#w1
      I_Contact( "Unit1.Em2.ControlNodes".cmTapeBtmUpDown.monitoring.inWorkPos )
      Coil( "Unit1.Em2.ControlNodes".semiAutoSplice."step".action1[3039] )
   END_RUNG
   RUNG wire#w1
      Contact( "Unit1.Em2.ControlNodes".cmTapeBtmUpDown.monitoring.inWorkPos )
      Coil( "Unit1.Em2.ControlNodes".semiAutoSplice."step".transition1[3039] )
   END_RUNG
   RUNG wire#w1
      Contact( "Unit1.Em2.ControlNodes".semiAutoSplice."step".transition1[3039] )
      { S7_Templates := "time_type := Time" } #statTonTimer[3039].TON(pt := #SeqDelayTime, et =>)
      Move(in := #JOB_30_STEP_40, out1 => "Unit1.Em2.ControlNodes".semiAutoSplice.sequence.status.nextStep)
   END_RUNG
   // the same network as SCL:
   #_w1 := ("Unit1.Em2.ControlNodes".semiAutoSplice.sequence.status.currentStep = #JOB_30_STEP_39) AND "Unit1.Em2.ControlNodes".semiAutoSplice.sequence.status.seqActive;
   "Unit1.Em2.ControlNodes".semiAutoSplice."step".action1[3039] := #_w1 AND NOT "Unit1.Em2.ControlNodes".cmTapeBtmUpDown.monitoring.inWorkPos;
   "Unit1.Em2.ControlNodes".semiAutoSplice."step".transition1[3039] := #_w1 AND "Unit1.Em2.ControlNodes".cmTapeBtmUpDown.monitoring.inWorkPos;
   #statTonTimer[3039].TON(IN := #_w1 AND "Unit1.Em2.ControlNodes".semiAutoSplice."step".transition1[3039],
                           PT := #SeqDelayTime);
   IF #statTonTimer[3039].Q THEN
       "Unit1.Em2.ControlNodes".semiAutoSplice.sequence.status.nextStep := #JOB_30_STEP_40;
   END_IF;
END_REGION

REGION Network 190: Step[3040] :
   RUNG wire#powerrail
      { S7_Templates := "SrcType := DInt" } EQ_Contact(in1 := "Unit1.Em2.ControlNodes".semiAutoSplice.sequence.status.currentStep, in2 := #JOB_30_STEP_40)
      Contact( "Unit1.Em2.ControlNodes".semiAutoSplice.sequence.status.seqActive )
      wire#w1
      Coil( "Unit1.Em2.ControlNodes".semiAutoSplice."step".action1[3040] )
   END_RUNG
   RUNG wire#w1
      Coil( "Unit1.Em2.ControlNodes".semiAutoSplice."step".transition1[3040] )
   END_RUNG
   RUNG wire#w1
      Contact( "Unit1.Em2.ControlNodes".semiAutoSplice."step".transition1[3040] )
      { S7_Templates := "time_type := Time" } #statTonTimer[3040].TON(pt := #SeqDelayTime, et =>)
      Move(in := #JOB_30_STEP_41, out1 => "Unit1.Em2.ControlNodes".semiAutoSplice.sequence.status.nextStep)
   END_RUNG
   // the same network as SCL:
   "Unit1.Em2.ControlNodes".semiAutoSplice."step".action1[3040] := ("Unit1.Em2.ControlNodes".semiAutoSplice.sequence.status.currentStep = #JOB_30_STEP_40) AND "Unit1.Em2.ControlNodes".semiAutoSplice.sequence.status.seqActive;
   "Unit1.Em2.ControlNodes".semiAutoSplice."step".transition1[3040] := ("Unit1.Em2.ControlNodes".semiAutoSplice.sequence.status.currentStep = #JOB_30_STEP_40) AND "Unit1.Em2.ControlNodes".semiAutoSplice.sequence.status.seqActive;
   #statTonTimer[3040].TON(IN := ("Unit1.Em2.ControlNodes".semiAutoSplice.sequence.status.currentStep = #JOB_30_STEP_40) AND "Unit1.Em2.ControlNodes".semiAutoSplice.sequence.status.seqActive AND "Unit1.Em2.ControlNodes".semiAutoSplice."step".transition1[3040],
                           PT := #SeqDelayTime);
   IF #statTonTimer[3040].Q THEN
       "Unit1.Em2.ControlNodes".semiAutoSplice.sequence.status.nextStep := #JOB_30_STEP_41;
   END_IF;
END_REGION

REGION Network 191: Step[3041] : Pad Btm Tape vacc Off
   RUNG wire#powerrail
      { S7_Templates := "SrcType := DInt" } EQ_Contact(in1 := "Unit1.Em2.ControlNodes".semiAutoSplice.sequence.status.currentStep, in2 := #JOB_30_STEP_41)
      Contact( "Unit1.Em2.ControlNodes".semiAutoSplice.sequence.status.seqActive )
      wire#w1
      I_Contact( "Unit1.Em2.ControlNodes".cmSuctionPadBtmTapeVaccum.monitoring.inHomePos )
      Coil( "Unit1.Em2.ControlNodes".semiAutoSplice."step".action1[3041] )
   END_RUNG
   RUNG wire#w1
      Contact( "Unit1.Em2.ControlNodes".cmSuctionPadBtmTapeVaccum.monitoring.inHomePos )
      Coil( "Unit1.Em2.ControlNodes".semiAutoSplice."step".transition1[3041] )
   END_RUNG
   RUNG wire#w1
      Contact( "Unit1.Em2.ControlNodes".semiAutoSplice."step".transition1[3041] )
      { S7_Templates := "time_type := Time" } #statTonTimer[3041].TON(pt := #SeqDelayTime, et =>)
      Move(in := #JOB_30_STEP_42, out1 => "Unit1.Em2.ControlNodes".semiAutoSplice.sequence.status.nextStep)
   END_RUNG
   // the same network as SCL:
   #_w1 := ("Unit1.Em2.ControlNodes".semiAutoSplice.sequence.status.currentStep = #JOB_30_STEP_41) AND "Unit1.Em2.ControlNodes".semiAutoSplice.sequence.status.seqActive;
   "Unit1.Em2.ControlNodes".semiAutoSplice."step".action1[3041] := #_w1 AND NOT "Unit1.Em2.ControlNodes".cmSuctionPadBtmTapeVaccum.monitoring.inHomePos;
   "Unit1.Em2.ControlNodes".semiAutoSplice."step".transition1[3041] := #_w1 AND "Unit1.Em2.ControlNodes".cmSuctionPadBtmTapeVaccum.monitoring.inHomePos;
   #statTonTimer[3041].TON(IN := #_w1 AND "Unit1.Em2.ControlNodes".semiAutoSplice."step".transition1[3041],
                           PT := #SeqDelayTime);
   IF #statTonTimer[3041].Q THEN
       "Unit1.Em2.ControlNodes".semiAutoSplice.sequence.status.nextStep := #JOB_30_STEP_42;
   END_IF;
END_REGION

REGION Network 192: Step[3042] :
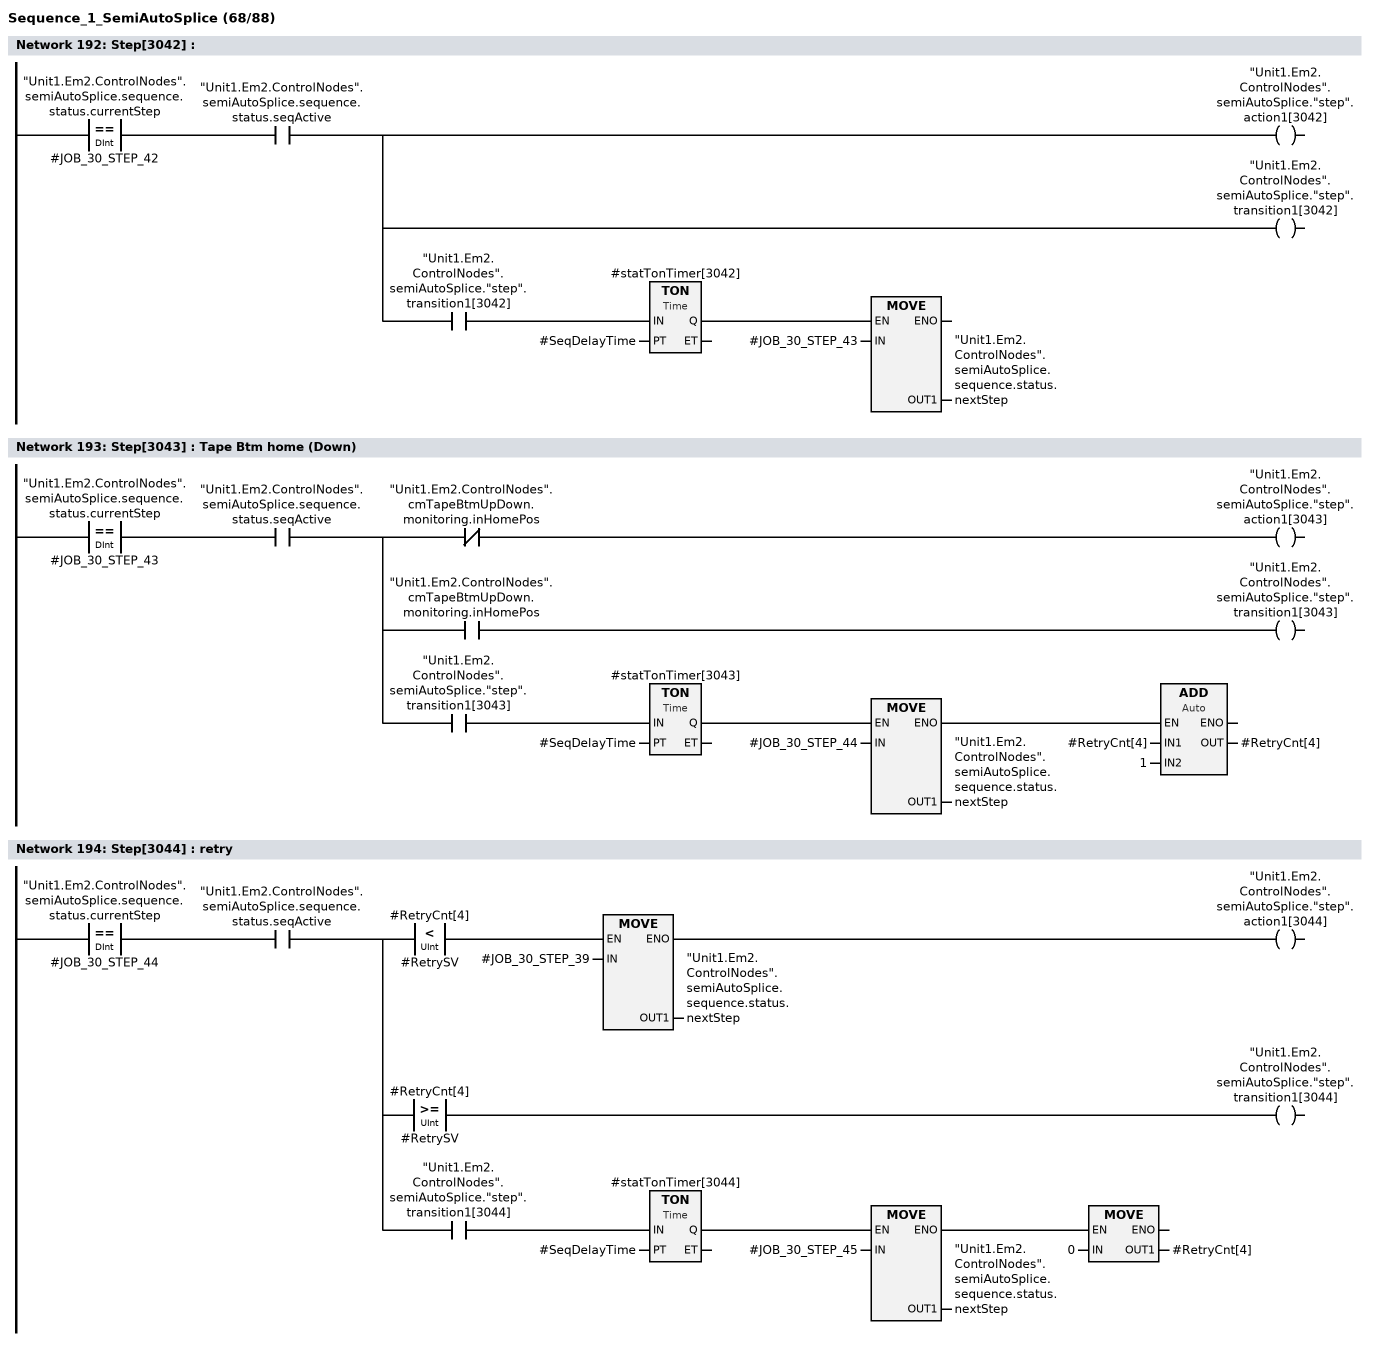
   RUNG wire#powerrail
      { S7_Templates := "SrcType := DInt" } EQ_Contact(in1 := "Unit1.Em2.ControlNodes".semiAutoSplice.sequence.status.currentStep, in2 := #JOB_30_STEP_42)
      Contact( "Unit1.Em2.ControlNodes".semiAutoSplice.sequence.status.seqActive )
      wire#w1
      Coil( "Unit1.Em2.ControlNodes".semiAutoSplice."step".action1[3042] )
   END_RUNG
   RUNG wire#w1
      Coil( "Unit1.Em2.ControlNodes".semiAutoSplice."step".transition1[3042] )
   END_RUNG
   RUNG wire#w1
      Contact( "Unit1.Em2.ControlNodes".semiAutoSplice."step".transition1[3042] )
      { S7_Templates := "time_type := Time" } #statTonTimer[3042].TON(pt := #SeqDelayTime, et =>)
      Move(in := #JOB_30_STEP_43, out1 => "Unit1.Em2.ControlNodes".semiAutoSplice.sequence.status.nextStep)
   END_RUNG
   // the same network as SCL:
   "Unit1.Em2.ControlNodes".semiAutoSplice."step".action1[3042] := ("Unit1.Em2.ControlNodes".semiAutoSplice.sequence.status.currentStep = #JOB_30_STEP_42) AND "Unit1.Em2.ControlNodes".semiAutoSplice.sequence.status.seqActive;
   "Unit1.Em2.ControlNodes".semiAutoSplice."step".transition1[3042] := ("Unit1.Em2.ControlNodes".semiAutoSplice.sequence.status.currentStep = #JOB_30_STEP_42) AND "Unit1.Em2.ControlNodes".semiAutoSplice.sequence.status.seqActive;
   #statTonTimer[3042].TON(IN := ("Unit1.Em2.ControlNodes".semiAutoSplice.sequence.status.currentStep = #JOB_30_STEP_42) AND "Unit1.Em2.ControlNodes".semiAutoSplice.sequence.status.seqActive AND "Unit1.Em2.ControlNodes".semiAutoSplice."step".transition1[3042],
                           PT := #SeqDelayTime);
   IF #statTonTimer[3042].Q THEN
       "Unit1.Em2.ControlNodes".semiAutoSplice.sequence.status.nextStep := #JOB_30_STEP_43;
   END_IF;
END_REGION

REGION Network 193: Step[3043] : Tape Btm home (Down)
   RUNG wire#powerrail
      { S7_Templates := "SrcType := DInt" } EQ_Contact(in1 := "Unit1.Em2.ControlNodes".semiAutoSplice.sequence.status.currentStep, in2 := #JOB_30_STEP_43)
      Contact( "Unit1.Em2.ControlNodes".semiAutoSplice.sequence.status.seqActive )
      wire#w1
      I_Contact( "Unit1.Em2.ControlNodes".cmTapeBtmUpDown.monitoring.inHomePos )
      Coil( "Unit1.Em2.ControlNodes".semiAutoSplice."step".action1[3043] )
   END_RUNG
   RUNG wire#w1
      Contact( "Unit1.Em2.ControlNodes".cmTapeBtmUpDown.monitoring.inHomePos )
      Coil( "Unit1.Em2.ControlNodes".semiAutoSplice."step".transition1[3043] )
   END_RUNG
   RUNG wire#w1
      Contact( "Unit1.Em2.ControlNodes".semiAutoSplice."step".transition1[3043] )
      { S7_Templates := "time_type := Time" } #statTonTimer[3043].TON(pt := #SeqDelayTime, et =>)
      Move(in := #JOB_30_STEP_44, out1 => "Unit1.Em2.ControlNodes".semiAutoSplice.sequence.status.nextStep)
      Add(in1 := #RetryCnt[4], in2 := 1, out => #RetryCnt[4])
   END_RUNG
   // the same network as SCL:
   #_w1 := ("Unit1.Em2.ControlNodes".semiAutoSplice.sequence.status.currentStep = #JOB_30_STEP_43) AND "Unit1.Em2.ControlNodes".semiAutoSplice.sequence.status.seqActive;
   "Unit1.Em2.ControlNodes".semiAutoSplice."step".action1[3043] := #_w1 AND NOT "Unit1.Em2.ControlNodes".cmTapeBtmUpDown.monitoring.inHomePos;
   "Unit1.Em2.ControlNodes".semiAutoSplice."step".transition1[3043] := #_w1 AND "Unit1.Em2.ControlNodes".cmTapeBtmUpDown.monitoring.inHomePos;
   #statTonTimer[3043].TON(IN := #_w1 AND "Unit1.Em2.ControlNodes".semiAutoSplice."step".transition1[3043],
                           PT := #SeqDelayTime);
   IF #statTonTimer[3043].Q THEN
       "Unit1.Em2.ControlNodes".semiAutoSplice.sequence.status.nextStep := #JOB_30_STEP_44;
       #RetryCnt[4] := #RetryCnt[4] + 1;
   END_IF;
END_REGION

REGION Network 194: Step[3044] : retry
   RUNG wire#powerrail
      { S7_Templates := "SrcType := DInt" } EQ_Contact(in1 := "Unit1.Em2.ControlNodes".semiAutoSplice.sequence.status.currentStep, in2 := #JOB_30_STEP_44)
      Contact( "Unit1.Em2.ControlNodes".semiAutoSplice.sequence.status.seqActive )
      wire#w1
      { S7_Templates := "SrcType := UInt" } LT_Contact(in1 := #RetryCnt[4], in2 := #RetrySV)
      Move(in := #JOB_30_STEP_39, out1 => "Unit1.Em2.ControlNodes".semiAutoSplice.sequence.status.nextStep)
      Coil( "Unit1.Em2.ControlNodes".semiAutoSplice."step".action1[3044] )
   END_RUNG
   RUNG wire#w1
      { S7_Templates := "SrcType := UInt" } GE_Contact(in1 := #RetryCnt[4], in2 := #RetrySV)
      Coil( "Unit1.Em2.ControlNodes".semiAutoSplice."step".transition1[3044] )
   END_RUNG
   RUNG wire#w1
      Contact( "Unit1.Em2.ControlNodes".semiAutoSplice."step".transition1[3044] )
      { S7_Templates := "time_type := Time" } #statTonTimer[3044].TON(pt := #SeqDelayTime, et =>)
      Move(in := #JOB_30_STEP_45, out1 => "Unit1.Em2.ControlNodes".semiAutoSplice.sequence.status.nextStep)
      Move(in := 0, out1 => #RetryCnt[4])
   END_RUNG
   // the same network as SCL:
   #_w1 := ("Unit1.Em2.ControlNodes".semiAutoSplice.sequence.status.currentStep = #JOB_30_STEP_44) AND "Unit1.Em2.ControlNodes".semiAutoSplice.sequence.status.seqActive;
   #_w2 := #_w1 AND (#RetryCnt[4] < #RetrySV);
   IF #_w2 THEN "Unit1.Em2.ControlNodes".semiAutoSplice.sequence.status.nextStep := #JOB_30_STEP_39; END_IF;
   "Unit1.Em2.ControlNodes".semiAutoSplice."step".action1[3044] := #_w2;
   "Unit1.Em2.ControlNodes".semiAutoSplice."step".transition1[3044] := #_w1 AND (#RetryCnt[4] >= #RetrySV);
   #statTonTimer[3044].TON(IN := #_w1 AND "Unit1.Em2.ControlNodes".semiAutoSplice."step".transition1[3044],
                           PT := #SeqDelayTime);
   IF #statTonTimer[3044].Q THEN
       "Unit1.Em2.ControlNodes".semiAutoSplice.sequence.status.nextStep := #JOB_30_STEP_45;
       #RetryCnt[4] := 0;
   END_IF;
END_REGION

REGION Network 195: Step[3045] :
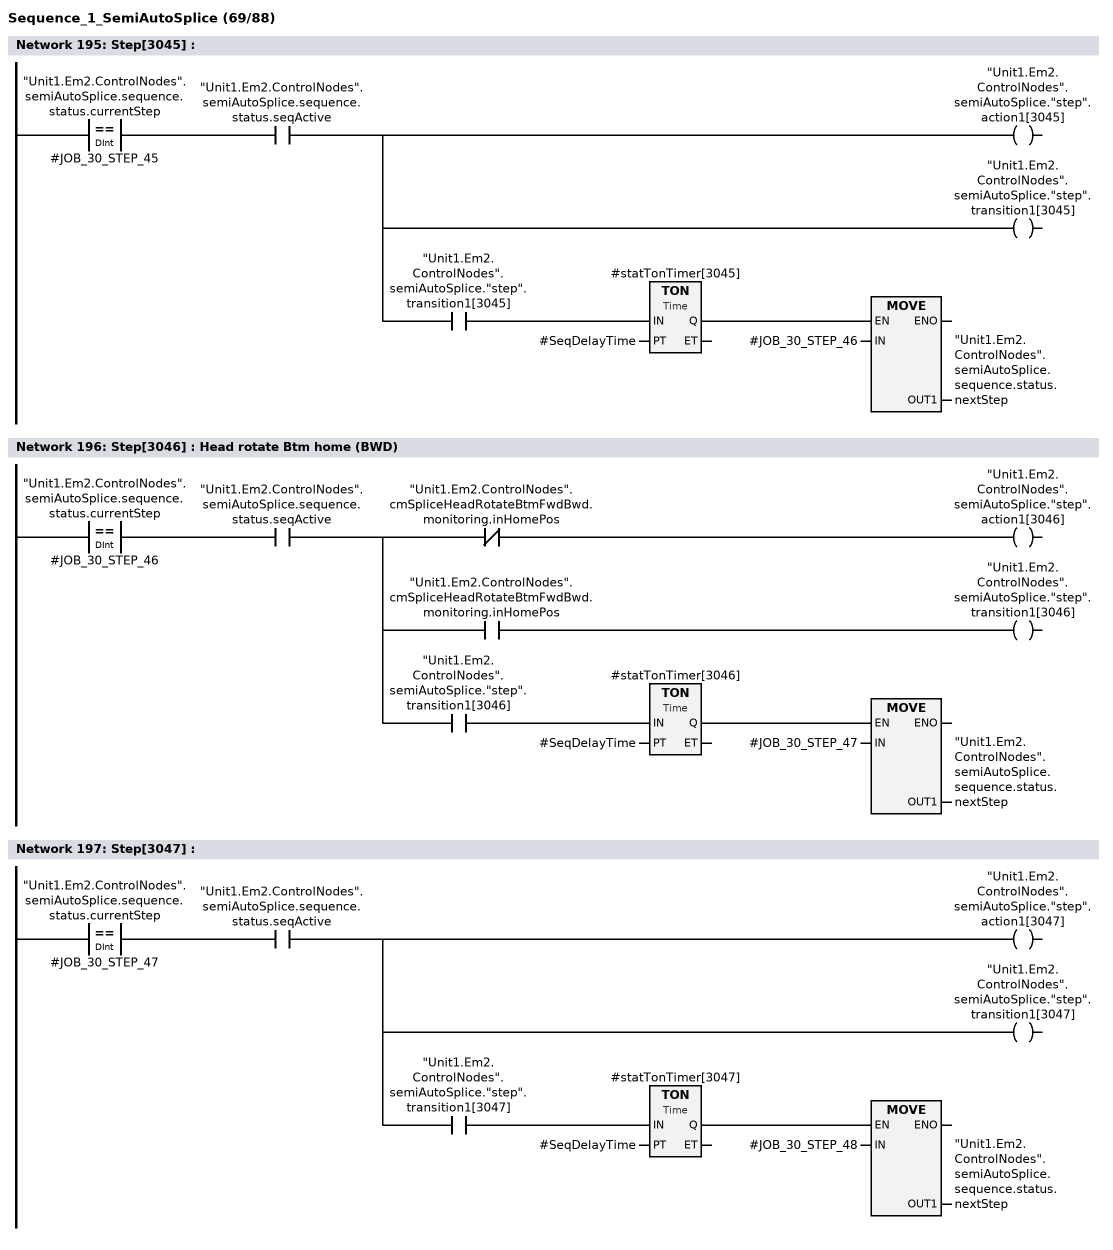
   RUNG wire#powerrail
      { S7_Templates := "SrcType := DInt" } EQ_Contact(in1 := "Unit1.Em2.ControlNodes".semiAutoSplice.sequence.status.currentStep, in2 := #JOB_30_STEP_45)
      Contact( "Unit1.Em2.ControlNodes".semiAutoSplice.sequence.status.seqActive )
      wire#w1
      Coil( "Unit1.Em2.ControlNodes".semiAutoSplice."step".action1[3045] )
   END_RUNG
   RUNG wire#w1
      Coil( "Unit1.Em2.ControlNodes".semiAutoSplice."step".transition1[3045] )
   END_RUNG
   RUNG wire#w1
      Contact( "Unit1.Em2.ControlNodes".semiAutoSplice."step".transition1[3045] )
      { S7_Templates := "time_type := Time" } #statTonTimer[3045].TON(pt := #SeqDelayTime, et =>)
      Move(in := #JOB_30_STEP_46, out1 => "Unit1.Em2.ControlNodes".semiAutoSplice.sequence.status.nextStep)
   END_RUNG
   // the same network as SCL:
   "Unit1.Em2.ControlNodes".semiAutoSplice."step".action1[3045] := ("Unit1.Em2.ControlNodes".semiAutoSplice.sequence.status.currentStep = #JOB_30_STEP_45) AND "Unit1.Em2.ControlNodes".semiAutoSplice.sequence.status.seqActive;
   "Unit1.Em2.ControlNodes".semiAutoSplice."step".transition1[3045] := ("Unit1.Em2.ControlNodes".semiAutoSplice.sequence.status.currentStep = #JOB_30_STEP_45) AND "Unit1.Em2.ControlNodes".semiAutoSplice.sequence.status.seqActive;
   #statTonTimer[3045].TON(IN := ("Unit1.Em2.ControlNodes".semiAutoSplice.sequence.status.currentStep = #JOB_30_STEP_45) AND "Unit1.Em2.ControlNodes".semiAutoSplice.sequence.status.seqActive AND "Unit1.Em2.ControlNodes".semiAutoSplice."step".transition1[3045],
                           PT := #SeqDelayTime);
   IF #statTonTimer[3045].Q THEN
       "Unit1.Em2.ControlNodes".semiAutoSplice.sequence.status.nextStep := #JOB_30_STEP_46;
   END_IF;
END_REGION

REGION Network 196: Step[3046] : Head rotate Btm home (BWD)
   RUNG wire#powerrail
      { S7_Templates := "SrcType := DInt" } EQ_Contact(in1 := "Unit1.Em2.ControlNodes".semiAutoSplice.sequence.status.currentStep, in2 := #JOB_30_STEP_46)
      Contact( "Unit1.Em2.ControlNodes".semiAutoSplice.sequence.status.seqActive )
      wire#w1
      I_Contact( "Unit1.Em2.ControlNodes".cmSpliceHeadRotateBtmFwdBwd.monitoring.inHomePos )
      Coil( "Unit1.Em2.ControlNodes".semiAutoSplice."step".action1[3046] )
   END_RUNG
   RUNG wire#w1
      Contact( "Unit1.Em2.ControlNodes".cmSpliceHeadRotateBtmFwdBwd.monitoring.inHomePos )
      Coil( "Unit1.Em2.ControlNodes".semiAutoSplice."step".transition1[3046] )
   END_RUNG
   RUNG wire#w1
      Contact( "Unit1.Em2.ControlNodes".semiAutoSplice."step".transition1[3046] )
      { S7_Templates := "time_type := Time" } #statTonTimer[3046].TON(pt := #SeqDelayTime, et =>)
      Move(in := #JOB_30_STEP_47, out1 => "Unit1.Em2.ControlNodes".semiAutoSplice.sequence.status.nextStep)
   END_RUNG
   // the same network as SCL:
   #_w1 := ("Unit1.Em2.ControlNodes".semiAutoSplice.sequence.status.currentStep = #JOB_30_STEP_46) AND "Unit1.Em2.ControlNodes".semiAutoSplice.sequence.status.seqActive;
   "Unit1.Em2.ControlNodes".semiAutoSplice."step".action1[3046] := #_w1 AND NOT "Unit1.Em2.ControlNodes".cmSpliceHeadRotateBtmFwdBwd.monitoring.inHomePos;
   "Unit1.Em2.ControlNodes".semiAutoSplice."step".transition1[3046] := #_w1 AND "Unit1.Em2.ControlNodes".cmSpliceHeadRotateBtmFwdBwd.monitoring.inHomePos;
   #statTonTimer[3046].TON(IN := #_w1 AND "Unit1.Em2.ControlNodes".semiAutoSplice."step".transition1[3046],
                           PT := #SeqDelayTime);
   IF #statTonTimer[3046].Q THEN
       "Unit1.Em2.ControlNodes".semiAutoSplice.sequence.status.nextStep := #JOB_30_STEP_47;
   END_IF;
END_REGION

REGION Network 197: Step[3047] :
   RUNG wire#powerrail
      { S7_Templates := "SrcType := DInt" } EQ_Contact(in1 := "Unit1.Em2.ControlNodes".semiAutoSplice.sequence.status.currentStep, in2 := #JOB_30_STEP_47)
      Contact( "Unit1.Em2.ControlNodes".semiAutoSplice.sequence.status.seqActive )
      wire#w1
      Coil( "Unit1.Em2.ControlNodes".semiAutoSplice."step".action1[3047] )
   END_RUNG
   RUNG wire#w1
      Coil( "Unit1.Em2.ControlNodes".semiAutoSplice."step".transition1[3047] )
   END_RUNG
   RUNG wire#w1
      Contact( "Unit1.Em2.ControlNodes".semiAutoSplice."step".transition1[3047] )
      { S7_Templates := "time_type := Time" } #statTonTimer[3047].TON(pt := #SeqDelayTime, et =>)
      Move(in := #JOB_30_STEP_48, out1 => "Unit1.Em2.ControlNodes".semiAutoSplice.sequence.status.nextStep)
   END_RUNG
   // the same network as SCL:
   "Unit1.Em2.ControlNodes".semiAutoSplice."step".action1[3047] := ("Unit1.Em2.ControlNodes".semiAutoSplice.sequence.status.currentStep = #JOB_30_STEP_47) AND "Unit1.Em2.ControlNodes".semiAutoSplice.sequence.status.seqActive;
   "Unit1.Em2.ControlNodes".semiAutoSplice."step".transition1[3047] := ("Unit1.Em2.ControlNodes".semiAutoSplice.sequence.status.currentStep = #JOB_30_STEP_47) AND "Unit1.Em2.ControlNodes".semiAutoSplice.sequence.status.seqActive;
   #statTonTimer[3047].TON(IN := ("Unit1.Em2.ControlNodes".semiAutoSplice.sequence.status.currentStep = #JOB_30_STEP_47) AND "Unit1.Em2.ControlNodes".semiAutoSplice.sequence.status.seqActive AND "Unit1.Em2.ControlNodes".semiAutoSplice."step".transition1[3047],
                           PT := #SeqDelayTime);
   IF #statTonTimer[3047].Q THEN
       "Unit1.Em2.ControlNodes".semiAutoSplice.sequence.status.nextStep := #JOB_30_STEP_48;
   END_IF;
END_REGION

